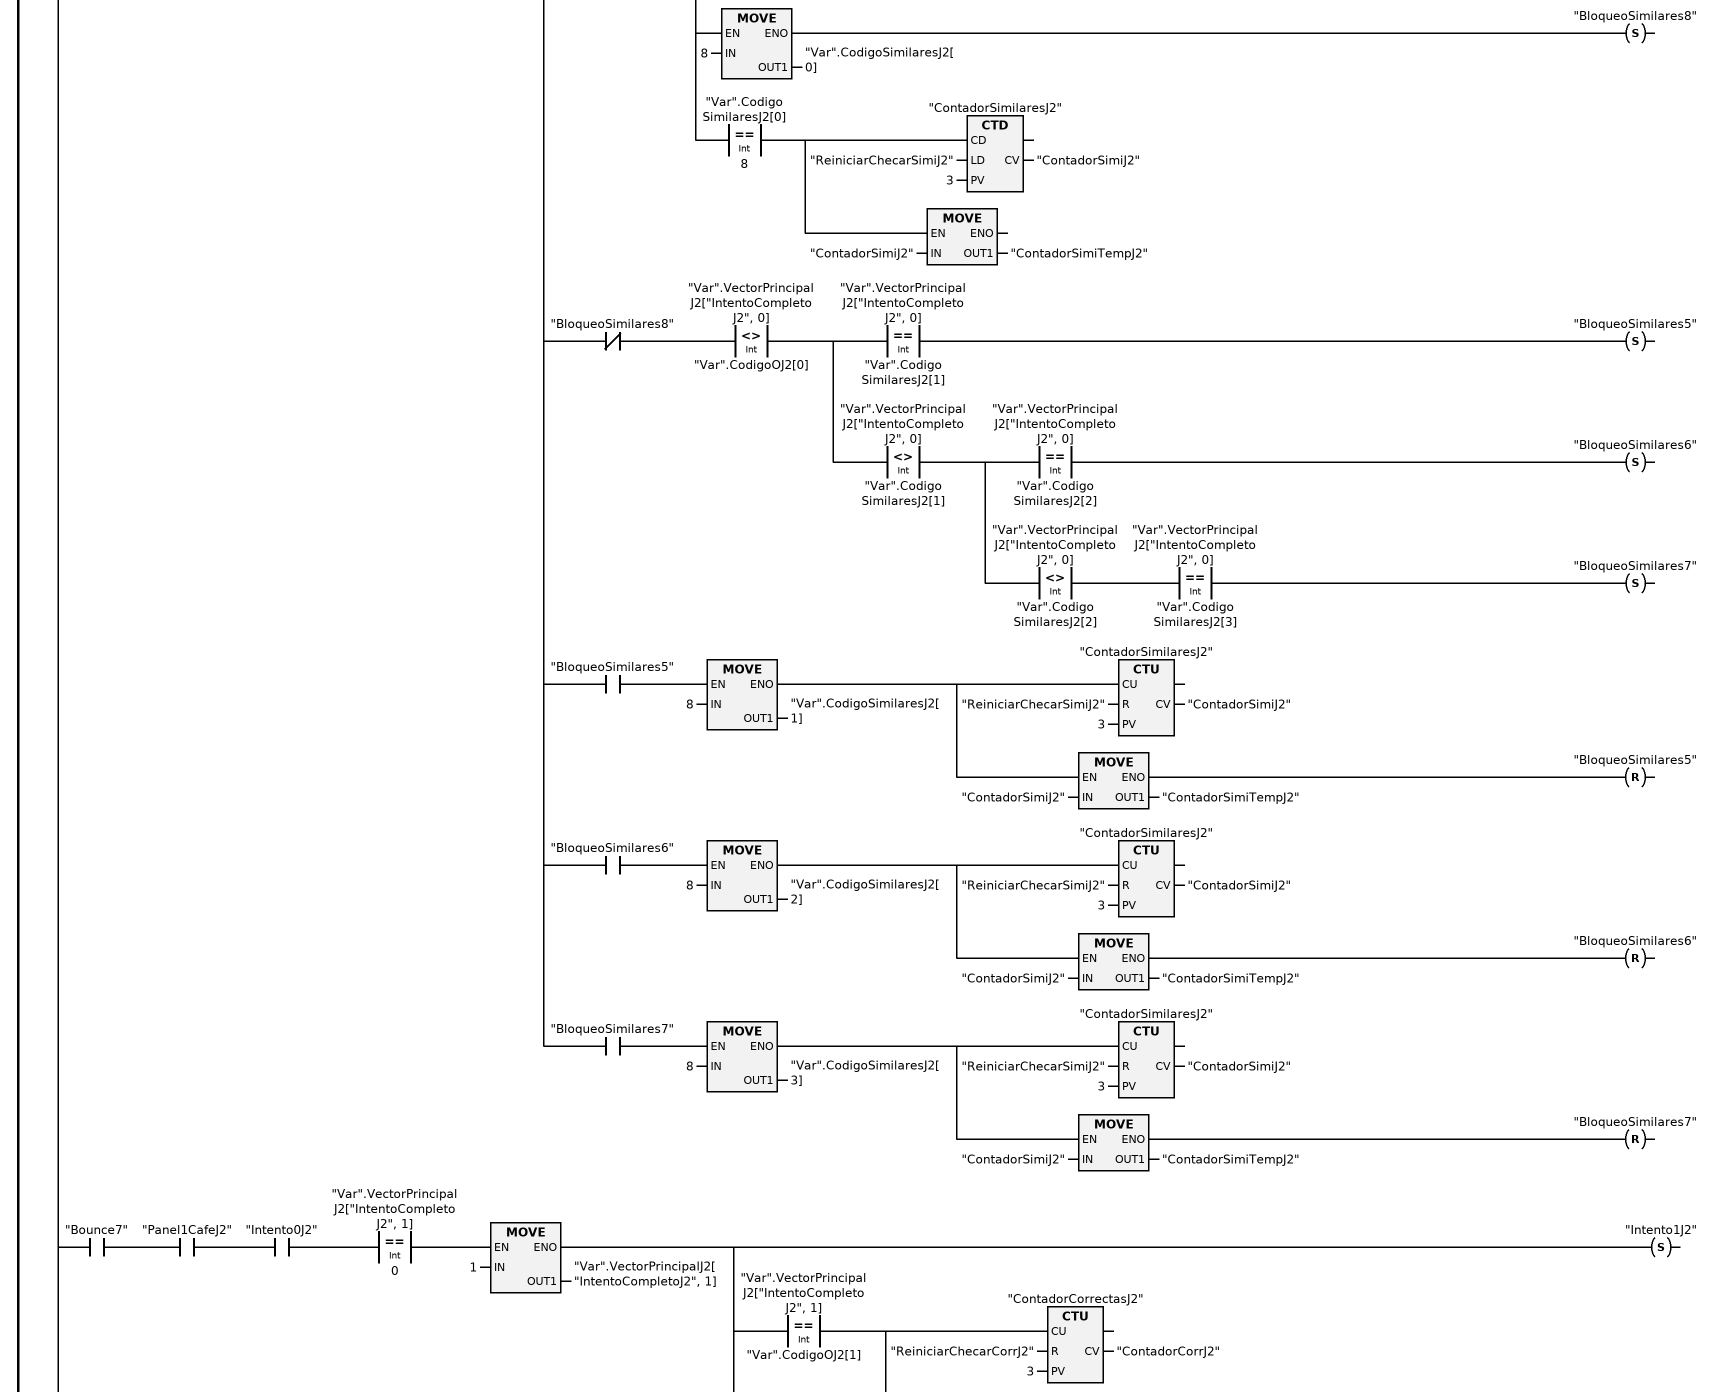
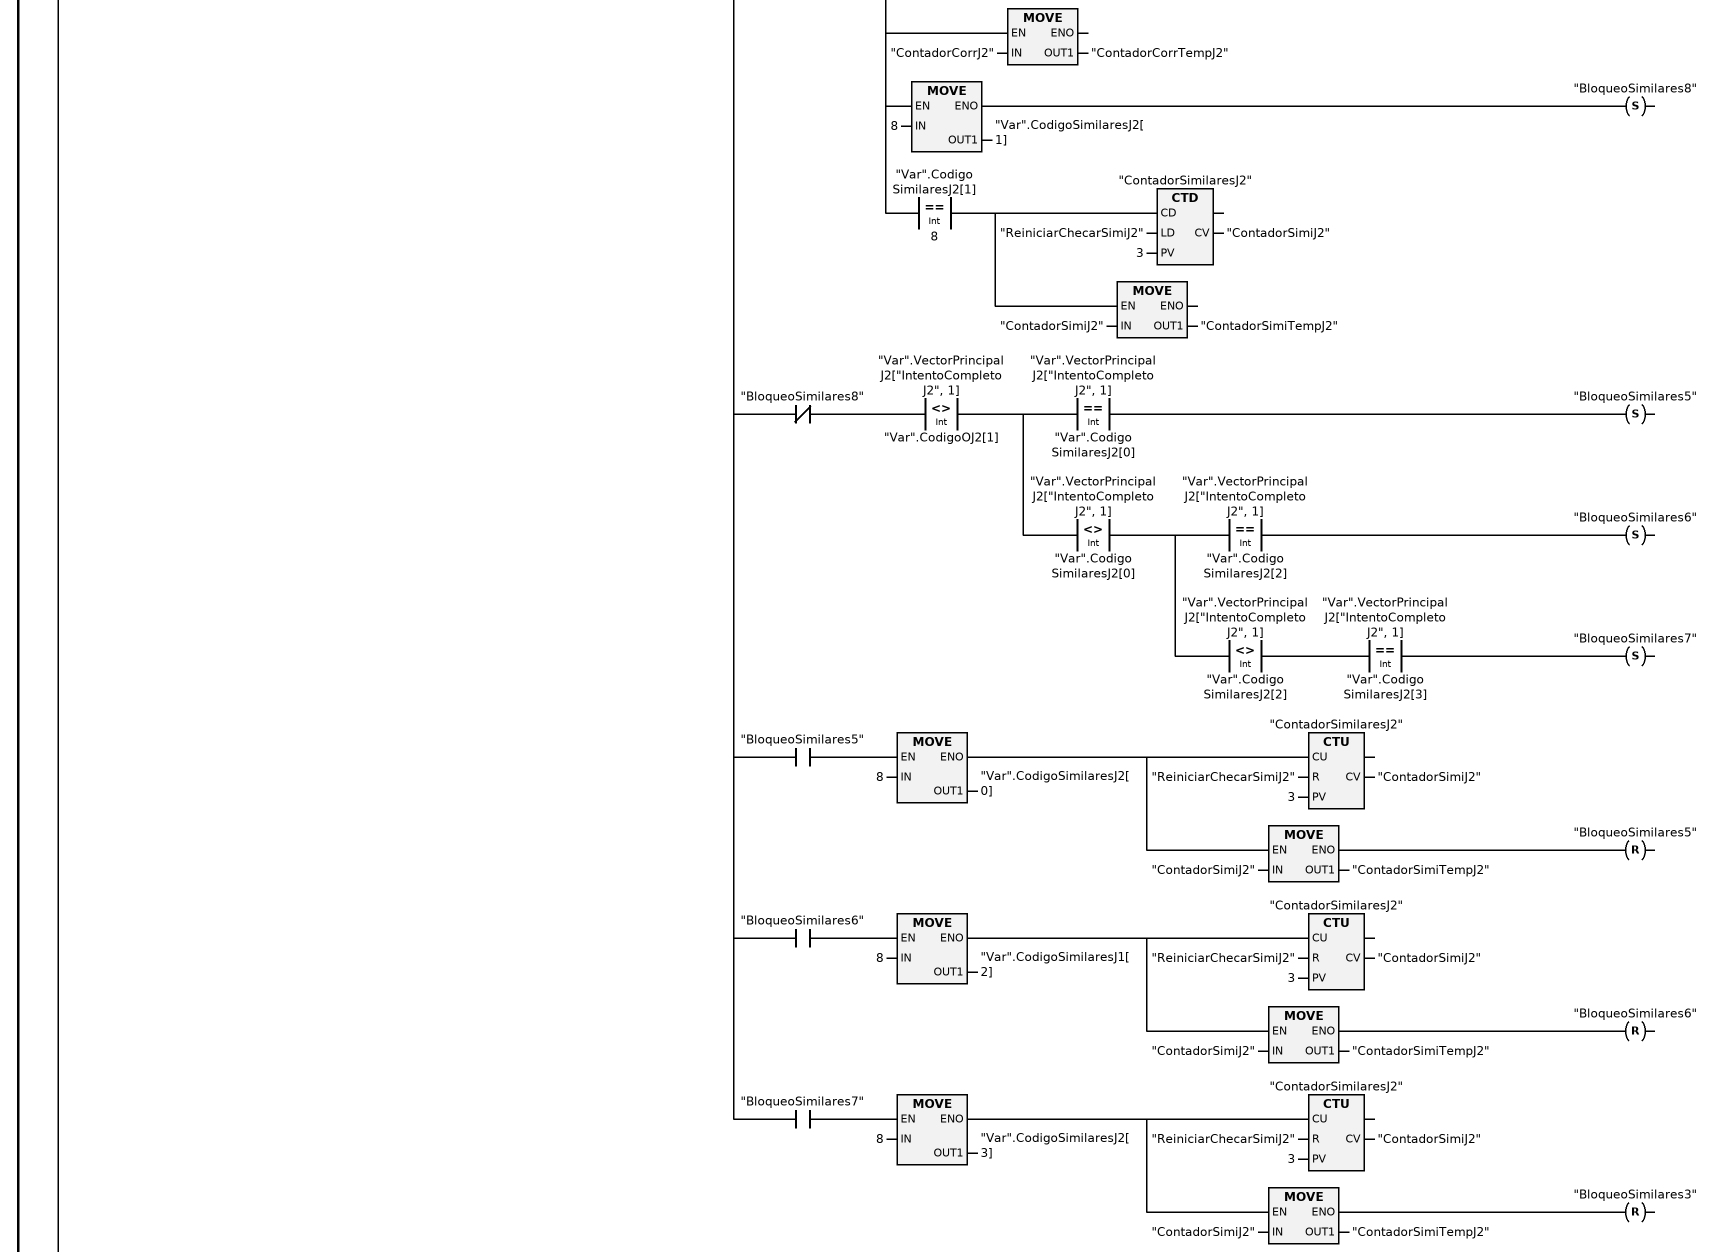
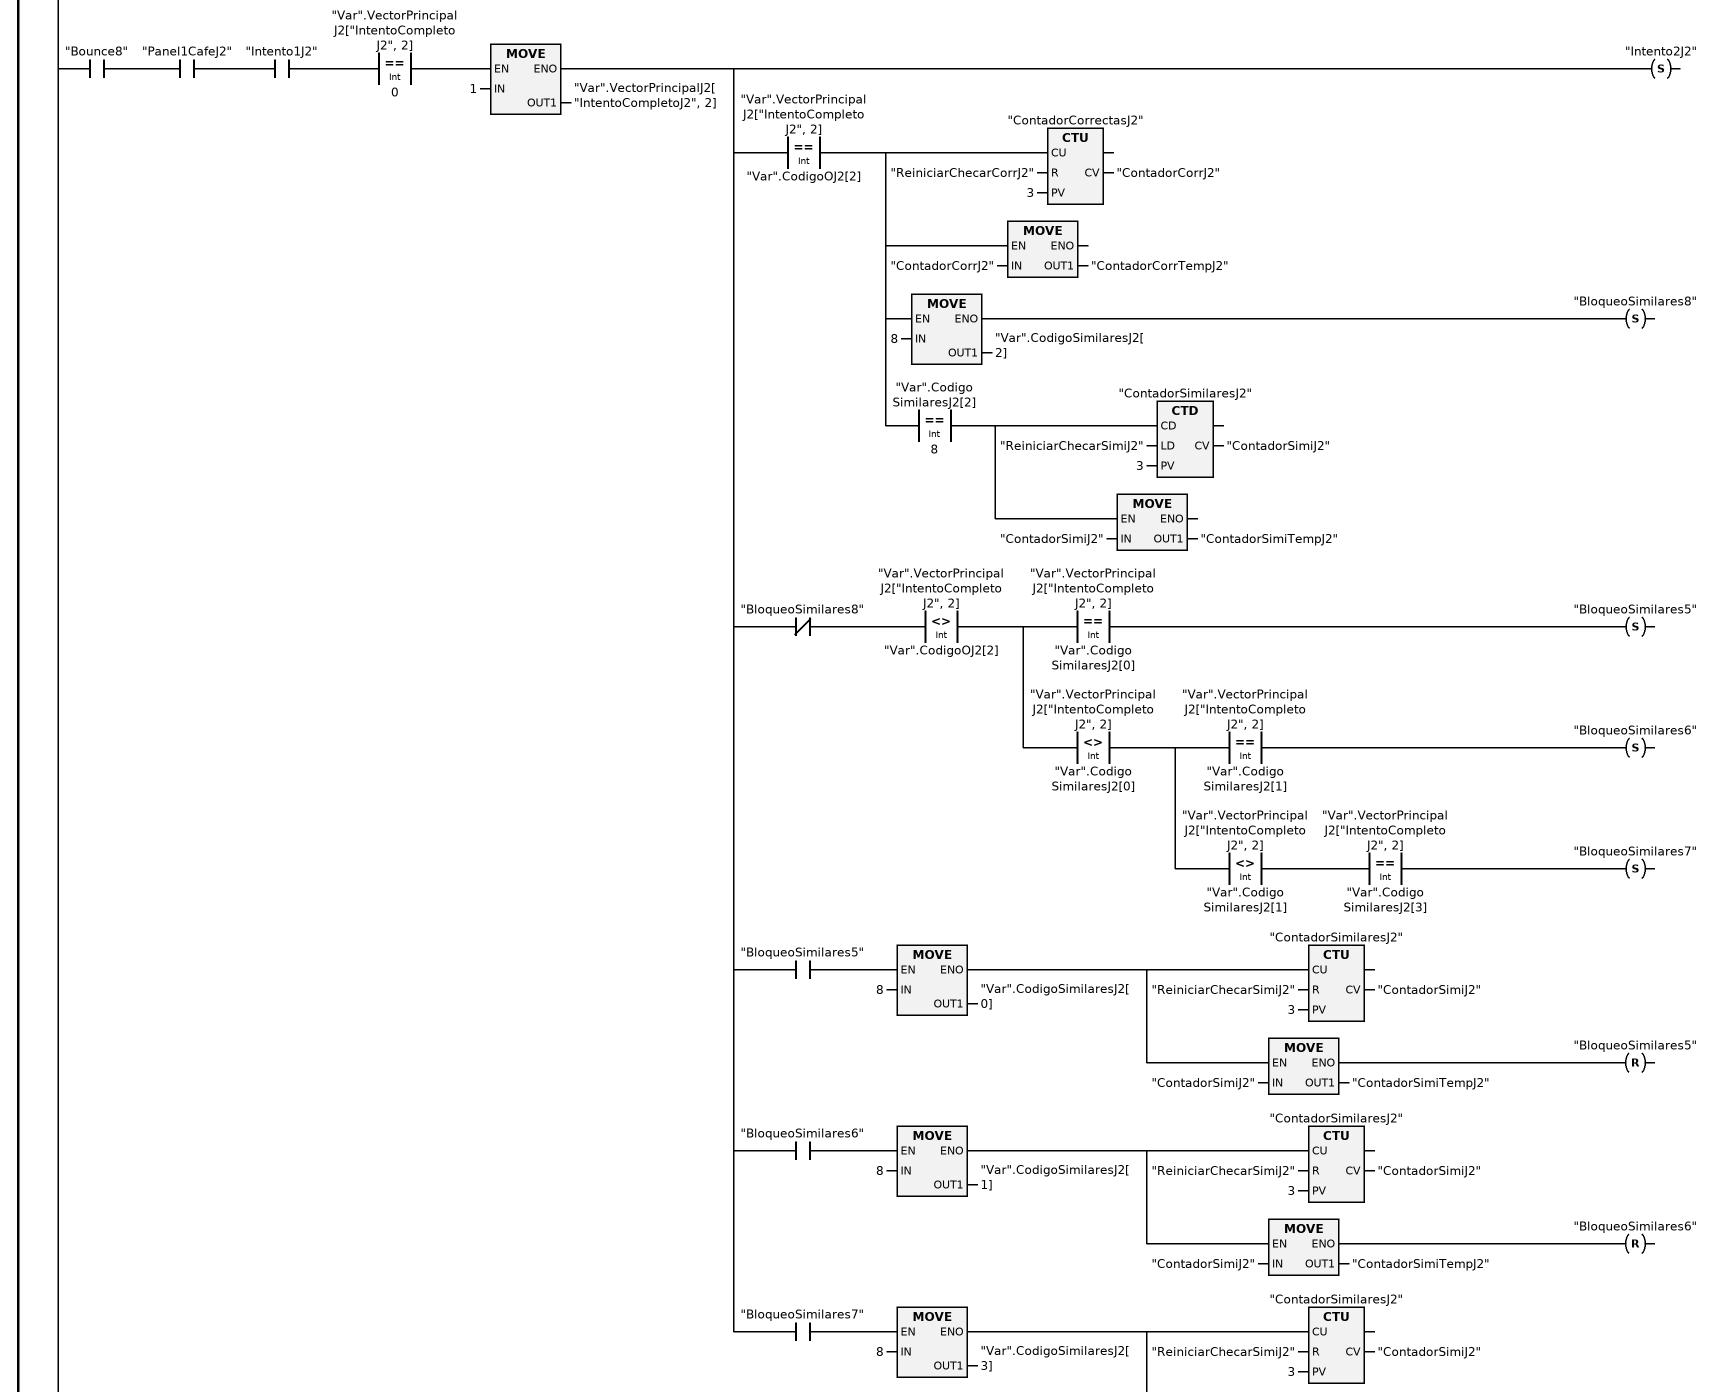
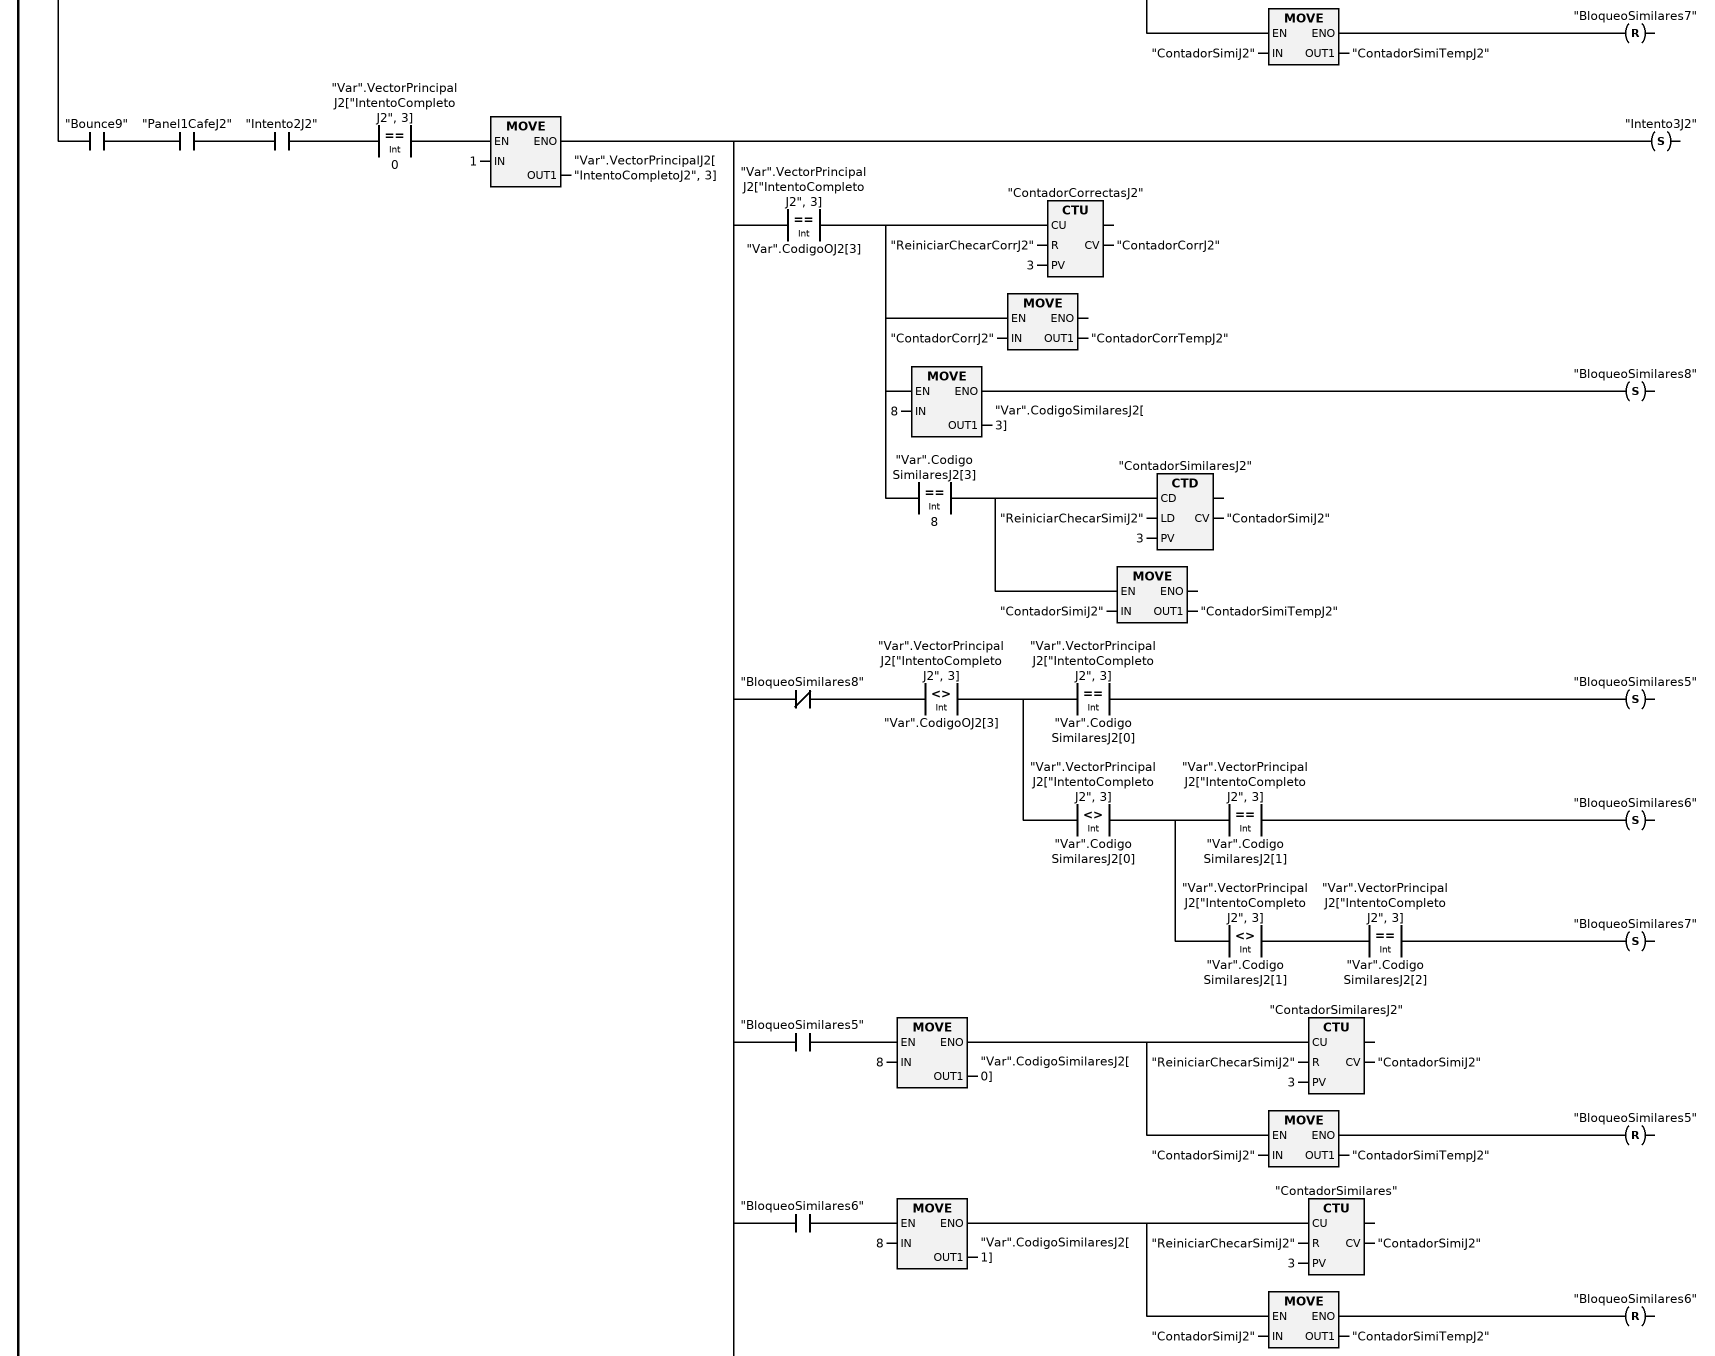
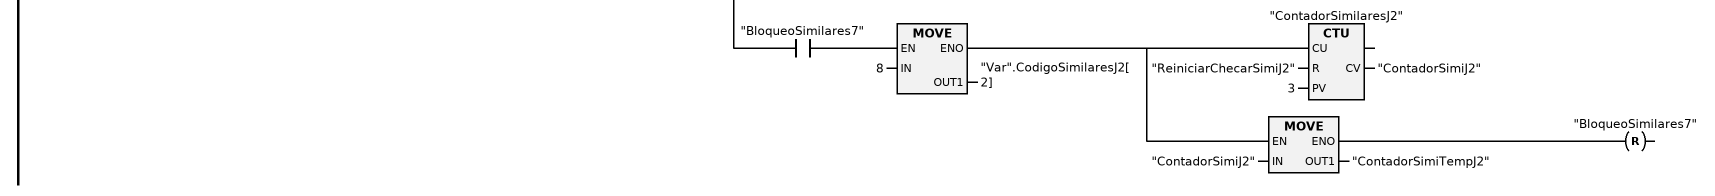
   // no SCL statement known for RBitfield: written as a call
   "IEC_Counter_0_DB_2".CTU(CU := "Intento3J2", R := "ReiniciarContadorJ2", PV := 10, CV => "IntentoCompletoJ2");
   "ReinicioCorrecto" := "IEC_Counter_0_DB_2".Q;
   #_w1 := "Intento3J2";
   IF #_w1 THEN
       RESET_BF(operand := "Bounce6", n := 4);
       "Bounce9" := FALSE;
       RESET_BF(operand := "Intento0J2", n := 4);
   END_IF;
   "CorrectasSimilaresJ2" := #_w1;
   IF #_w1 THEN
       MOVE_BLK(IN := "Var".CodigoSimilaresJ2Temp[0], COUNT := 4, OUT => "Var".CodigoSimilaresJ2[0]);
   END_IF;
   #_w2 := NOT "Panel2J2Activado" AND NOT "Panel1CafeJ2" AND NOT "Panel1RosaJ2" AND NOT "Panel1MoradoJ2" AND NOT "Panel1RojoJ2" AND NOT "Panel1AzulJ2" AND NOT "Panel1VerdeJ2" AND NOT "Panel1AmarilloJ2";
   #_w3 := #_w2 AND "Intento0J2" AND "Bounce10" AND NOT "Bounce7" AND NOT "Bounce8" AND NOT "Bounce9";
   IF #_w3 THEN
       "Bounce7" := TRUE;
       "BloqueoSimilares8" := FALSE;
   END_IF;
   #_w4 := #_w2 AND "Intento1J2" AND "Bounce10" AND "Bounce7" AND NOT "Bounce8" AND NOT "Bounce9";
   IF #_w4 THEN
       "Bounce8" := TRUE;
       "BloqueoSimilares8" := FALSE;
   END_IF;
   #_w5 := #_w2 AND "Intento2J2" AND "Bounce10" AND "Bounce7" AND "Bounce8" AND NOT "Bounce9";
   IF #_w5 THEN
       "Bounce9" := TRUE;
       "BloqueoSimilares8" := FALSE;
   END_IF;
   IF #_w2 AND "Bounce10" THEN
       "Bounce6" := TRUE;
       "BloqueoSimilares8" := FALSE;
   END_IF;
   #_w6 := "Panel1CafeJ2" AND ("Var".VectorPrincipalJ2["IntentoCompletoJ2", 0] = 0) AND "Bounce6";
   IF #_w6 THEN
       "Var".VectorPrincipalJ2["IntentoCompletoJ2", 0] := 1;
       "Intento0J2" := TRUE;
   END_IF;
   #_w7 := #_w6 AND ("Var".VectorPrincipalJ2["IntentoCompletoJ2", 0] = "Var".CodigoOJ2[0]);
   "ContadorCorrectasJ2".CTU(CU := #_w7, R := "ReiniciarChecarCorrJ2", PV := 3, CV => "ContadorCorrJ2");
   IF #_w7 THEN
       "ContadorCorrTempJ2" := "ContadorCorrJ2";
       "Var".CodigoSimilaresJ2[0] := 8;
       "BloqueoSimilares8" := TRUE;
   END_IF;
   #_w8 := #_w7 AND ("Var".CodigoSimilaresJ2[0] = 8);
   "ContadorSimilaresJ2".CTD(CD := #_w8, LD := "ReiniciarChecarSimiJ2", PV := 3, CV => "ContadorSimiJ2");
   IF #_w8 THEN "ContadorSimiTempJ2" := "ContadorSimiJ2"; END_IF;
   #_w9 := #_w6 AND NOT "BloqueoSimilares8" AND ("Var".VectorPrincipalJ2["IntentoCompletoJ2", 0] <> "Var".CodigoOJ2[0]);
   IF #_w9 AND ("Var".VectorPrincipalJ2["IntentoCompletoJ2", 0] = "Var".CodigoSimilaresJ2[1]) THEN
       "BloqueoSimilares5" := TRUE;
   END_IF;
   #_w10 := #_w9 AND ("Var".VectorPrincipalJ2["IntentoCompletoJ2", 0] <> "Var".CodigoSimilaresJ2[1]);
   IF #_w10 AND ("Var".VectorPrincipalJ2["IntentoCompletoJ2", 0] = "Var".CodigoSimilaresJ2[2]) THEN
       "BloqueoSimilares6" := TRUE;
   END_IF;
   IF #_w10 AND ("Var".VectorPrincipalJ2["IntentoCompletoJ2", 0] <> "Var".CodigoSimilaresJ2[2]) AND ("Var".VectorPrincipalJ2["IntentoCompletoJ2", 0] = "Var".CodigoSimilaresJ2[3]) THEN
       "BloqueoSimilares7" := TRUE;
   END_IF;
   #_w11 := #_w6 AND "BloqueoSimilares5";
   IF #_w11 THEN "Var".CodigoSimilaresJ2[1] := 8; END_IF;
   "ContadorSimilaresJ2".CTU(CU := #_w11, R := "ReiniciarChecarSimiJ2", PV := 3, CV => "ContadorSimiJ2");
   IF #_w11 THEN
       "ContadorSimiTempJ2" := "ContadorSimiJ2";
       "BloqueoSimilares5" := FALSE;
   END_IF;
   #_w12 := #_w6 AND "BloqueoSimilares6";
   IF #_w12 THEN "Var".CodigoSimilaresJ2[2] := 8; END_IF;
   "ContadorSimilaresJ2".CTU(CU := #_w12, R := "ReiniciarChecarSimiJ2", PV := 3, CV => "ContadorSimiJ2");
   IF #_w12 THEN
       "ContadorSimiTempJ2" := "ContadorSimiJ2";
       "BloqueoSimilares6" := FALSE;
   END_IF;
   #_w13 := #_w6 AND "BloqueoSimilares7";
   IF #_w13 THEN "Var".CodigoSimilaresJ2[3] := 8; END_IF;
   "ContadorSimilaresJ2".CTU(CU := #_w13, R := "ReiniciarChecarSimiJ2", PV := 3, CV => "ContadorSimiJ2");
   IF #_w13 THEN
       "ContadorSimiTempJ2" := "ContadorSimiJ2";
       "BloqueoSimilares7" := FALSE;
   END_IF;
   #_w14 := "Panel1CafeJ2" AND "Bounce7" AND "Panel1CafeJ2" AND "Intento0J2" AND ("Var".VectorPrincipalJ2["IntentoCompletoJ2", 1] = 0);
   IF #_w14 THEN
       "Var".VectorPrincipalJ2["IntentoCompletoJ2", 1] := 1;
       "Intento1J2" := TRUE;
   END_IF;
   #_w15 := #_w14 AND ("Var".VectorPrincipalJ2["IntentoCompletoJ2", 1] = "Var".CodigoOJ2[1]);
   "ContadorCorrectasJ2".CTU(CU := #_w15, R := "ReiniciarChecarCorrJ2", PV := 3, CV => "ContadorCorrJ2");
   IF #_w15 THEN
       "ContadorCorrTempJ2" := "ContadorCorrJ2";
       "Var".CodigoSimilaresJ2[1] := 8;
       "BloqueoSimilares8" := TRUE;
   END_IF;
   #_w16 := #_w15 AND ("Var".CodigoSimilaresJ2[1] = 8);
   "ContadorSimilaresJ2".CTD(CD := #_w16, LD := "ReiniciarChecarSimiJ2", PV := 3, CV => "ContadorSimiJ2");
   IF #_w16 THEN "ContadorSimiTempJ2" := "ContadorSimiJ2"; END_IF;
   #_w17 := #_w14 AND NOT "BloqueoSimilares8" AND ("Var".VectorPrincipalJ2["IntentoCompletoJ2", 1] <> "Var".CodigoOJ2[1]);
   IF #_w17 AND ("Var".VectorPrincipalJ2["IntentoCompletoJ2", 1] = "Var".CodigoSimilaresJ2[0]) THEN
       "BloqueoSimilares5" := TRUE;
   END_IF;
   #_w18 := #_w17 AND ("Var".VectorPrincipalJ2["IntentoCompletoJ2", 1] <> "Var".CodigoSimilaresJ2[0]);
   IF #_w18 AND ("Var".VectorPrincipalJ2["IntentoCompletoJ2", 1] = "Var".CodigoSimilaresJ2[2]) THEN
       "BloqueoSimilares6" := TRUE;
   END_IF;
   IF #_w18 AND ("Var".VectorPrincipalJ2["IntentoCompletoJ2", 1] <> "Var".CodigoSimilaresJ2[2]) AND ("Var".VectorPrincipalJ2["IntentoCompletoJ2", 1] = "Var".CodigoSimilaresJ2[3]) THEN
       "BloqueoSimilares7" := TRUE;
   END_IF;
   #_w19 := #_w14 AND "BloqueoSimilares5";
   IF #_w19 THEN "Var".CodigoSimilaresJ2[0] := 8; END_IF;
   "ContadorSimilaresJ2".CTU(CU := #_w19, R := "ReiniciarChecarSimiJ2", PV := 3, CV => "ContadorSimiJ2");
   IF #_w19 THEN
       "ContadorSimiTempJ2" := "ContadorSimiJ2";
       "BloqueoSimilares5" := FALSE;
   END_IF;
   #_w20 := #_w14 AND "BloqueoSimilares6";
   IF #_w20 THEN "Var".CodigoSimilaresJ1[2] := 8; END_IF;
   "ContadorSimilaresJ2".CTU(CU := #_w20, R := "ReiniciarChecarSimiJ2", PV := 3, CV => "ContadorSimiJ2");
   IF #_w20 THEN
       "ContadorSimiTempJ2" := "ContadorSimiJ2";
       "BloqueoSimilares6" := FALSE;
   END_IF;
   #_w21 := #_w14 AND "BloqueoSimilares7";
   IF #_w21 THEN "Var".CodigoSimilaresJ2[3] := 8; END_IF;
   "ContadorSimilaresJ2".CTU(CU := #_w21, R := "ReiniciarChecarSimiJ2", PV := 3, CV => "ContadorSimiJ2");
   IF #_w21 THEN
       "ContadorSimiTempJ2" := "ContadorSimiJ2";
       "BloqueoSimilares3" := FALSE;
   END_IF;
   #_w22 := "Panel1CafeJ2" AND "Bounce8" AND "Panel1CafeJ2" AND "Intento1J2" AND ("Var".VectorPrincipalJ2["IntentoCompletoJ2", 2] = 0);
   IF #_w22 THEN
       "Var".VectorPrincipalJ2["IntentoCompletoJ2", 2] := 1;
       "Intento2J2" := TRUE;
   END_IF;
   #_w23 := #_w22 AND ("Var".VectorPrincipalJ2["IntentoCompletoJ2", 2] = "Var".CodigoOJ2[2]);
   "ContadorCorrectasJ2".CTU(CU := #_w23, R := "ReiniciarChecarCorrJ2", PV := 3, CV => "ContadorCorrJ2");
   IF #_w23 THEN
       "ContadorCorrTempJ2" := "ContadorCorrJ2";
       "Var".CodigoSimilaresJ2[2] := 8;
       "BloqueoSimilares8" := TRUE;
   END_IF;
   #_w24 := #_w23 AND ("Var".CodigoSimilaresJ2[2] = 8);
   "ContadorSimilaresJ2".CTD(CD := #_w24, LD := "ReiniciarChecarSimiJ2", PV := 3, CV => "ContadorSimiJ2");
   IF #_w24 THEN "ContadorSimiTempJ2" := "ContadorSimiJ2"; END_IF;
   #_w25 := #_w22 AND NOT "BloqueoSimilares8" AND ("Var".VectorPrincipalJ2["IntentoCompletoJ2", 2] <> "Var".CodigoOJ2[2]);
   IF #_w25 AND ("Var".VectorPrincipalJ2["IntentoCompletoJ2", 2] = "Var".CodigoSimilaresJ2[0]) THEN
       "BloqueoSimilares5" := TRUE;
   END_IF;
   #_w26 := #_w25 AND ("Var".VectorPrincipalJ2["IntentoCompletoJ2", 2] <> "Var".CodigoSimilaresJ2[0]);
   IF #_w26 AND ("Var".VectorPrincipalJ2["IntentoCompletoJ2", 2] = "Var".CodigoSimilaresJ2[1]) THEN
       "BloqueoSimilares6" := TRUE;
   END_IF;
   IF #_w26 AND ("Var".VectorPrincipalJ2["IntentoCompletoJ2", 2] <> "Var".CodigoSimilaresJ2[1]) AND ("Var".VectorPrincipalJ2["IntentoCompletoJ2", 2] = "Var".CodigoSimilaresJ2[3]) THEN
       "BloqueoSimilares7" := TRUE;
   END_IF;
   #_w27 := #_w22 AND "BloqueoSimilares5";
   IF #_w27 THEN "Var".CodigoSimilaresJ2[0] := 8; END_IF;
   "ContadorSimilaresJ2".CTU(CU := #_w27, R := "ReiniciarChecarSimiJ2", PV := 3, CV => "ContadorSimiJ2");
   IF #_w27 THEN
       "ContadorSimiTempJ2" := "ContadorSimiJ2";
       "BloqueoSimilares5" := FALSE;
   END_IF;
   #_w28 := #_w22 AND "BloqueoSimilares6";
   IF #_w28 THEN "Var".CodigoSimilaresJ2[1] := 8; END_IF;
   "ContadorSimilaresJ2".CTU(CU := #_w28, R := "ReiniciarChecarSimiJ2", PV := 3, CV => "ContadorSimiJ2");
   IF #_w28 THEN
       "ContadorSimiTempJ2" := "ContadorSimiJ2";
       "BloqueoSimilares6" := FALSE;
   END_IF;
   #_w29 := #_w22 AND "BloqueoSimilares7";
   IF #_w29 THEN "Var".CodigoSimilaresJ2[3] := 8; END_IF;
   "ContadorSimilaresJ2".CTU(CU := #_w29, R := "ReiniciarChecarSimiJ2", PV := 3, CV => "ContadorSimiJ2");
   IF #_w29 THEN
       "ContadorSimiTempJ2" := "ContadorSimiJ2";
       "BloqueoSimilares7" := FALSE;
   END_IF;
   #_w30 := "Panel1CafeJ2" AND "Bounce9" AND "Panel1CafeJ2" AND "Intento2J2" AND ("Var".VectorPrincipalJ2["IntentoCompletoJ2", 3] = 0);
   IF #_w30 THEN
       "Var".VectorPrincipalJ2["IntentoCompletoJ2", 3] := 1;
       "Intento3J2" := TRUE;
   END_IF;
   #_w31 := #_w30 AND ("Var".VectorPrincipalJ2["IntentoCompletoJ2", 3] = "Var".CodigoOJ2[3]);
   "ContadorCorrectasJ2".CTU(CU := #_w31, R := "ReiniciarChecarCorrJ2", PV := 3, CV => "ContadorCorrJ2");
   IF #_w31 THEN
       "ContadorCorrTempJ2" := "ContadorCorrJ2";
       "Var".CodigoSimilaresJ2[3] := 8;
       "BloqueoSimilares8" := TRUE;
   END_IF;
   #_w32 := #_w31 AND ("Var".CodigoSimilaresJ2[3] = 8);
   "ContadorSimilaresJ2".CTD(CD := #_w32, LD := "ReiniciarChecarSimiJ2", PV := 3, CV => "ContadorSimiJ2");
   IF #_w32 THEN "ContadorSimiTempJ2" := "ContadorSimiJ2"; END_IF;
   #_w33 := #_w30 AND NOT "BloqueoSimilares8" AND ("Var".VectorPrincipalJ2["IntentoCompletoJ2", 3] <> "Var".CodigoOJ2[3]);
   IF #_w33 AND ("Var".VectorPrincipalJ2["IntentoCompletoJ2", 3] = "Var".CodigoSimilaresJ2[0]) THEN
       "BloqueoSimilares5" := TRUE;
   END_IF;
   #_w34 := #_w33 AND ("Var".VectorPrincipalJ2["IntentoCompletoJ2", 3] <> "Var".CodigoSimilaresJ2[0]);
   IF #_w34 AND ("Var".VectorPrincipalJ2["IntentoCompletoJ2", 3] = "Var".CodigoSimilaresJ2[1]) THEN
       "BloqueoSimilares6" := TRUE;
   END_IF;
   IF #_w34 AND ("Var".VectorPrincipalJ2["IntentoCompletoJ2", 3] <> "Var".CodigoSimilaresJ2[1]) AND ("Var".VectorPrincipalJ2["IntentoCompletoJ2", 3] = "Var".CodigoSimilaresJ2[2]) THEN
       "BloqueoSimilares7" := TRUE;
   END_IF;
   #_w35 := #_w30 AND "BloqueoSimilares5";
   IF #_w35 THEN "Var".CodigoSimilaresJ2[0] := 8; END_IF;
   "ContadorSimilaresJ2".CTU(CU := #_w35, R := "ReiniciarChecarSimiJ2", PV := 3, CV => "ContadorSimiJ2");
   IF #_w35 THEN
       "ContadorSimiTempJ2" := "ContadorSimiJ2";
       "BloqueoSimilares5" := FALSE;
   END_IF;
   #_w36 := #_w30 AND "BloqueoSimilares6";
   IF #_w36 THEN "Var".CodigoSimilaresJ2[1] := 8; END_IF;
   "ContadorSimilares".CTU(CU := #_w36, R := "ReiniciarChecarSimiJ2", PV := 3, CV => "ContadorSimiJ2");
   IF #_w36 THEN
       "ContadorSimiTempJ2" := "ContadorSimiJ2";
       "BloqueoSimilares6" := FALSE;
   END_IF;
   #_w37 := #_w30 AND "BloqueoSimilares7";
   IF #_w37 THEN "Var".CodigoSimilaresJ2[2] := 8; END_IF;
   "ContadorSimilaresJ2".CTU(CU := #_w37, R := "ReiniciarChecarSimiJ2", PV := 3, CV => "ContadorSimiJ2");
   IF #_w37 THEN
       "ContadorSimiTempJ2" := "ContadorSimiJ2";
       "BloqueoSimilares7" := FALSE;
   END_IF;
END_REGION

REGION Network 20: Rosa J2
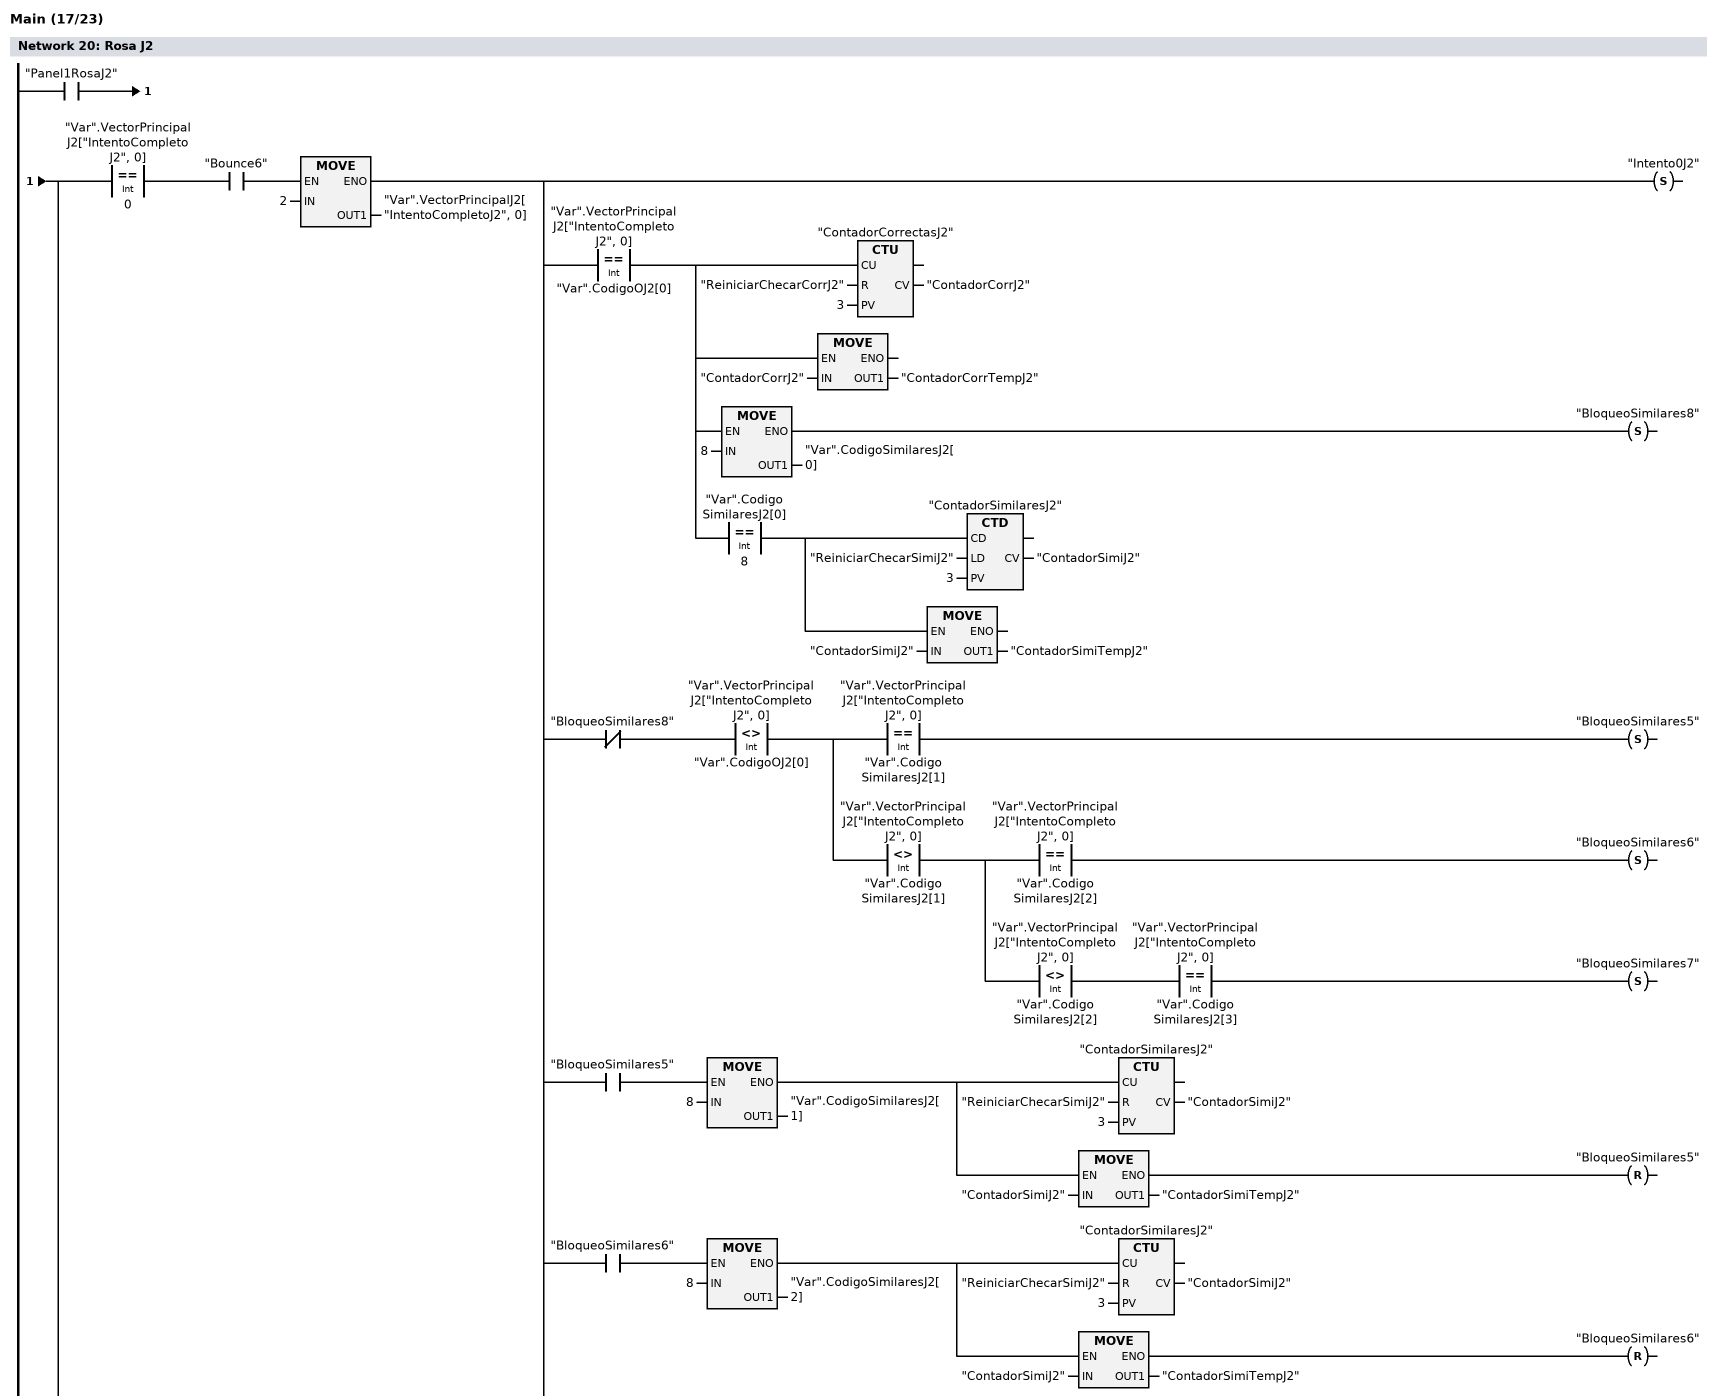
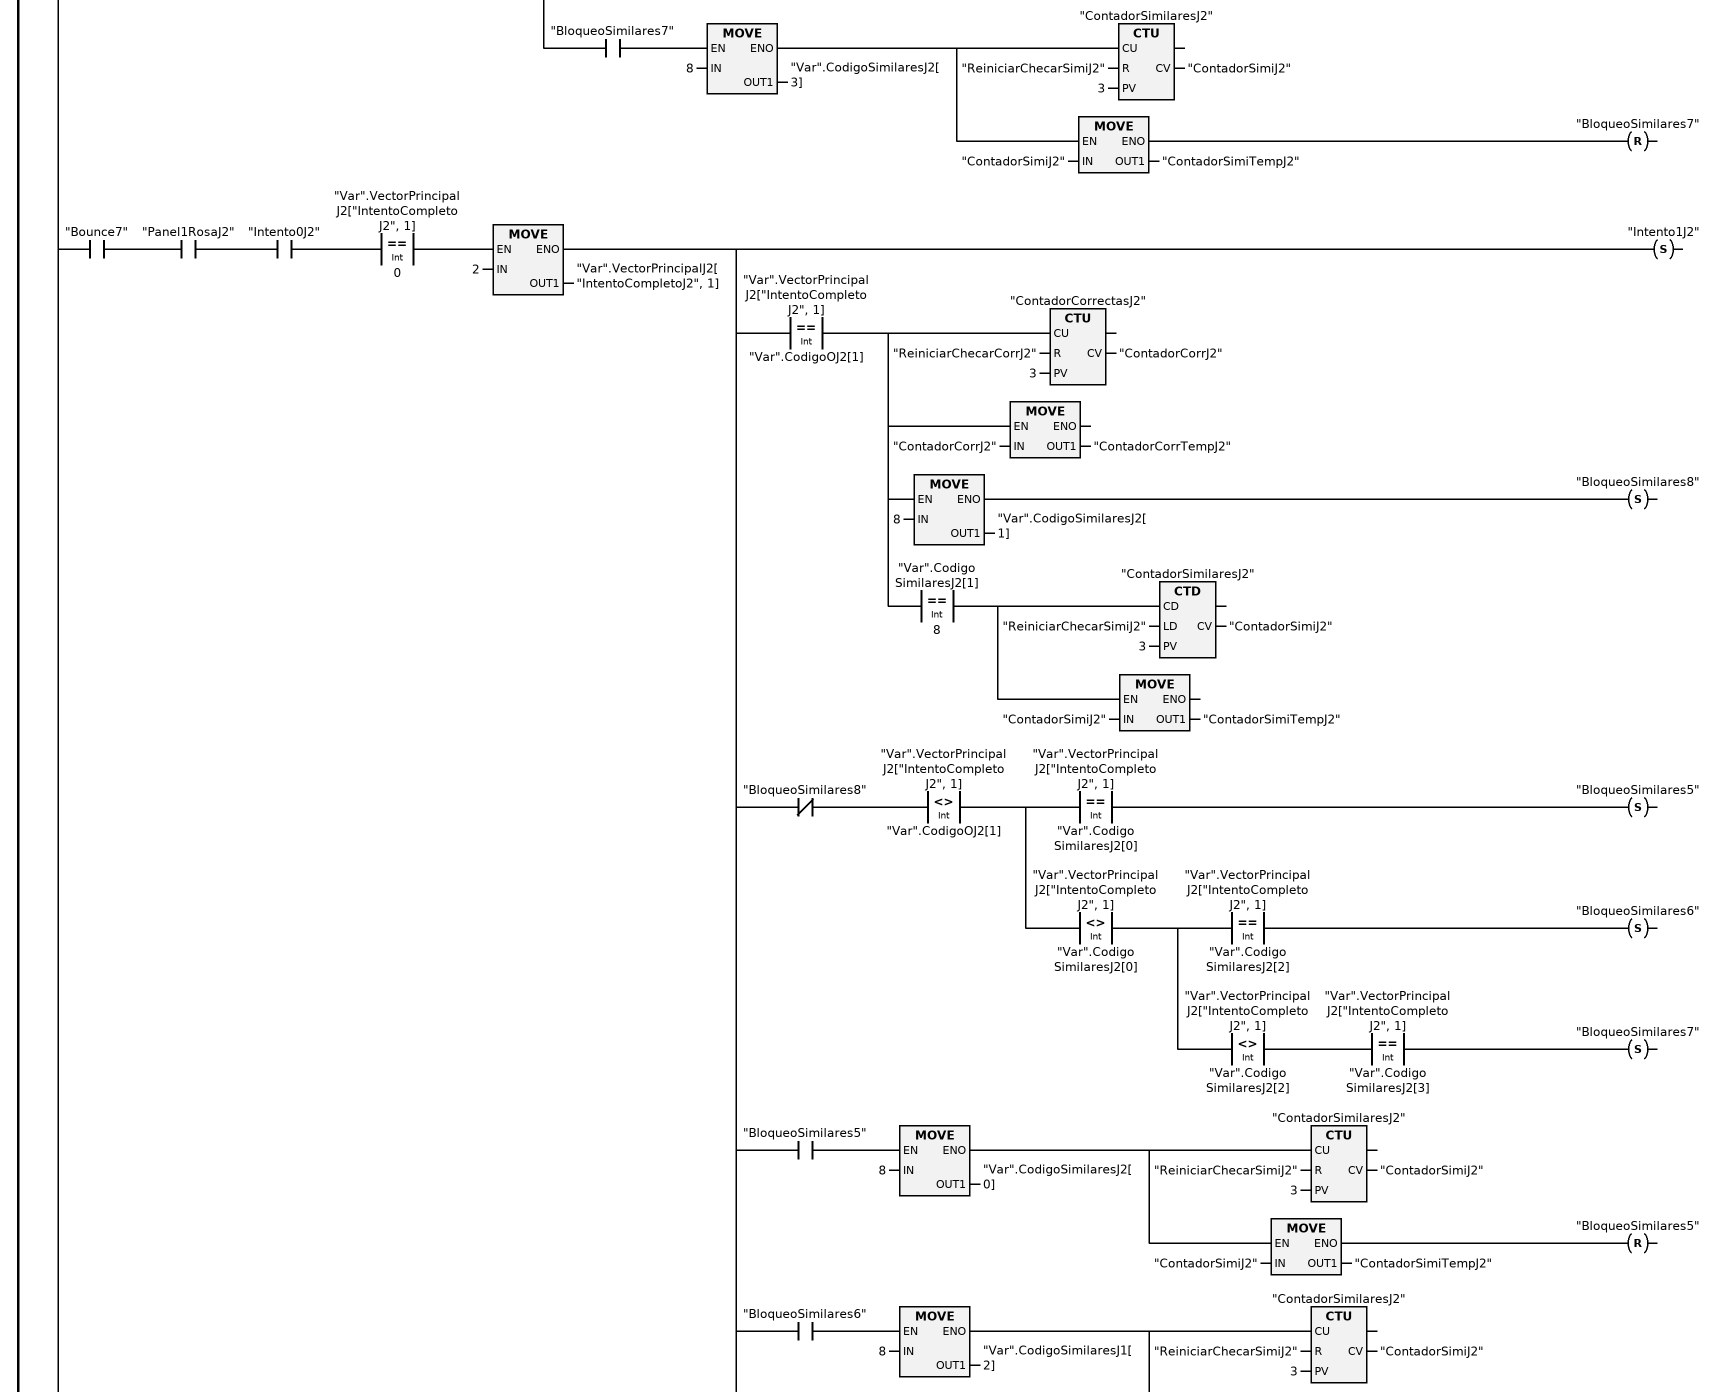
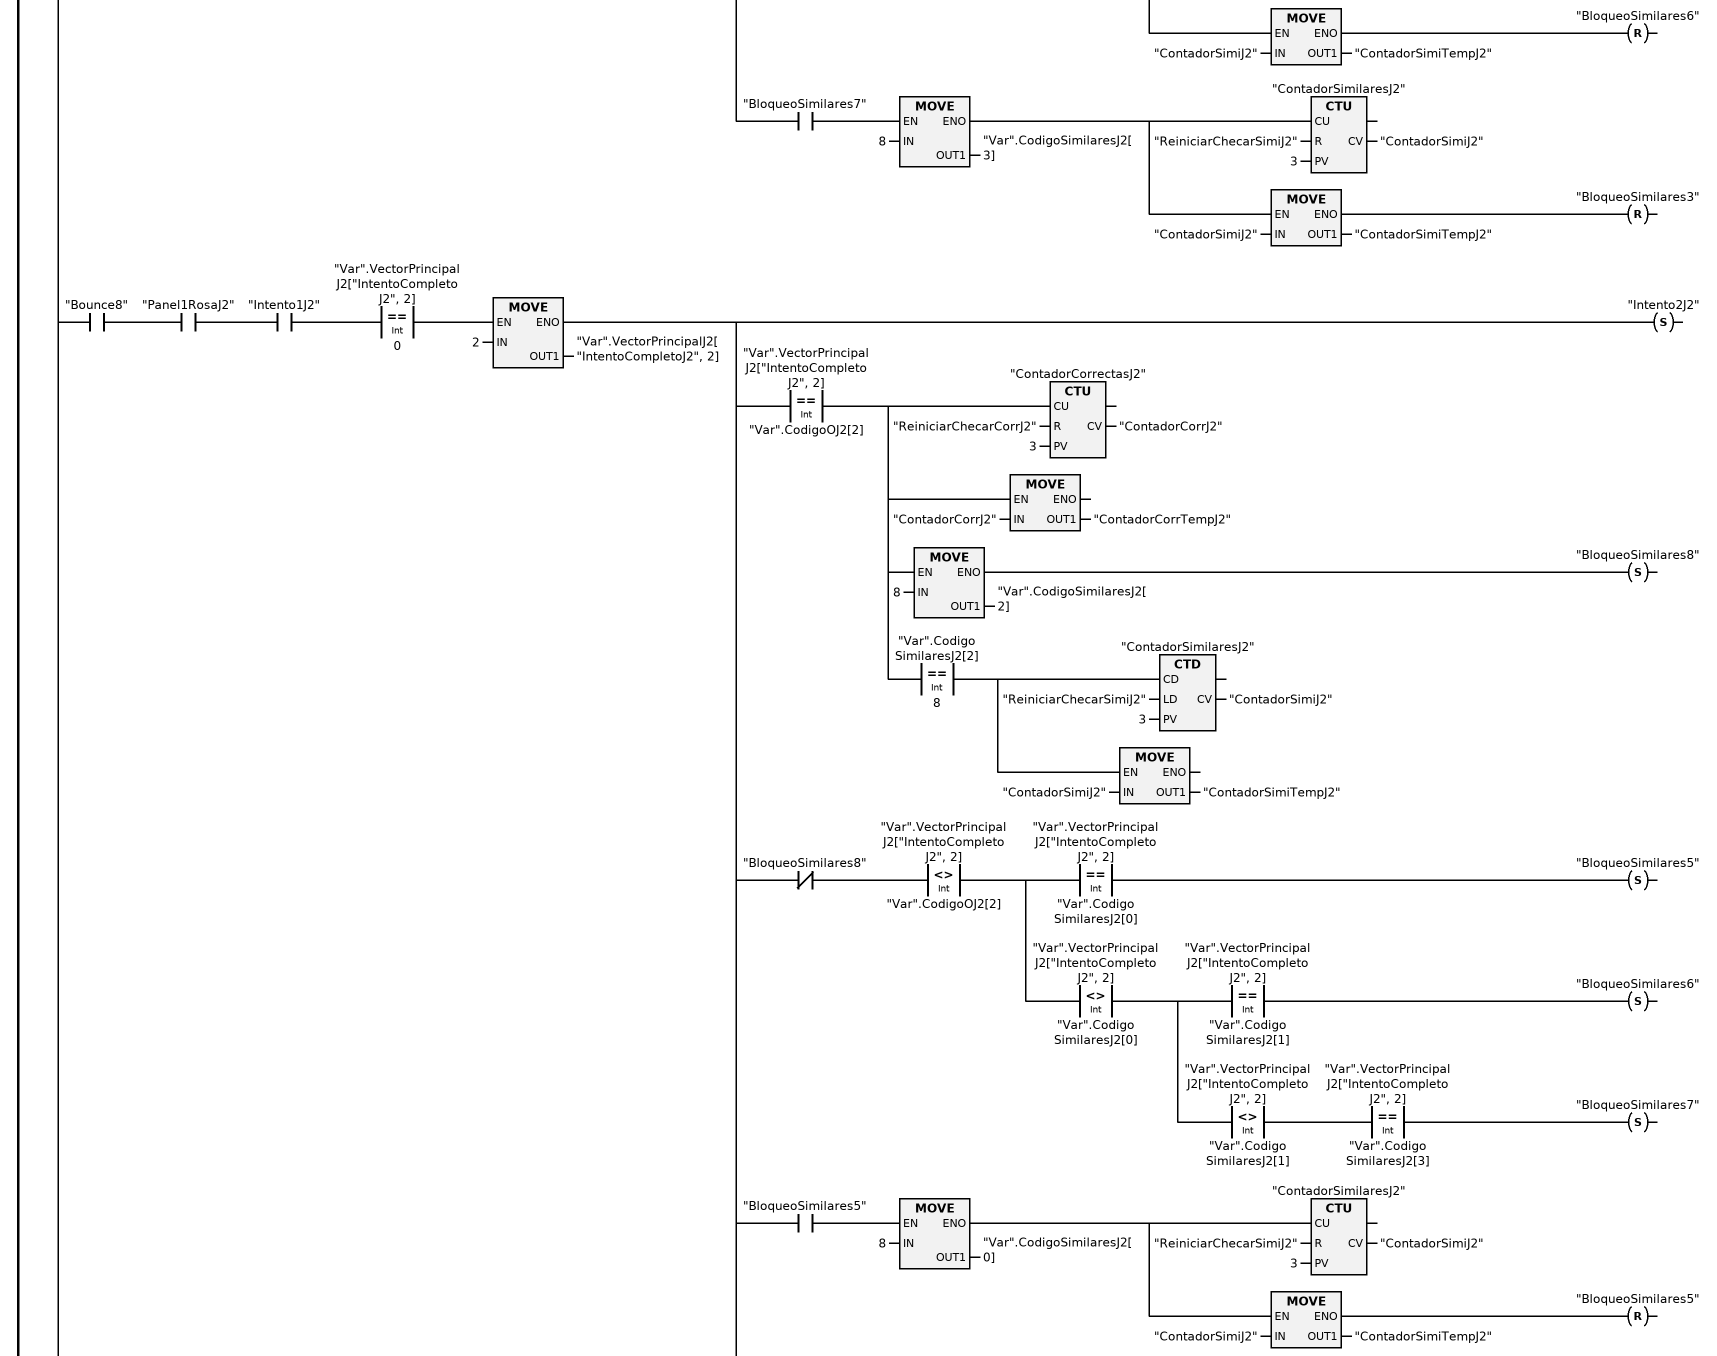
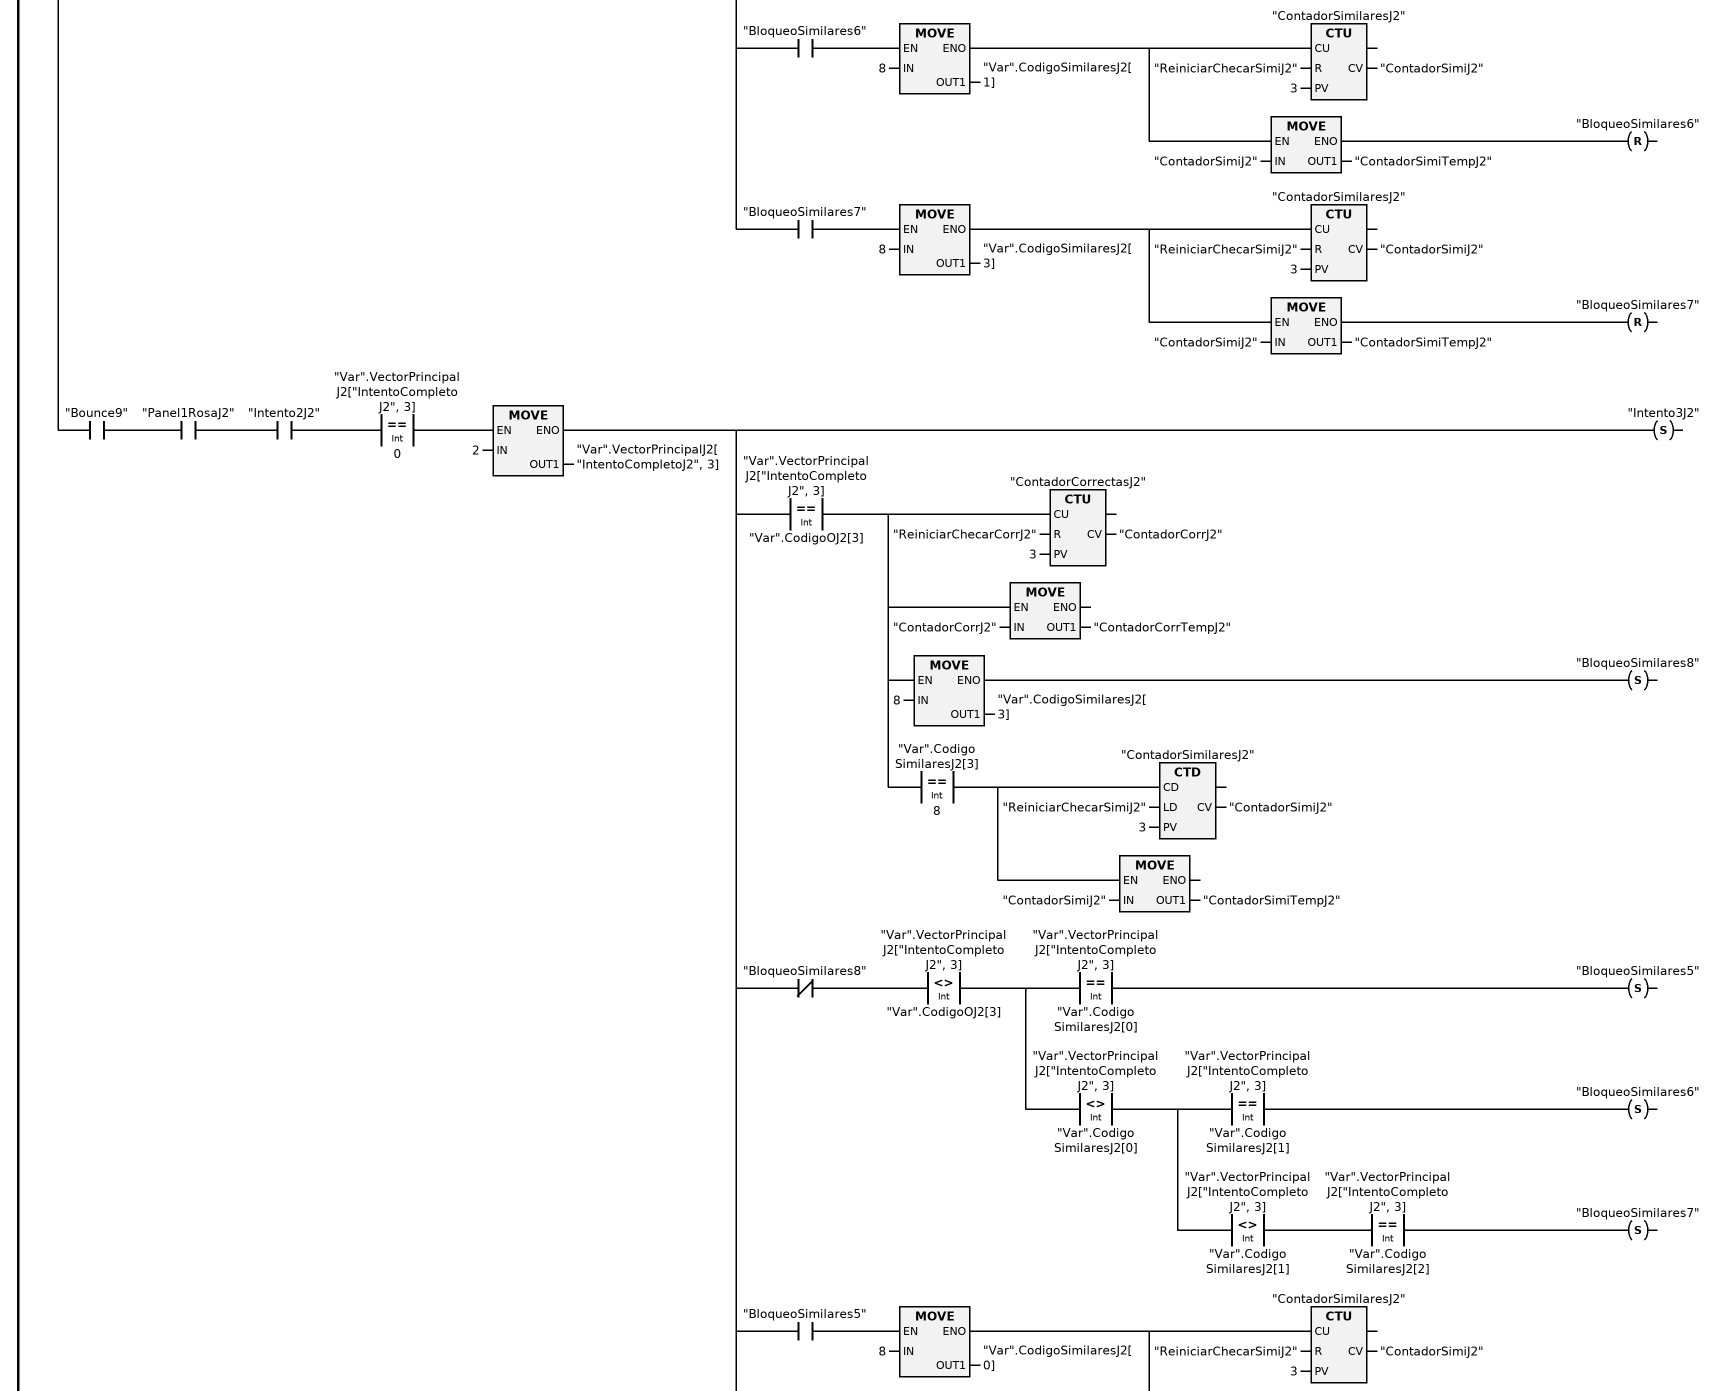
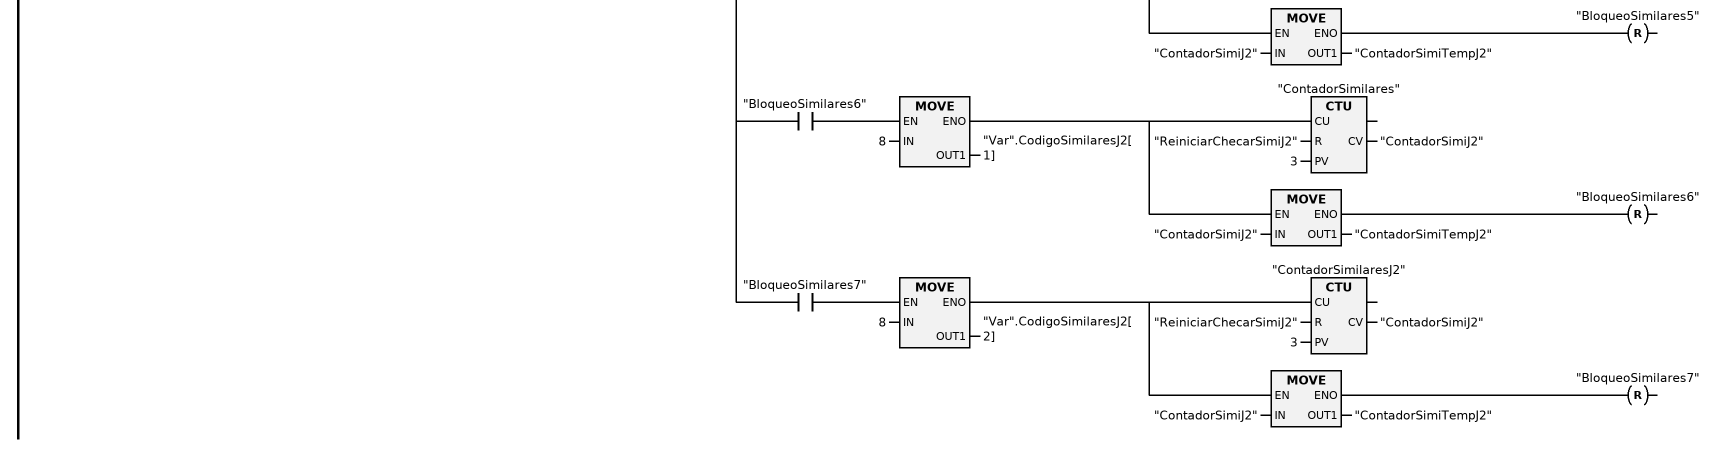
   #_w1 := "Panel1RosaJ2" AND ("Var".VectorPrincipalJ2["IntentoCompletoJ2", 0] = 0) AND "Bounce6";
   IF #_w1 THEN
       "Var".VectorPrincipalJ2["IntentoCompletoJ2", 0] := 2;
       "Intento0J2" := TRUE;
   END_IF;
   #_w2 := #_w1 AND ("Var".VectorPrincipalJ2["IntentoCompletoJ2", 0] = "Var".CodigoOJ2[0]);
   "ContadorCorrectasJ2".CTU(CU := #_w2, R := "ReiniciarChecarCorrJ2", PV := 3, CV => "ContadorCorrJ2");
   IF #_w2 THEN
       "ContadorCorrTempJ2" := "ContadorCorrJ2";
       "Var".CodigoSimilaresJ2[0] := 8;
       "BloqueoSimilares8" := TRUE;
   END_IF;
   #_w3 := #_w2 AND ("Var".CodigoSimilaresJ2[0] = 8);
   "ContadorSimilaresJ2".CTD(CD := #_w3, LD := "ReiniciarChecarSimiJ2", PV := 3, CV => "ContadorSimiJ2");
   IF #_w3 THEN "ContadorSimiTempJ2" := "ContadorSimiJ2"; END_IF;
   #_w4 := #_w1 AND NOT "BloqueoSimilares8" AND ("Var".VectorPrincipalJ2["IntentoCompletoJ2", 0] <> "Var".CodigoOJ2[0]);
   IF #_w4 AND ("Var".VectorPrincipalJ2["IntentoCompletoJ2", 0] = "Var".CodigoSimilaresJ2[1]) THEN
       "BloqueoSimilares5" := TRUE;
   END_IF;
   #_w5 := #_w4 AND ("Var".VectorPrincipalJ2["IntentoCompletoJ2", 0] <> "Var".CodigoSimilaresJ2[1]);
   IF #_w5 AND ("Var".VectorPrincipalJ2["IntentoCompletoJ2", 0] = "Var".CodigoSimilaresJ2[2]) THEN
       "BloqueoSimilares6" := TRUE;
   END_IF;
   IF #_w5 AND ("Var".VectorPrincipalJ2["IntentoCompletoJ2", 0] <> "Var".CodigoSimilaresJ2[2]) AND ("Var".VectorPrincipalJ2["IntentoCompletoJ2", 0] = "Var".CodigoSimilaresJ2[3]) THEN
       "BloqueoSimilares7" := TRUE;
   END_IF;
   #_w6 := #_w1 AND "BloqueoSimilares5";
   IF #_w6 THEN "Var".CodigoSimilaresJ2[1] := 8; END_IF;
   "ContadorSimilaresJ2".CTU(CU := #_w6, R := "ReiniciarChecarSimiJ2", PV := 3, CV => "ContadorSimiJ2");
   IF #_w6 THEN
       "ContadorSimiTempJ2" := "ContadorSimiJ2";
       "BloqueoSimilares5" := FALSE;
   END_IF;
   #_w7 := #_w1 AND "BloqueoSimilares6";
   IF #_w7 THEN "Var".CodigoSimilaresJ2[2] := 8; END_IF;
   "ContadorSimilaresJ2".CTU(CU := #_w7, R := "ReiniciarChecarSimiJ2", PV := 3, CV => "ContadorSimiJ2");
   IF #_w7 THEN
       "ContadorSimiTempJ2" := "ContadorSimiJ2";
       "BloqueoSimilares6" := FALSE;
   END_IF;
   #_w8 := #_w1 AND "BloqueoSimilares7";
   IF #_w8 THEN "Var".CodigoSimilaresJ2[3] := 8; END_IF;
   "ContadorSimilaresJ2".CTU(CU := #_w8, R := "ReiniciarChecarSimiJ2", PV := 3, CV => "ContadorSimiJ2");
   IF #_w8 THEN
       "ContadorSimiTempJ2" := "ContadorSimiJ2";
       "BloqueoSimilares7" := FALSE;
   END_IF;
   #_w9 := "Panel1RosaJ2" AND "Bounce7" AND "Panel1RosaJ2" AND "Intento0J2" AND ("Var".VectorPrincipalJ2["IntentoCompletoJ2", 1] = 0);
   IF #_w9 THEN
       "Var".VectorPrincipalJ2["IntentoCompletoJ2", 1] := 2;
       "Intento1J2" := TRUE;
   END_IF;
   #_w10 := #_w9 AND ("Var".VectorPrincipalJ2["IntentoCompletoJ2", 1] = "Var".CodigoOJ2[1]);
   "ContadorCorrectasJ2".CTU(CU := #_w10, R := "ReiniciarChecarCorrJ2", PV := 3, CV => "ContadorCorrJ2");
   IF #_w10 THEN
       "ContadorCorrTempJ2" := "ContadorCorrJ2";
       "Var".CodigoSimilaresJ2[1] := 8;
       "BloqueoSimilares8" := TRUE;
   END_IF;
   #_w11 := #_w10 AND ("Var".CodigoSimilaresJ2[1] = 8);
   "ContadorSimilaresJ2".CTD(CD := #_w11, LD := "ReiniciarChecarSimiJ2", PV := 3, CV => "ContadorSimiJ2");
   IF #_w11 THEN "ContadorSimiTempJ2" := "ContadorSimiJ2"; END_IF;
   #_w12 := #_w9 AND NOT "BloqueoSimilares8" AND ("Var".VectorPrincipalJ2["IntentoCompletoJ2", 1] <> "Var".CodigoOJ2[1]);
   IF #_w12 AND ("Var".VectorPrincipalJ2["IntentoCompletoJ2", 1] = "Var".CodigoSimilaresJ2[0]) THEN
       "BloqueoSimilares5" := TRUE;
   END_IF;
   #_w13 := #_w12 AND ("Var".VectorPrincipalJ2["IntentoCompletoJ2", 1] <> "Var".CodigoSimilaresJ2[0]);
   IF #_w13 AND ("Var".VectorPrincipalJ2["IntentoCompletoJ2", 1] = "Var".CodigoSimilaresJ2[2]) THEN
       "BloqueoSimilares6" := TRUE;
   END_IF;
   IF #_w13 AND ("Var".VectorPrincipalJ2["IntentoCompletoJ2", 1] <> "Var".CodigoSimilaresJ2[2]) AND ("Var".VectorPrincipalJ2["IntentoCompletoJ2", 1] = "Var".CodigoSimilaresJ2[3]) THEN
       "BloqueoSimilares7" := TRUE;
   END_IF;
   #_w14 := #_w9 AND "BloqueoSimilares5";
   IF #_w14 THEN "Var".CodigoSimilaresJ2[0] := 8; END_IF;
   "ContadorSimilaresJ2".CTU(CU := #_w14, R := "ReiniciarChecarSimiJ2", PV := 3, CV => "ContadorSimiJ2");
   IF #_w14 THEN
       "ContadorSimiTempJ2" := "ContadorSimiJ2";
       "BloqueoSimilares5" := FALSE;
   END_IF;
   #_w15 := #_w9 AND "BloqueoSimilares6";
   IF #_w15 THEN "Var".CodigoSimilaresJ1[2] := 8; END_IF;
   "ContadorSimilaresJ2".CTU(CU := #_w15, R := "ReiniciarChecarSimiJ2", PV := 3, CV => "ContadorSimiJ2");
   IF #_w15 THEN
       "ContadorSimiTempJ2" := "ContadorSimiJ2";
       "BloqueoSimilares6" := FALSE;
   END_IF;
   #_w16 := #_w9 AND "BloqueoSimilares7";
   IF #_w16 THEN "Var".CodigoSimilaresJ2[3] := 8; END_IF;
   "ContadorSimilaresJ2".CTU(CU := #_w16, R := "ReiniciarChecarSimiJ2", PV := 3, CV => "ContadorSimiJ2");
   IF #_w16 THEN
       "ContadorSimiTempJ2" := "ContadorSimiJ2";
       "BloqueoSimilares3" := FALSE;
   END_IF;
   #_w17 := "Panel1RosaJ2" AND "Bounce8" AND "Panel1RosaJ2" AND "Intento1J2" AND ("Var".VectorPrincipalJ2["IntentoCompletoJ2", 2] = 0);
   IF #_w17 THEN
       "Var".VectorPrincipalJ2["IntentoCompletoJ2", 2] := 2;
       "Intento2J2" := TRUE;
   END_IF;
   #_w18 := #_w17 AND ("Var".VectorPrincipalJ2["IntentoCompletoJ2", 2] = "Var".CodigoOJ2[2]);
   "ContadorCorrectasJ2".CTU(CU := #_w18, R := "ReiniciarChecarCorrJ2", PV := 3, CV => "ContadorCorrJ2");
   IF #_w18 THEN
       "ContadorCorrTempJ2" := "ContadorCorrJ2";
       "Var".CodigoSimilaresJ2[2] := 8;
       "BloqueoSimilares8" := TRUE;
   END_IF;
   #_w19 := #_w18 AND ("Var".CodigoSimilaresJ2[2] = 8);
   "ContadorSimilaresJ2".CTD(CD := #_w19, LD := "ReiniciarChecarSimiJ2", PV := 3, CV => "ContadorSimiJ2");
   IF #_w19 THEN "ContadorSimiTempJ2" := "ContadorSimiJ2"; END_IF;
   #_w20 := #_w17 AND NOT "BloqueoSimilares8" AND ("Var".VectorPrincipalJ2["IntentoCompletoJ2", 2] <> "Var".CodigoOJ2[2]);
   IF #_w20 AND ("Var".VectorPrincipalJ2["IntentoCompletoJ2", 2] = "Var".CodigoSimilaresJ2[0]) THEN
       "BloqueoSimilares5" := TRUE;
   END_IF;
   #_w21 := #_w20 AND ("Var".VectorPrincipalJ2["IntentoCompletoJ2", 2] <> "Var".CodigoSimilaresJ2[0]);
   IF #_w21 AND ("Var".VectorPrincipalJ2["IntentoCompletoJ2", 2] = "Var".CodigoSimilaresJ2[1]) THEN
       "BloqueoSimilares6" := TRUE;
   END_IF;
   IF #_w21 AND ("Var".VectorPrincipalJ2["IntentoCompletoJ2", 2] <> "Var".CodigoSimilaresJ2[1]) AND ("Var".VectorPrincipalJ2["IntentoCompletoJ2", 2] = "Var".CodigoSimilaresJ2[3]) THEN
       "BloqueoSimilares7" := TRUE;
   END_IF;
   #_w22 := #_w17 AND "BloqueoSimilares5";
   IF #_w22 THEN "Var".CodigoSimilaresJ2[0] := 8; END_IF;
   "ContadorSimilaresJ2".CTU(CU := #_w22, R := "ReiniciarChecarSimiJ2", PV := 3, CV => "ContadorSimiJ2");
   IF #_w22 THEN
       "ContadorSimiTempJ2" := "ContadorSimiJ2";
       "BloqueoSimilares5" := FALSE;
   END_IF;
   #_w23 := #_w17 AND "BloqueoSimilares6";
   IF #_w23 THEN "Var".CodigoSimilaresJ2[1] := 8; END_IF;
   "ContadorSimilaresJ2".CTU(CU := #_w23, R := "ReiniciarChecarSimiJ2", PV := 3, CV => "ContadorSimiJ2");
   IF #_w23 THEN
       "ContadorSimiTempJ2" := "ContadorSimiJ2";
       "BloqueoSimilares6" := FALSE;
   END_IF;
   #_w24 := #_w17 AND "BloqueoSimilares7";
   IF #_w24 THEN "Var".CodigoSimilaresJ2[3] := 8; END_IF;
   "ContadorSimilaresJ2".CTU(CU := #_w24, R := "ReiniciarChecarSimiJ2", PV := 3, CV => "ContadorSimiJ2");
   IF #_w24 THEN
       "ContadorSimiTempJ2" := "ContadorSimiJ2";
       "BloqueoSimilares7" := FALSE;
   END_IF;
   #_w25 := "Panel1RosaJ2" AND "Bounce9" AND "Panel1RosaJ2" AND "Intento2J2" AND ("Var".VectorPrincipalJ2["IntentoCompletoJ2", 3] = 0);
   IF #_w25 THEN
       "Var".VectorPrincipalJ2["IntentoCompletoJ2", 3] := 2;
       "Intento3J2" := TRUE;
   END_IF;
   #_w26 := #_w25 AND ("Var".VectorPrincipalJ2["IntentoCompletoJ2", 3] = "Var".CodigoOJ2[3]);
   "ContadorCorrectasJ2".CTU(CU := #_w26, R := "ReiniciarChecarCorrJ2", PV := 3, CV => "ContadorCorrJ2");
   IF #_w26 THEN
       "ContadorCorrTempJ2" := "ContadorCorrJ2";
       "Var".CodigoSimilaresJ2[3] := 8;
       "BloqueoSimilares8" := TRUE;
   END_IF;
   #_w27 := #_w26 AND ("Var".CodigoSimilaresJ2[3] = 8);
   "ContadorSimilaresJ2".CTD(CD := #_w27, LD := "ReiniciarChecarSimiJ2", PV := 3, CV => "ContadorSimiJ2");
   IF #_w27 THEN "ContadorSimiTempJ2" := "ContadorSimiJ2"; END_IF;
   #_w28 := #_w25 AND NOT "BloqueoSimilares8" AND ("Var".VectorPrincipalJ2["IntentoCompletoJ2", 3] <> "Var".CodigoOJ2[3]);
   IF #_w28 AND ("Var".VectorPrincipalJ2["IntentoCompletoJ2", 3] = "Var".CodigoSimilaresJ2[0]) THEN
       "BloqueoSimilares5" := TRUE;
   END_IF;
   #_w29 := #_w28 AND ("Var".VectorPrincipalJ2["IntentoCompletoJ2", 3] <> "Var".CodigoSimilaresJ2[0]);
   IF #_w29 AND ("Var".VectorPrincipalJ2["IntentoCompletoJ2", 3] = "Var".CodigoSimilaresJ2[1]) THEN
       "BloqueoSimilares6" := TRUE;
   END_IF;
   IF #_w29 AND ("Var".VectorPrincipalJ2["IntentoCompletoJ2", 3] <> "Var".CodigoSimilaresJ2[1]) AND ("Var".VectorPrincipalJ2["IntentoCompletoJ2", 3] = "Var".CodigoSimilaresJ2[2]) THEN
       "BloqueoSimilares7" := TRUE;
   END_IF;
   #_w30 := #_w25 AND "BloqueoSimilares5";
   IF #_w30 THEN "Var".CodigoSimilaresJ2[0] := 8; END_IF;
   "ContadorSimilaresJ2".CTU(CU := #_w30, R := "ReiniciarChecarSimiJ2", PV := 3, CV => "ContadorSimiJ2");
   IF #_w30 THEN
       "ContadorSimiTempJ2" := "ContadorSimiJ2";
       "BloqueoSimilares5" := FALSE;
   END_IF;
   #_w31 := #_w25 AND "BloqueoSimilares6";
   IF #_w31 THEN "Var".CodigoSimilaresJ2[1] := 8; END_IF;
   "ContadorSimilares".CTU(CU := #_w31, R := "ReiniciarChecarSimiJ2", PV := 3, CV => "ContadorSimiJ2");
   IF #_w31 THEN
       "ContadorSimiTempJ2" := "ContadorSimiJ2";
       "BloqueoSimilares6" := FALSE;
   END_IF;
   #_w32 := #_w25 AND "BloqueoSimilares7";
   IF #_w32 THEN "Var".CodigoSimilaresJ2[2] := 8; END_IF;
   "ContadorSimilaresJ2".CTU(CU := #_w32, R := "ReiniciarChecarSimiJ2", PV := 3, CV => "ContadorSimiJ2");
   IF #_w32 THEN
       "ContadorSimiTempJ2" := "ContadorSimiJ2";
       "BloqueoSimilares7" := FALSE;
   END_IF;
END_REGION

REGION Network 21: Morado J2
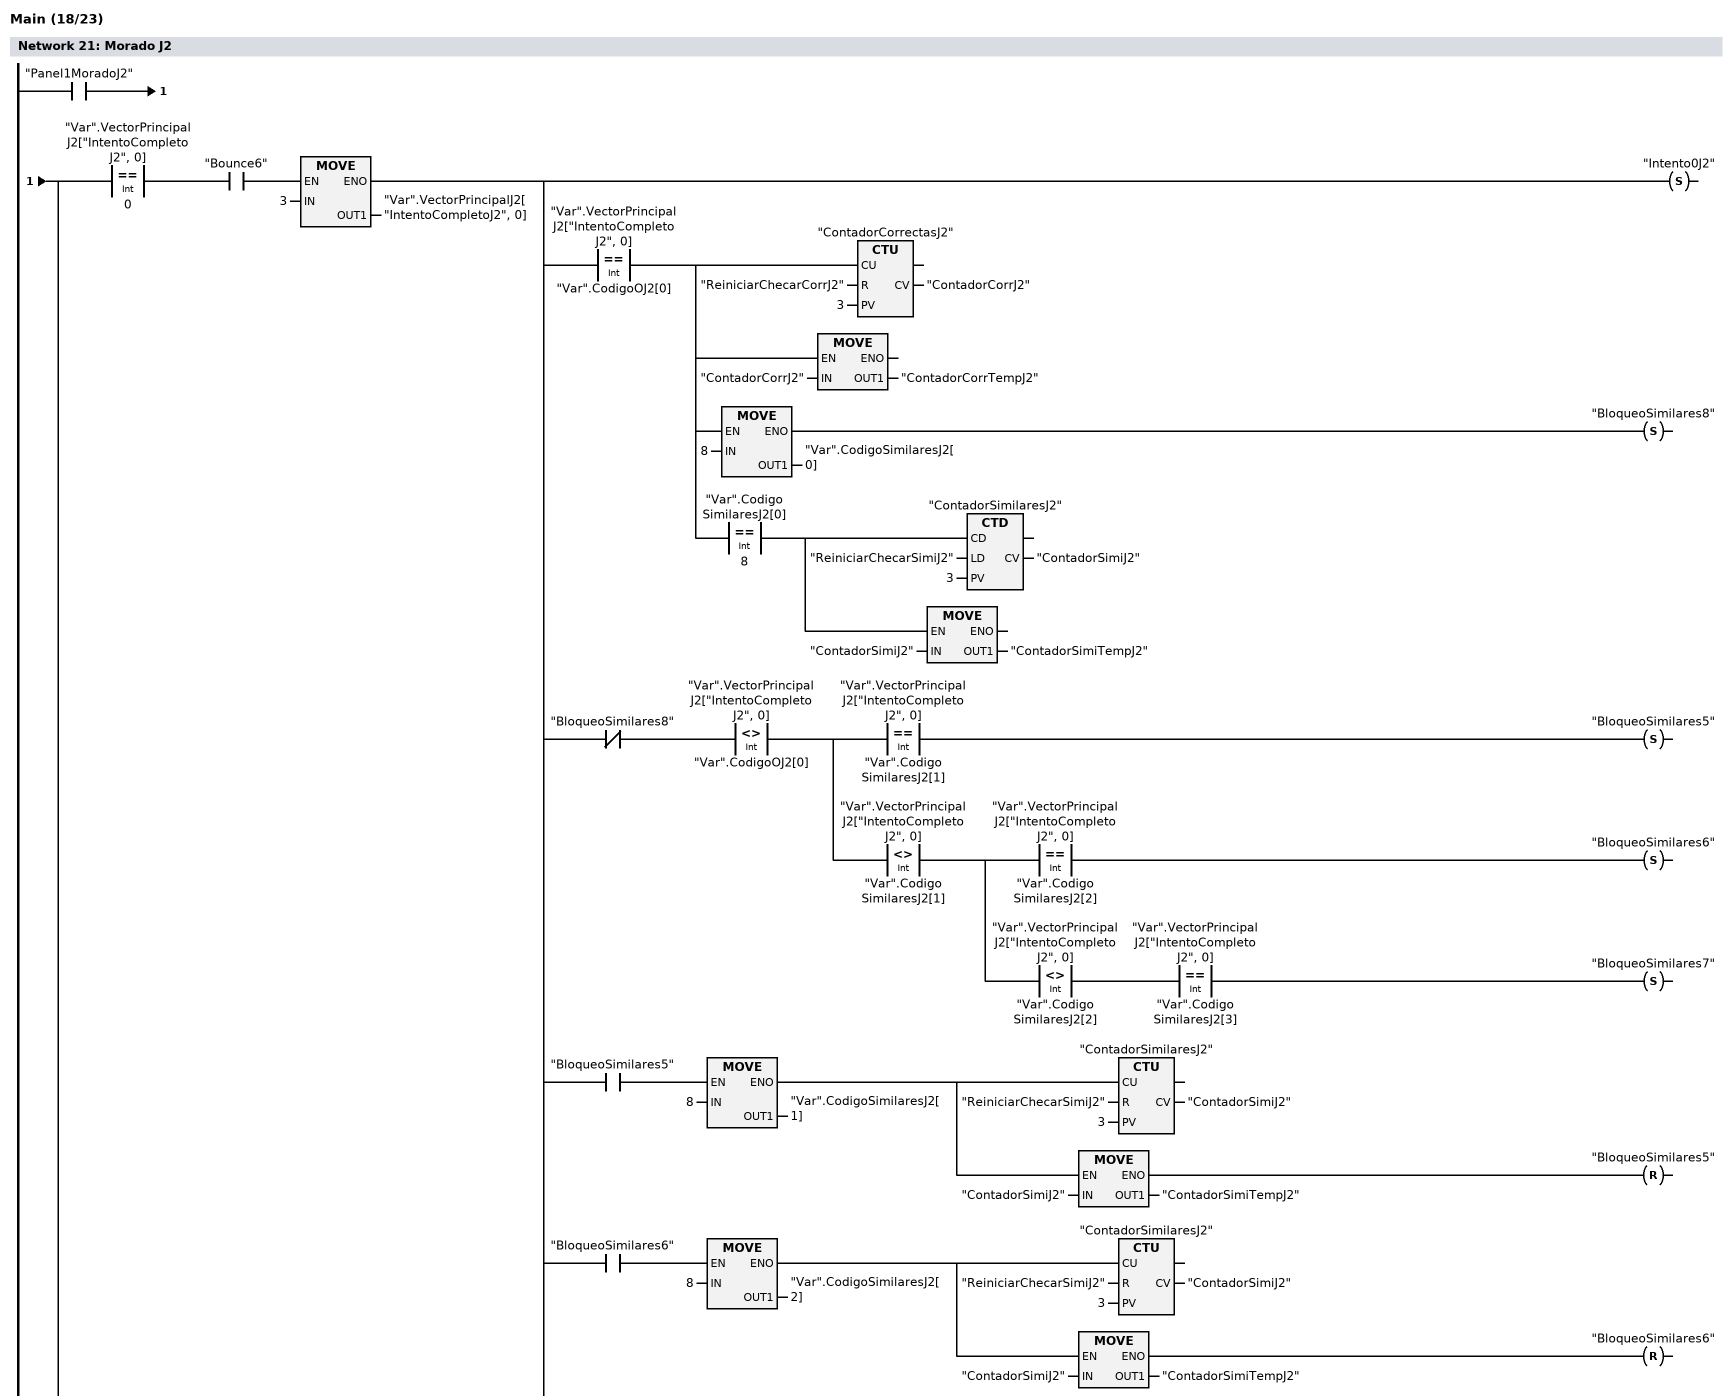
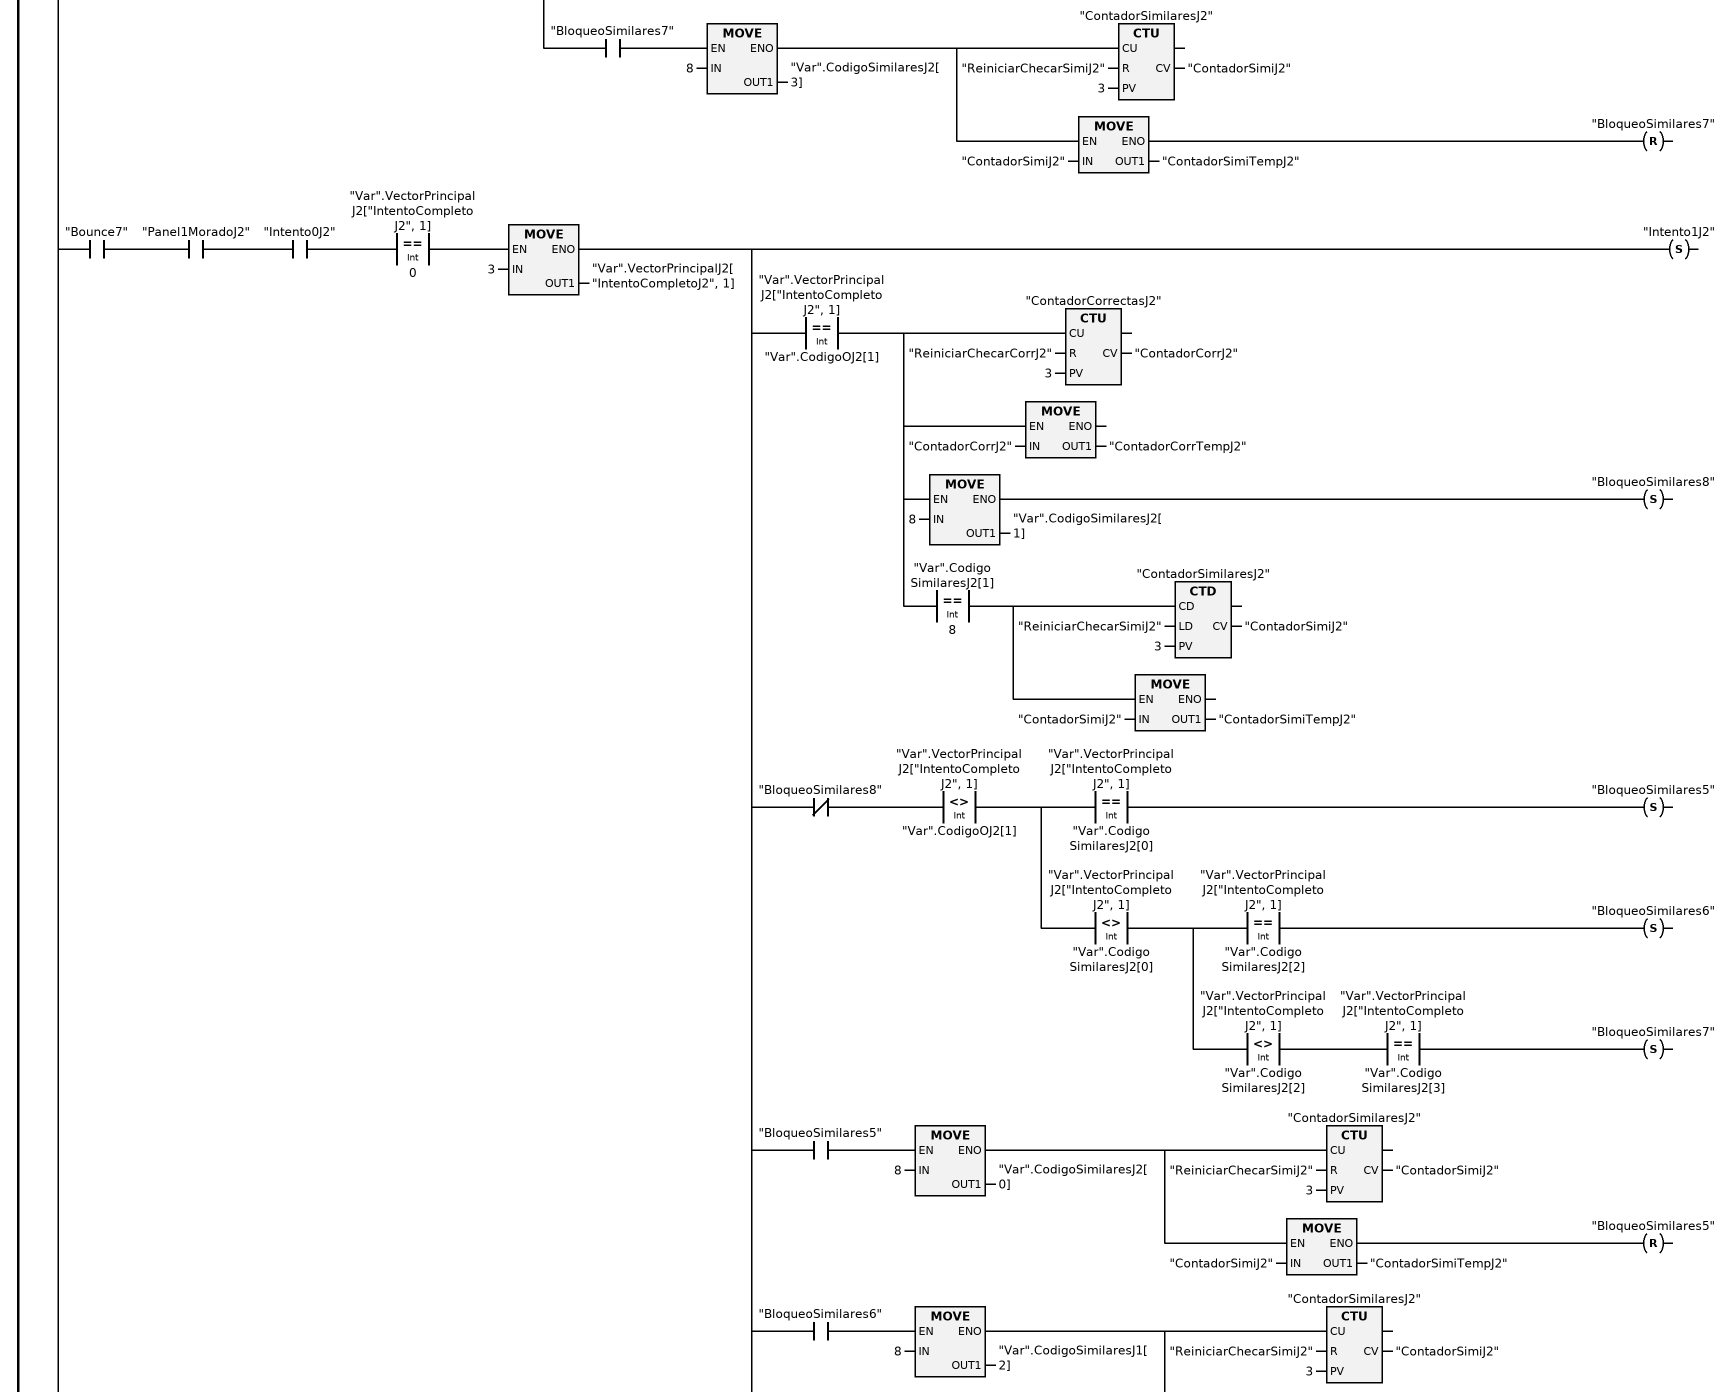
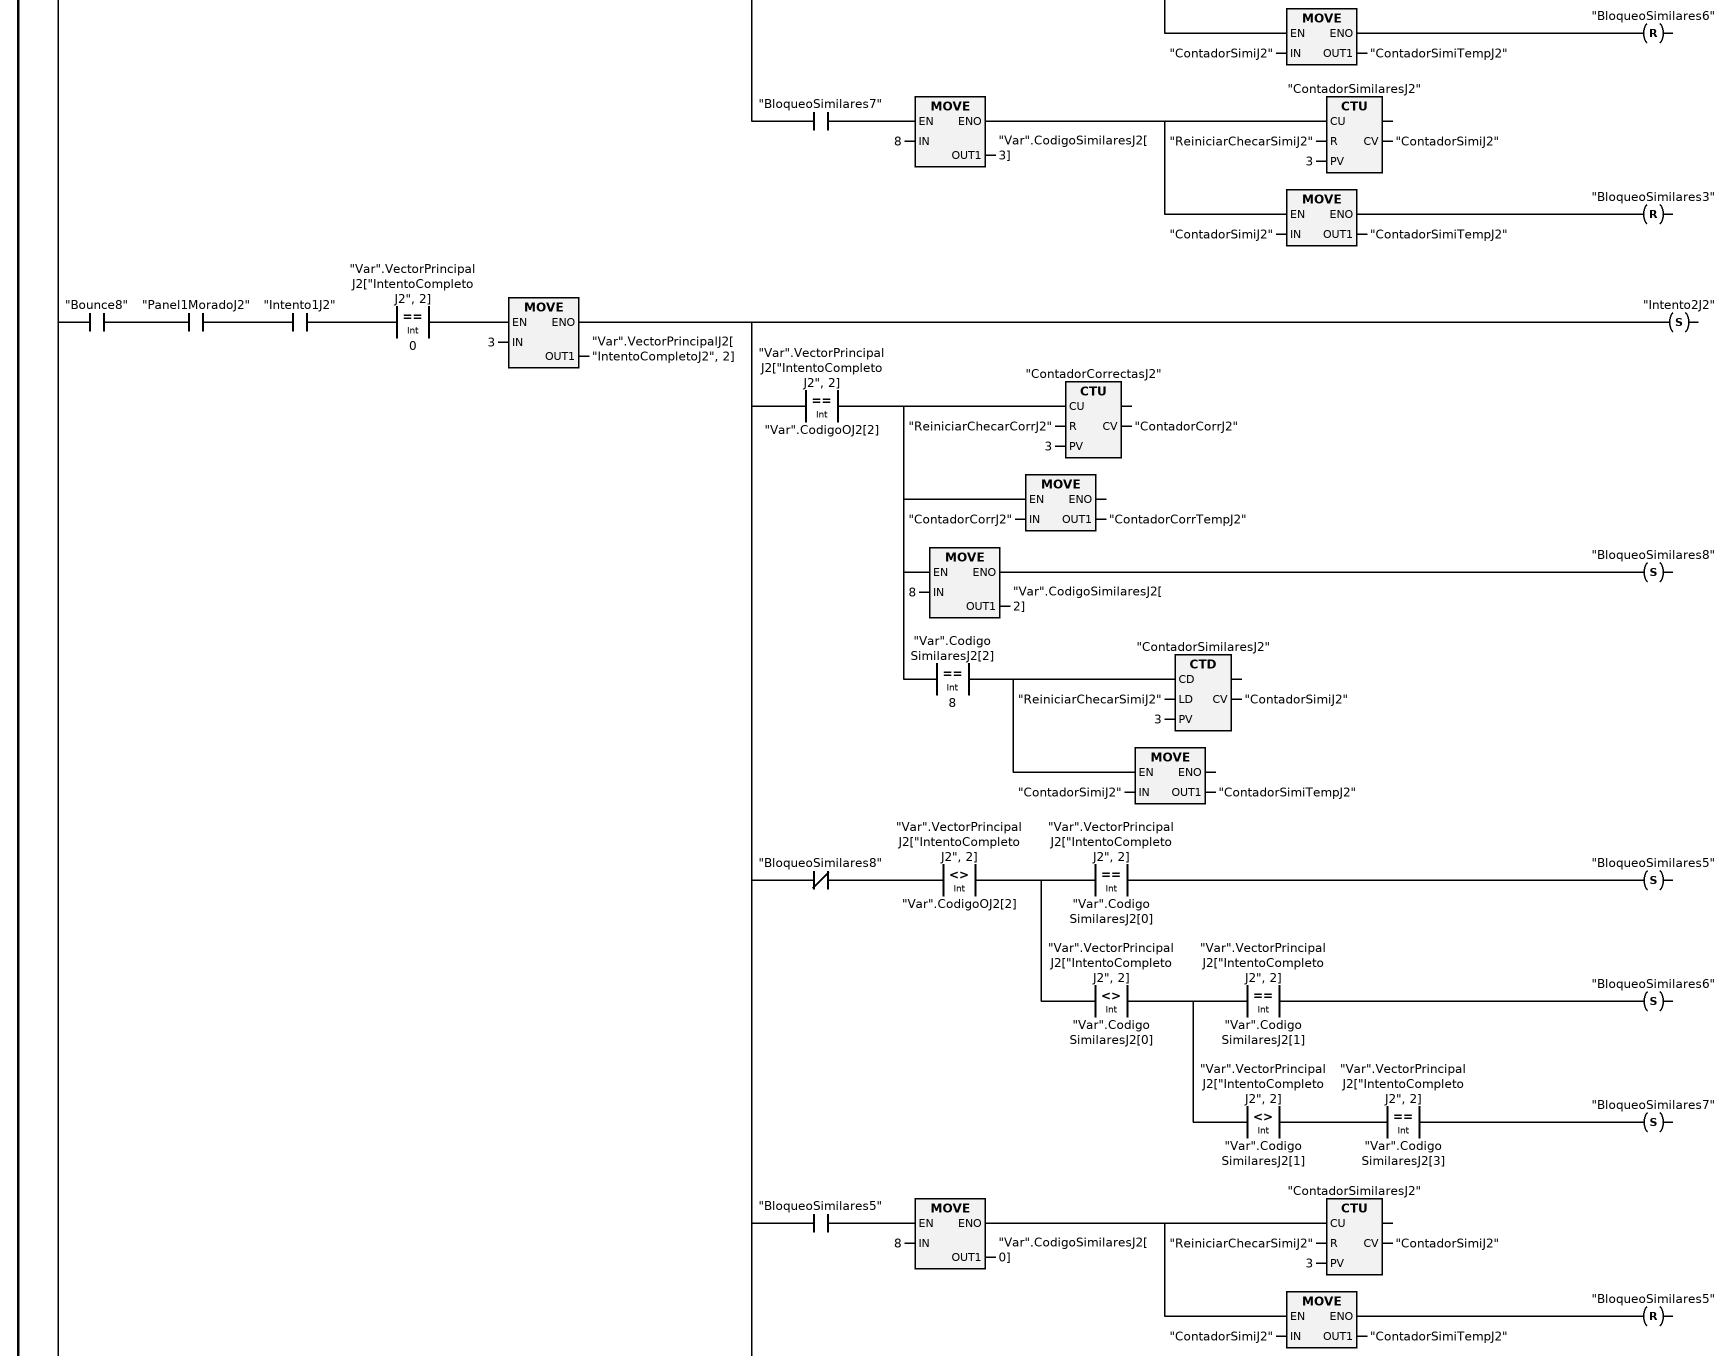
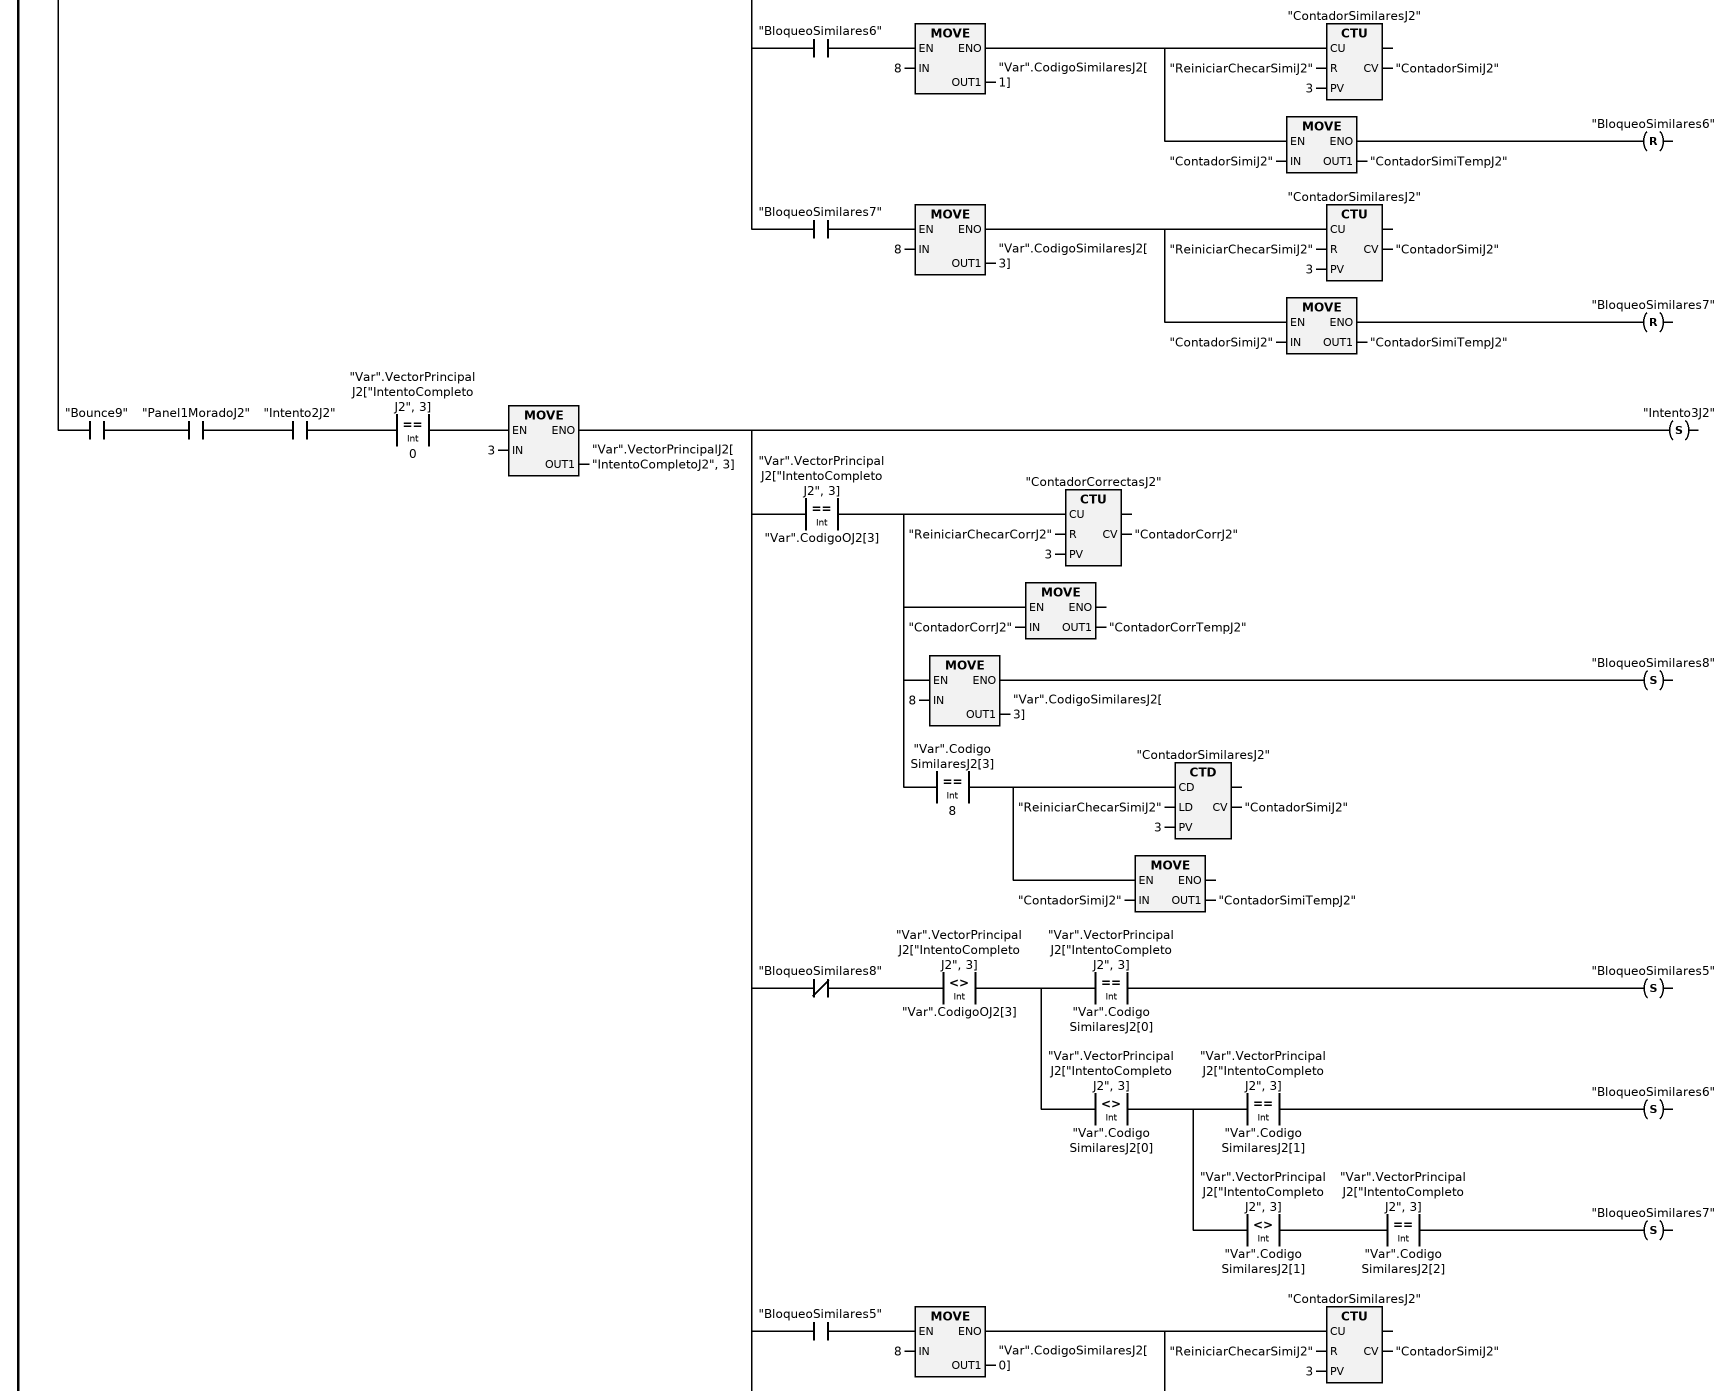
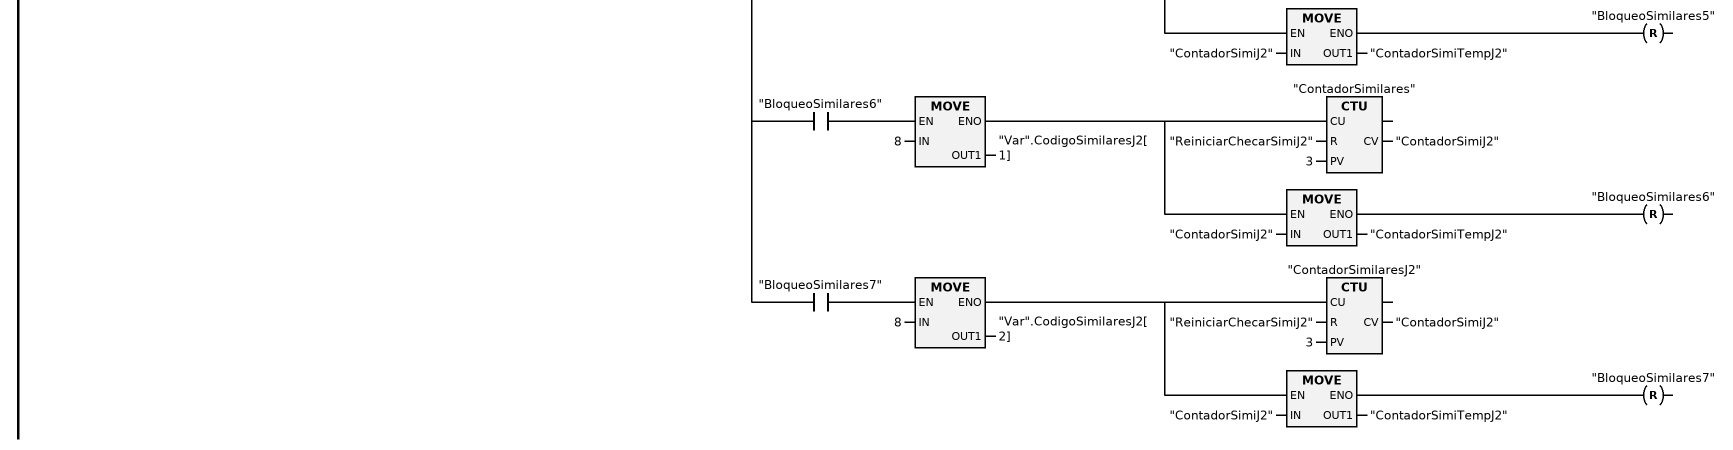
   #_w1 := "Panel1MoradoJ2" AND ("Var".VectorPrincipalJ2["IntentoCompletoJ2", 0] = 0) AND "Bounce6";
   IF #_w1 THEN
       "Var".VectorPrincipalJ2["IntentoCompletoJ2", 0] := 3;
       "Intento0J2" := TRUE;
   END_IF;
   #_w2 := #_w1 AND ("Var".VectorPrincipalJ2["IntentoCompletoJ2", 0] = "Var".CodigoOJ2[0]);
   "ContadorCorrectasJ2".CTU(CU := #_w2, R := "ReiniciarChecarCorrJ2", PV := 3, CV => "ContadorCorrJ2");
   IF #_w2 THEN
       "ContadorCorrTempJ2" := "ContadorCorrJ2";
       "Var".CodigoSimilaresJ2[0] := 8;
       "BloqueoSimilares8" := TRUE;
   END_IF;
   #_w3 := #_w2 AND ("Var".CodigoSimilaresJ2[0] = 8);
   "ContadorSimilaresJ2".CTD(CD := #_w3, LD := "ReiniciarChecarSimiJ2", PV := 3, CV => "ContadorSimiJ2");
   IF #_w3 THEN "ContadorSimiTempJ2" := "ContadorSimiJ2"; END_IF;
   #_w4 := #_w1 AND NOT "BloqueoSimilares8" AND ("Var".VectorPrincipalJ2["IntentoCompletoJ2", 0] <> "Var".CodigoOJ2[0]);
   IF #_w4 AND ("Var".VectorPrincipalJ2["IntentoCompletoJ2", 0] = "Var".CodigoSimilaresJ2[1]) THEN
       "BloqueoSimilares5" := TRUE;
   END_IF;
   #_w5 := #_w4 AND ("Var".VectorPrincipalJ2["IntentoCompletoJ2", 0] <> "Var".CodigoSimilaresJ2[1]);
   IF #_w5 AND ("Var".VectorPrincipalJ2["IntentoCompletoJ2", 0] = "Var".CodigoSimilaresJ2[2]) THEN
       "BloqueoSimilares6" := TRUE;
   END_IF;
   IF #_w5 AND ("Var".VectorPrincipalJ2["IntentoCompletoJ2", 0] <> "Var".CodigoSimilaresJ2[2]) AND ("Var".VectorPrincipalJ2["IntentoCompletoJ2", 0] = "Var".CodigoSimilaresJ2[3]) THEN
       "BloqueoSimilares7" := TRUE;
   END_IF;
   #_w6 := #_w1 AND "BloqueoSimilares5";
   IF #_w6 THEN "Var".CodigoSimilaresJ2[1] := 8; END_IF;
   "ContadorSimilaresJ2".CTU(CU := #_w6, R := "ReiniciarChecarSimiJ2", PV := 3, CV => "ContadorSimiJ2");
   IF #_w6 THEN
       "ContadorSimiTempJ2" := "ContadorSimiJ2";
       "BloqueoSimilares5" := FALSE;
   END_IF;
   #_w7 := #_w1 AND "BloqueoSimilares6";
   IF #_w7 THEN "Var".CodigoSimilaresJ2[2] := 8; END_IF;
   "ContadorSimilaresJ2".CTU(CU := #_w7, R := "ReiniciarChecarSimiJ2", PV := 3, CV => "ContadorSimiJ2");
   IF #_w7 THEN
       "ContadorSimiTempJ2" := "ContadorSimiJ2";
       "BloqueoSimilares6" := FALSE;
   END_IF;
   #_w8 := #_w1 AND "BloqueoSimilares7";
   IF #_w8 THEN "Var".CodigoSimilaresJ2[3] := 8; END_IF;
   "ContadorSimilaresJ2".CTU(CU := #_w8, R := "ReiniciarChecarSimiJ2", PV := 3, CV => "ContadorSimiJ2");
   IF #_w8 THEN
       "ContadorSimiTempJ2" := "ContadorSimiJ2";
       "BloqueoSimilares7" := FALSE;
   END_IF;
   #_w9 := "Panel1MoradoJ2" AND "Bounce7" AND "Panel1MoradoJ2" AND "Intento0J2" AND ("Var".VectorPrincipalJ2["IntentoCompletoJ2", 1] = 0);
   IF #_w9 THEN
       "Var".VectorPrincipalJ2["IntentoCompletoJ2", 1] := 3;
       "Intento1J2" := TRUE;
   END_IF;
   #_w10 := #_w9 AND ("Var".VectorPrincipalJ2["IntentoCompletoJ2", 1] = "Var".CodigoOJ2[1]);
   "ContadorCorrectasJ2".CTU(CU := #_w10, R := "ReiniciarChecarCorrJ2", PV := 3, CV => "ContadorCorrJ2");
   IF #_w10 THEN
       "ContadorCorrTempJ2" := "ContadorCorrJ2";
       "Var".CodigoSimilaresJ2[1] := 8;
       "BloqueoSimilares8" := TRUE;
   END_IF;
   #_w11 := #_w10 AND ("Var".CodigoSimilaresJ2[1] = 8);
   "ContadorSimilaresJ2".CTD(CD := #_w11, LD := "ReiniciarChecarSimiJ2", PV := 3, CV => "ContadorSimiJ2");
   IF #_w11 THEN "ContadorSimiTempJ2" := "ContadorSimiJ2"; END_IF;
   #_w12 := #_w9 AND NOT "BloqueoSimilares8" AND ("Var".VectorPrincipalJ2["IntentoCompletoJ2", 1] <> "Var".CodigoOJ2[1]);
   IF #_w12 AND ("Var".VectorPrincipalJ2["IntentoCompletoJ2", 1] = "Var".CodigoSimilaresJ2[0]) THEN
       "BloqueoSimilares5" := TRUE;
   END_IF;
   #_w13 := #_w12 AND ("Var".VectorPrincipalJ2["IntentoCompletoJ2", 1] <> "Var".CodigoSimilaresJ2[0]);
   IF #_w13 AND ("Var".VectorPrincipalJ2["IntentoCompletoJ2", 1] = "Var".CodigoSimilaresJ2[2]) THEN
       "BloqueoSimilares6" := TRUE;
   END_IF;
   IF #_w13 AND ("Var".VectorPrincipalJ2["IntentoCompletoJ2", 1] <> "Var".CodigoSimilaresJ2[2]) AND ("Var".VectorPrincipalJ2["IntentoCompletoJ2", 1] = "Var".CodigoSimilaresJ2[3]) THEN
       "BloqueoSimilares7" := TRUE;
   END_IF;
   #_w14 := #_w9 AND "BloqueoSimilares5";
   IF #_w14 THEN "Var".CodigoSimilaresJ2[0] := 8; END_IF;
   "ContadorSimilaresJ2".CTU(CU := #_w14, R := "ReiniciarChecarSimiJ2", PV := 3, CV => "ContadorSimiJ2");
   IF #_w14 THEN
       "ContadorSimiTempJ2" := "ContadorSimiJ2";
       "BloqueoSimilares5" := FALSE;
   END_IF;
   #_w15 := #_w9 AND "BloqueoSimilares6";
   IF #_w15 THEN "Var".CodigoSimilaresJ1[2] := 8; END_IF;
   "ContadorSimilaresJ2".CTU(CU := #_w15, R := "ReiniciarChecarSimiJ2", PV := 3, CV => "ContadorSimiJ2");
   IF #_w15 THEN
       "ContadorSimiTempJ2" := "ContadorSimiJ2";
       "BloqueoSimilares6" := FALSE;
   END_IF;
   #_w16 := #_w9 AND "BloqueoSimilares7";
   IF #_w16 THEN "Var".CodigoSimilaresJ2[3] := 8; END_IF;
   "ContadorSimilaresJ2".CTU(CU := #_w16, R := "ReiniciarChecarSimiJ2", PV := 3, CV => "ContadorSimiJ2");
   IF #_w16 THEN
       "ContadorSimiTempJ2" := "ContadorSimiJ2";
       "BloqueoSimilares3" := FALSE;
   END_IF;
   #_w17 := "Panel1MoradoJ2" AND "Bounce8" AND "Panel1MoradoJ2" AND "Intento1J2" AND ("Var".VectorPrincipalJ2["IntentoCompletoJ2", 2] = 0);
   IF #_w17 THEN
       "Var".VectorPrincipalJ2["IntentoCompletoJ2", 2] := 3;
       "Intento2J2" := TRUE;
   END_IF;
   #_w18 := #_w17 AND ("Var".VectorPrincipalJ2["IntentoCompletoJ2", 2] = "Var".CodigoOJ2[2]);
   "ContadorCorrectasJ2".CTU(CU := #_w18, R := "ReiniciarChecarCorrJ2", PV := 3, CV => "ContadorCorrJ2");
   IF #_w18 THEN
       "ContadorCorrTempJ2" := "ContadorCorrJ2";
       "Var".CodigoSimilaresJ2[2] := 8;
       "BloqueoSimilares8" := TRUE;
   END_IF;
   #_w19 := #_w18 AND ("Var".CodigoSimilaresJ2[2] = 8);
   "ContadorSimilaresJ2".CTD(CD := #_w19, LD := "ReiniciarChecarSimiJ2", PV := 3, CV => "ContadorSimiJ2");
   IF #_w19 THEN "ContadorSimiTempJ2" := "ContadorSimiJ2"; END_IF;
   #_w20 := #_w17 AND NOT "BloqueoSimilares8" AND ("Var".VectorPrincipalJ2["IntentoCompletoJ2", 2] <> "Var".CodigoOJ2[2]);
   IF #_w20 AND ("Var".VectorPrincipalJ2["IntentoCompletoJ2", 2] = "Var".CodigoSimilaresJ2[0]) THEN
       "BloqueoSimilares5" := TRUE;
   END_IF;
   #_w21 := #_w20 AND ("Var".VectorPrincipalJ2["IntentoCompletoJ2", 2] <> "Var".CodigoSimilaresJ2[0]);
   IF #_w21 AND ("Var".VectorPrincipalJ2["IntentoCompletoJ2", 2] = "Var".CodigoSimilaresJ2[1]) THEN
       "BloqueoSimilares6" := TRUE;
   END_IF;
   IF #_w21 AND ("Var".VectorPrincipalJ2["IntentoCompletoJ2", 2] <> "Var".CodigoSimilaresJ2[1]) AND ("Var".VectorPrincipalJ2["IntentoCompletoJ2", 2] = "Var".CodigoSimilaresJ2[3]) THEN
       "BloqueoSimilares7" := TRUE;
   END_IF;
   #_w22 := #_w17 AND "BloqueoSimilares5";
   IF #_w22 THEN "Var".CodigoSimilaresJ2[0] := 8; END_IF;
   "ContadorSimilaresJ2".CTU(CU := #_w22, R := "ReiniciarChecarSimiJ2", PV := 3, CV => "ContadorSimiJ2");
   IF #_w22 THEN
       "ContadorSimiTempJ2" := "ContadorSimiJ2";
       "BloqueoSimilares5" := FALSE;
   END_IF;
   #_w23 := #_w17 AND "BloqueoSimilares6";
   IF #_w23 THEN "Var".CodigoSimilaresJ2[1] := 8; END_IF;
   "ContadorSimilaresJ2".CTU(CU := #_w23, R := "ReiniciarChecarSimiJ2", PV := 3, CV => "ContadorSimiJ2");
   IF #_w23 THEN
       "ContadorSimiTempJ2" := "ContadorSimiJ2";
       "BloqueoSimilares6" := FALSE;
   END_IF;
   #_w24 := #_w17 AND "BloqueoSimilares7";
   IF #_w24 THEN "Var".CodigoSimilaresJ2[3] := 8; END_IF;
   "ContadorSimilaresJ2".CTU(CU := #_w24, R := "ReiniciarChecarSimiJ2", PV := 3, CV => "ContadorSimiJ2");
   IF #_w24 THEN
       "ContadorSimiTempJ2" := "ContadorSimiJ2";
       "BloqueoSimilares7" := FALSE;
   END_IF;
   #_w25 := "Panel1MoradoJ2" AND "Bounce9" AND "Panel1MoradoJ2" AND "Intento2J2" AND ("Var".VectorPrincipalJ2["IntentoCompletoJ2", 3] = 0);
   IF #_w25 THEN
       "Var".VectorPrincipalJ2["IntentoCompletoJ2", 3] := 3;
       "Intento3J2" := TRUE;
   END_IF;
   #_w26 := #_w25 AND ("Var".VectorPrincipalJ2["IntentoCompletoJ2", 3] = "Var".CodigoOJ2[3]);
   "ContadorCorrectasJ2".CTU(CU := #_w26, R := "ReiniciarChecarCorrJ2", PV := 3, CV => "ContadorCorrJ2");
   IF #_w26 THEN
       "ContadorCorrTempJ2" := "ContadorCorrJ2";
       "Var".CodigoSimilaresJ2[3] := 8;
       "BloqueoSimilares8" := TRUE;
   END_IF;
   #_w27 := #_w26 AND ("Var".CodigoSimilaresJ2[3] = 8);
   "ContadorSimilaresJ2".CTD(CD := #_w27, LD := "ReiniciarChecarSimiJ2", PV := 3, CV => "ContadorSimiJ2");
   IF #_w27 THEN "ContadorSimiTempJ2" := "ContadorSimiJ2"; END_IF;
   #_w28 := #_w25 AND NOT "BloqueoSimilares8" AND ("Var".VectorPrincipalJ2["IntentoCompletoJ2", 3] <> "Var".CodigoOJ2[3]);
   IF #_w28 AND ("Var".VectorPrincipalJ2["IntentoCompletoJ2", 3] = "Var".CodigoSimilaresJ2[0]) THEN
       "BloqueoSimilares5" := TRUE;
   END_IF;
   #_w29 := #_w28 AND ("Var".VectorPrincipalJ2["IntentoCompletoJ2", 3] <> "Var".CodigoSimilaresJ2[0]);
   IF #_w29 AND ("Var".VectorPrincipalJ2["IntentoCompletoJ2", 3] = "Var".CodigoSimilaresJ2[1]) THEN
       "BloqueoSimilares6" := TRUE;
   END_IF;
   IF #_w29 AND ("Var".VectorPrincipalJ2["IntentoCompletoJ2", 3] <> "Var".CodigoSimilaresJ2[1]) AND ("Var".VectorPrincipalJ2["IntentoCompletoJ2", 3] = "Var".CodigoSimilaresJ2[2]) THEN
       "BloqueoSimilares7" := TRUE;
   END_IF;
   #_w30 := #_w25 AND "BloqueoSimilares5";
   IF #_w30 THEN "Var".CodigoSimilaresJ2[0] := 8; END_IF;
   "ContadorSimilaresJ2".CTU(CU := #_w30, R := "ReiniciarChecarSimiJ2", PV := 3, CV => "ContadorSimiJ2");
   IF #_w30 THEN
       "ContadorSimiTempJ2" := "ContadorSimiJ2";
       "BloqueoSimilares5" := FALSE;
   END_IF;
   #_w31 := #_w25 AND "BloqueoSimilares6";
   IF #_w31 THEN "Var".CodigoSimilaresJ2[1] := 8; END_IF;
   "ContadorSimilares".CTU(CU := #_w31, R := "ReiniciarChecarSimiJ2", PV := 3, CV => "ContadorSimiJ2");
   IF #_w31 THEN
       "ContadorSimiTempJ2" := "ContadorSimiJ2";
       "BloqueoSimilares6" := FALSE;
   END_IF;
   #_w32 := #_w25 AND "BloqueoSimilares7";
   IF #_w32 THEN "Var".CodigoSimilaresJ2[2] := 8; END_IF;
   "ContadorSimilaresJ2".CTU(CU := #_w32, R := "ReiniciarChecarSimiJ2", PV := 3, CV => "ContadorSimiJ2");
   IF #_w32 THEN
       "ContadorSimiTempJ2" := "ContadorSimiJ2";
       "BloqueoSimilares7" := FALSE;
   END_IF;
END_REGION

REGION Network 22: Rojo J2
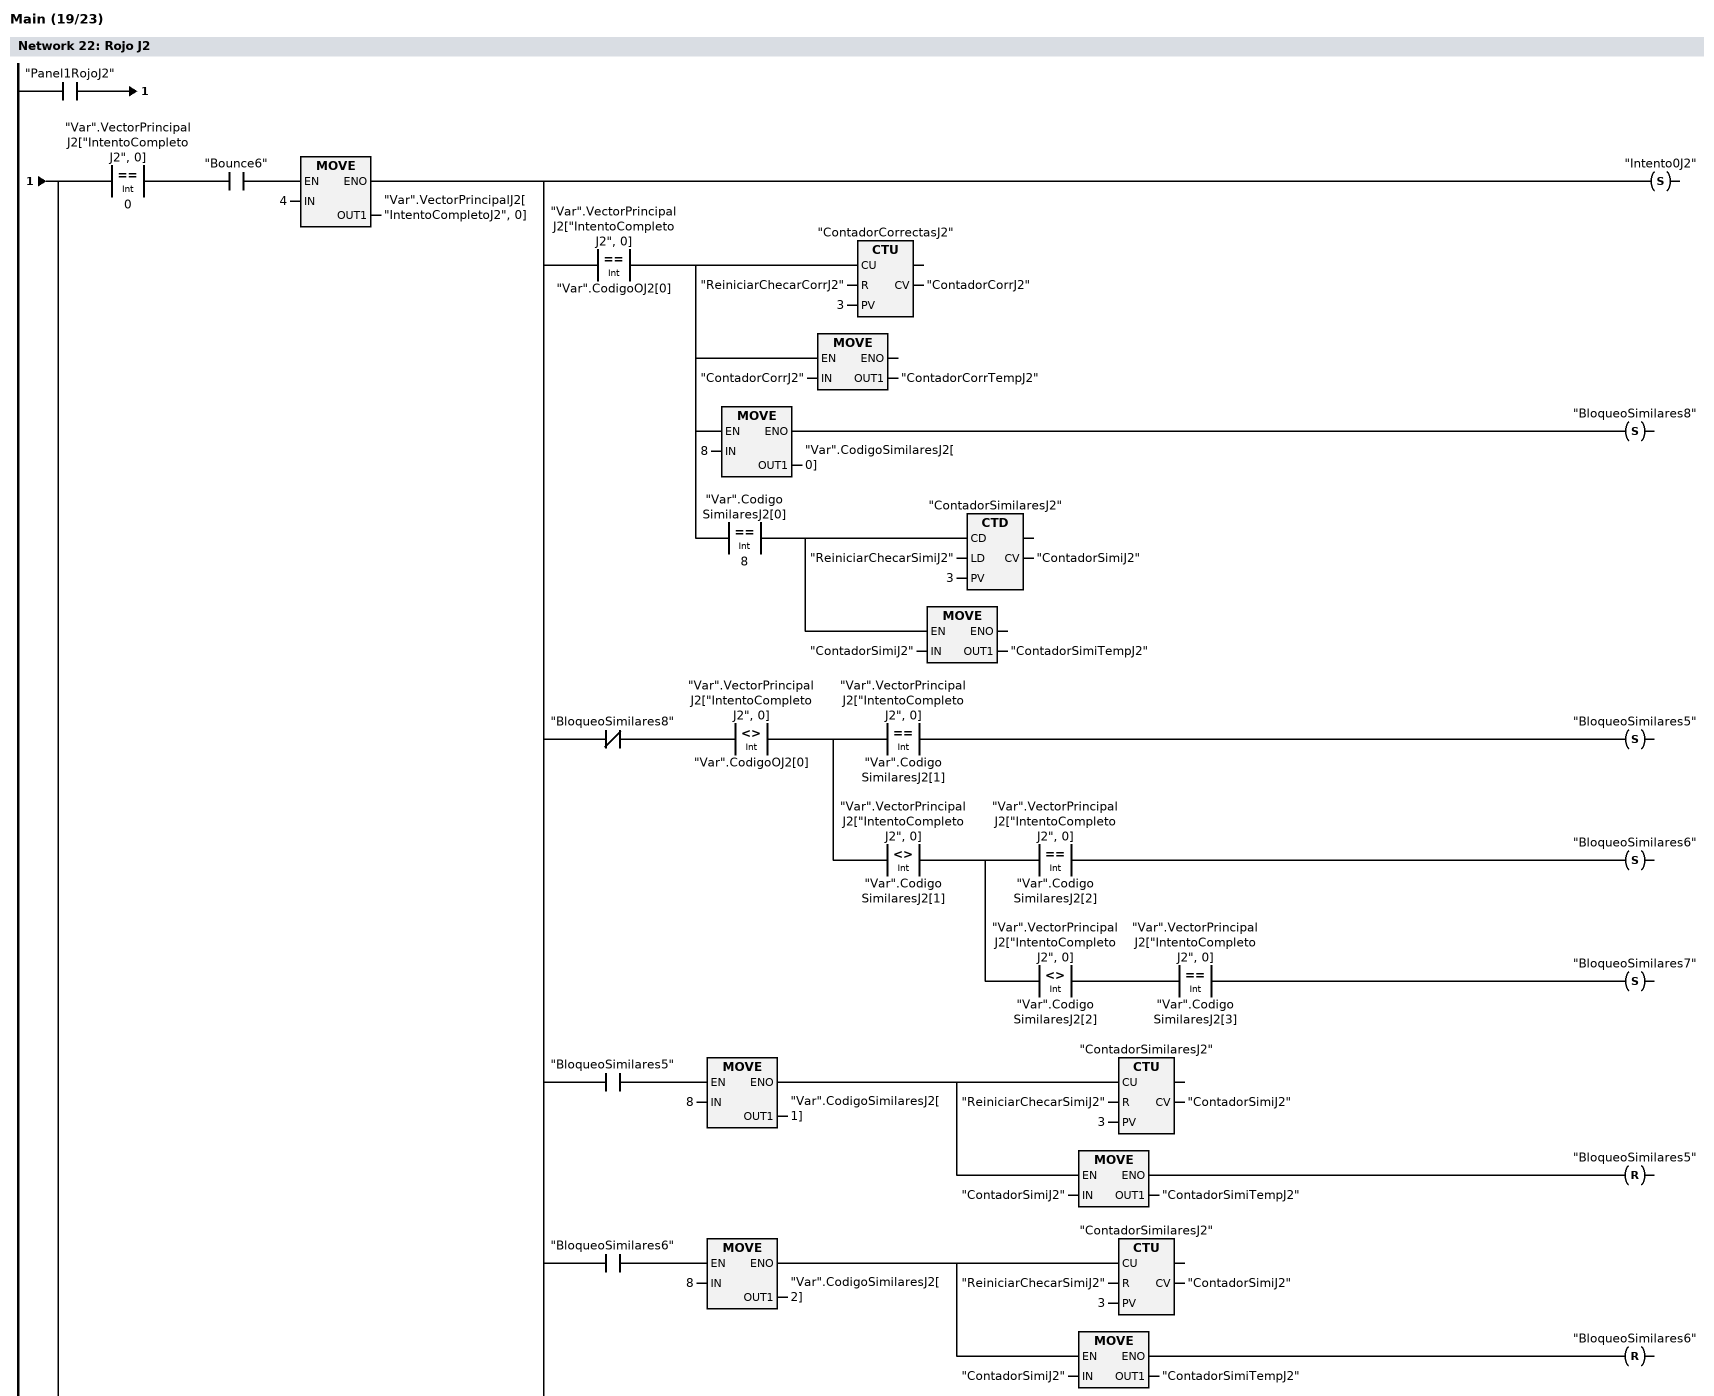
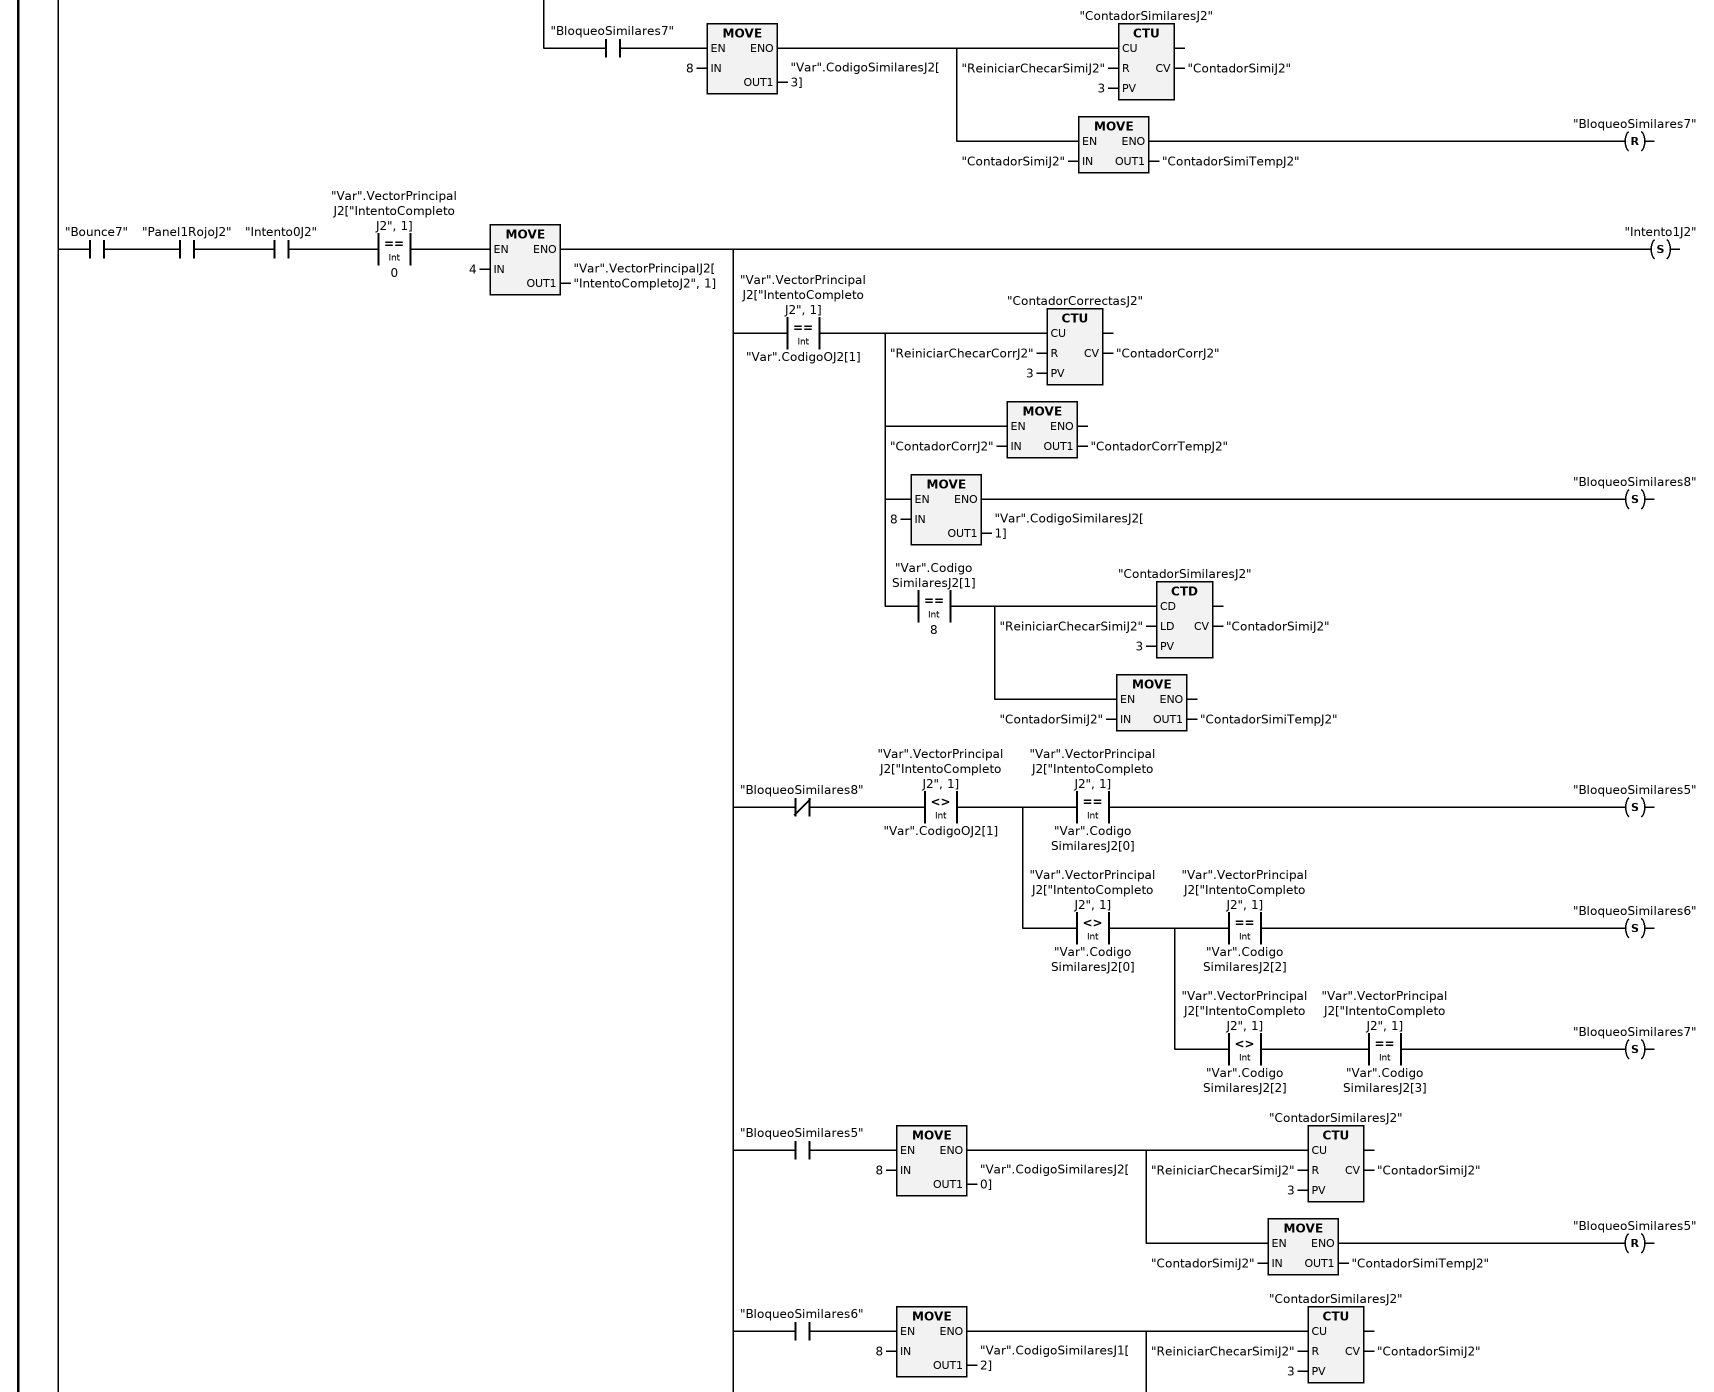
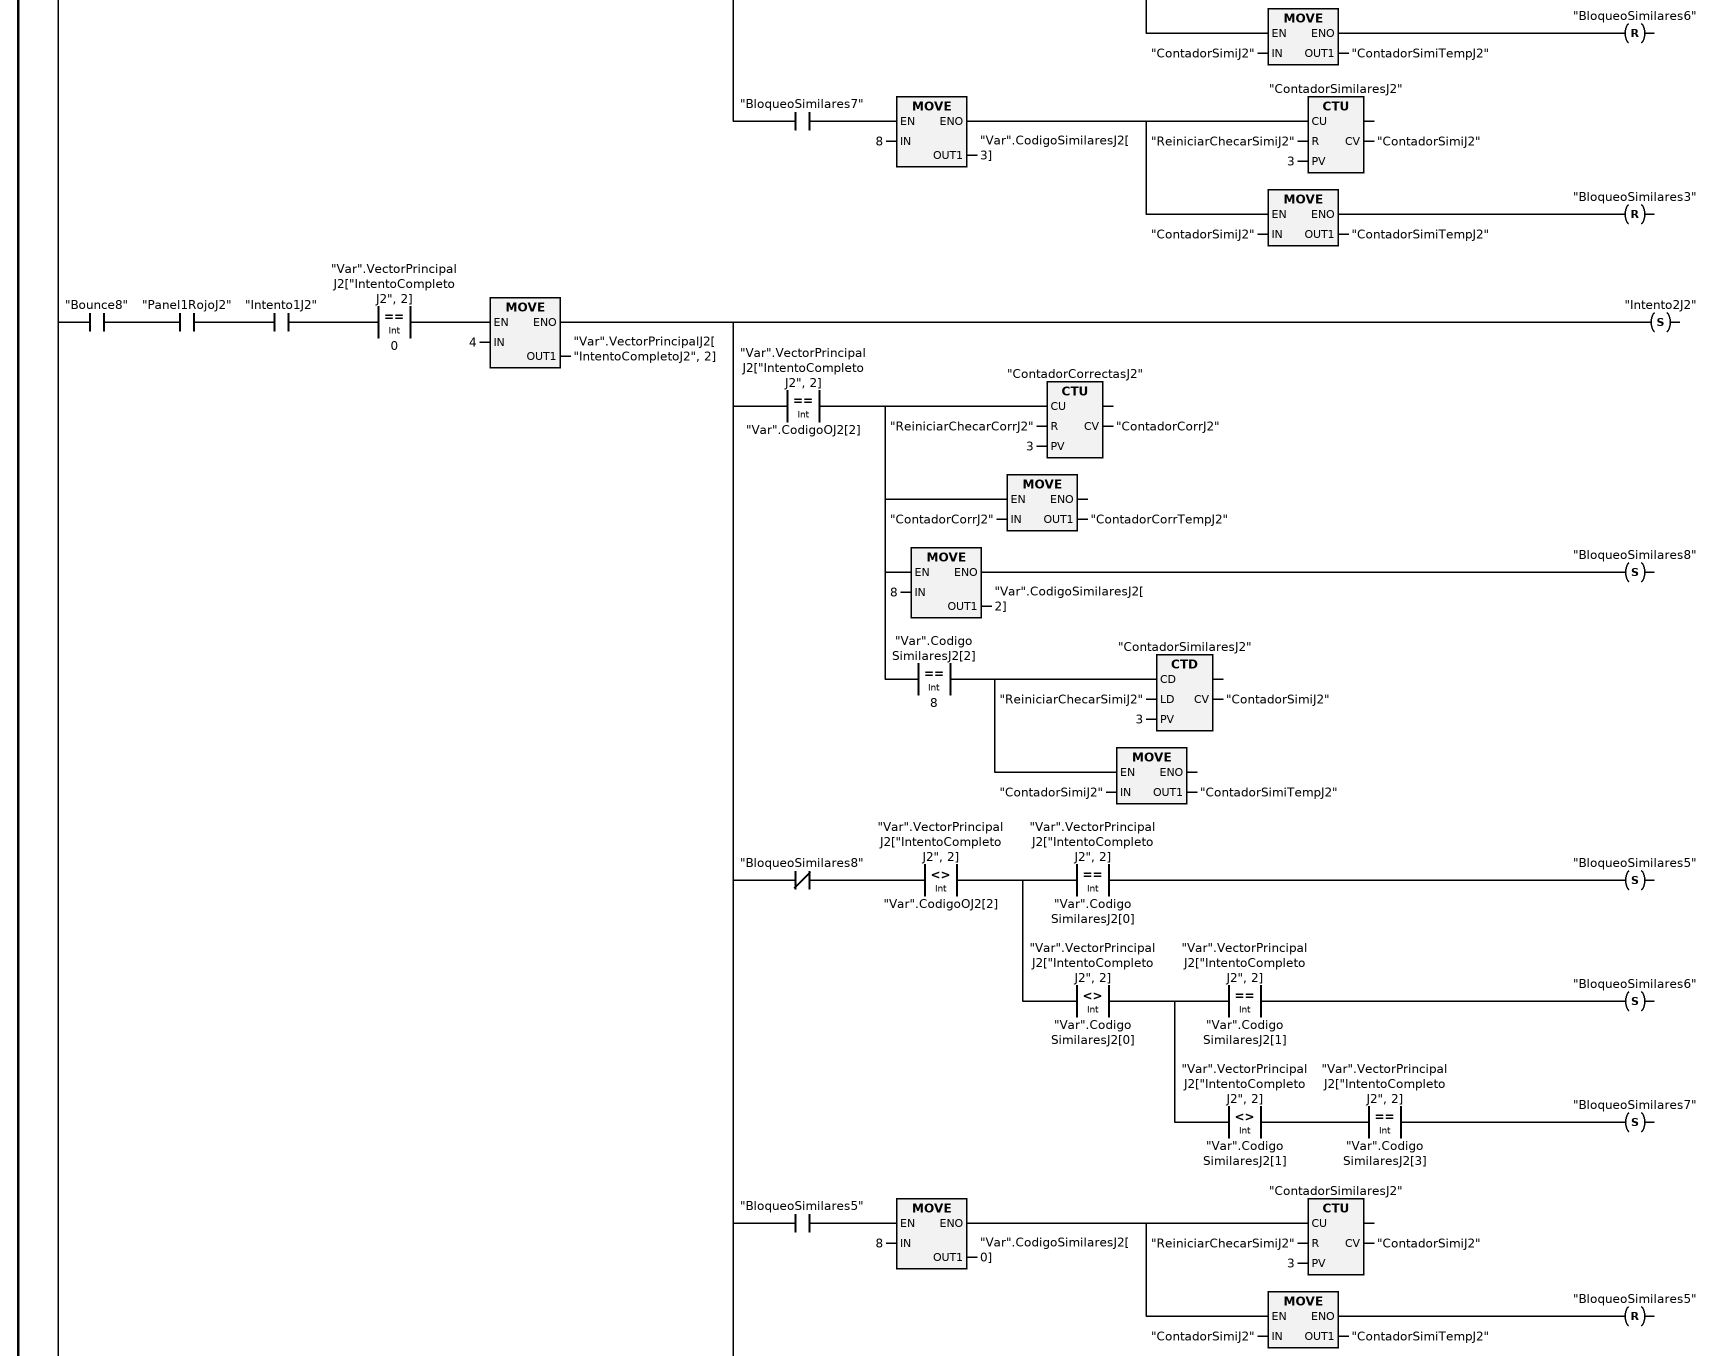
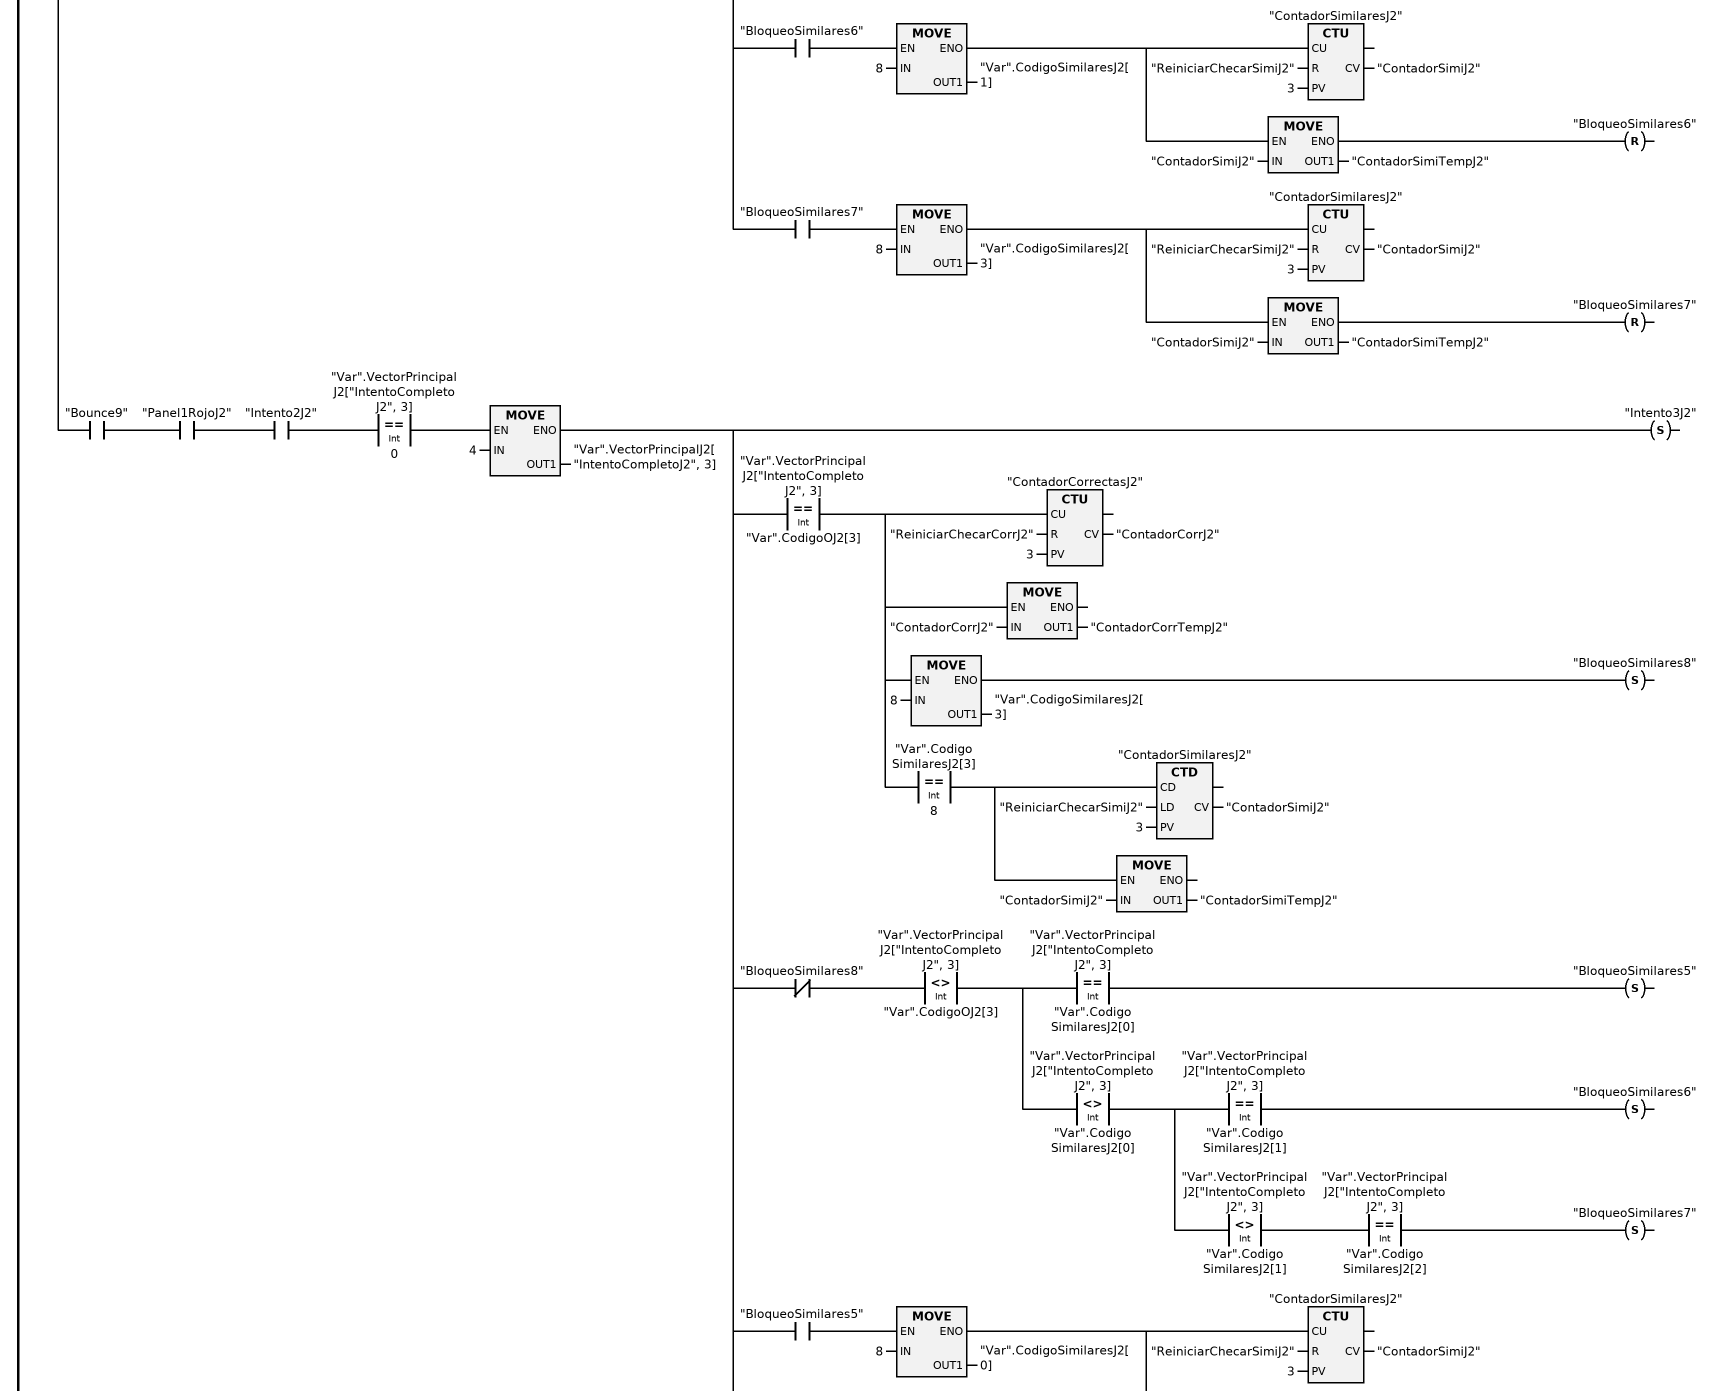
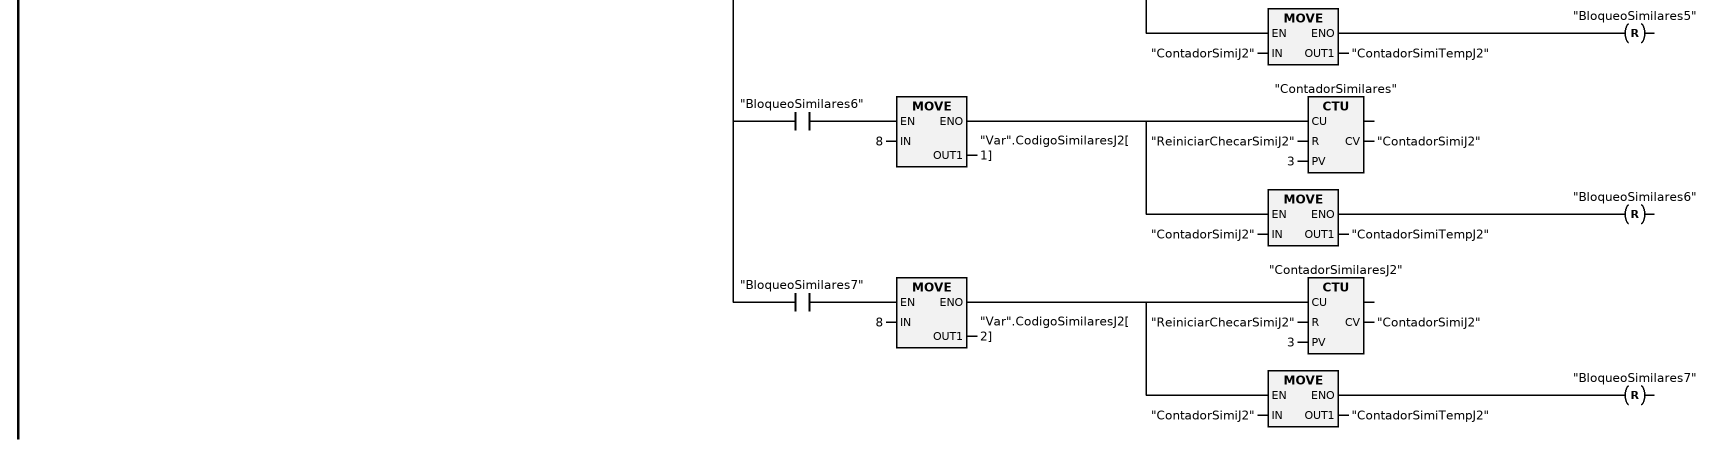
   #_w1 := "Panel1RojoJ2" AND ("Var".VectorPrincipalJ2["IntentoCompletoJ2", 0] = 0) AND "Bounce6";
   IF #_w1 THEN
       "Var".VectorPrincipalJ2["IntentoCompletoJ2", 0] := 4;
       "Intento0J2" := TRUE;
   END_IF;
   #_w2 := #_w1 AND ("Var".VectorPrincipalJ2["IntentoCompletoJ2", 0] = "Var".CodigoOJ2[0]);
   "ContadorCorrectasJ2".CTU(CU := #_w2, R := "ReiniciarChecarCorrJ2", PV := 3, CV => "ContadorCorrJ2");
   IF #_w2 THEN
       "ContadorCorrTempJ2" := "ContadorCorrJ2";
       "Var".CodigoSimilaresJ2[0] := 8;
       "BloqueoSimilares8" := TRUE;
   END_IF;
   #_w3 := #_w2 AND ("Var".CodigoSimilaresJ2[0] = 8);
   "ContadorSimilaresJ2".CTD(CD := #_w3, LD := "ReiniciarChecarSimiJ2", PV := 3, CV => "ContadorSimiJ2");
   IF #_w3 THEN "ContadorSimiTempJ2" := "ContadorSimiJ2"; END_IF;
   #_w4 := #_w1 AND NOT "BloqueoSimilares8" AND ("Var".VectorPrincipalJ2["IntentoCompletoJ2", 0] <> "Var".CodigoOJ2[0]);
   IF #_w4 AND ("Var".VectorPrincipalJ2["IntentoCompletoJ2", 0] = "Var".CodigoSimilaresJ2[1]) THEN
       "BloqueoSimilares5" := TRUE;
   END_IF;
   #_w5 := #_w4 AND ("Var".VectorPrincipalJ2["IntentoCompletoJ2", 0] <> "Var".CodigoSimilaresJ2[1]);
   IF #_w5 AND ("Var".VectorPrincipalJ2["IntentoCompletoJ2", 0] = "Var".CodigoSimilaresJ2[2]) THEN
       "BloqueoSimilares6" := TRUE;
   END_IF;
   IF #_w5 AND ("Var".VectorPrincipalJ2["IntentoCompletoJ2", 0] <> "Var".CodigoSimilaresJ2[2]) AND ("Var".VectorPrincipalJ2["IntentoCompletoJ2", 0] = "Var".CodigoSimilaresJ2[3]) THEN
       "BloqueoSimilares7" := TRUE;
   END_IF;
   #_w6 := #_w1 AND "BloqueoSimilares5";
   IF #_w6 THEN "Var".CodigoSimilaresJ2[1] := 8; END_IF;
   "ContadorSimilaresJ2".CTU(CU := #_w6, R := "ReiniciarChecarSimiJ2", PV := 3, CV => "ContadorSimiJ2");
   IF #_w6 THEN
       "ContadorSimiTempJ2" := "ContadorSimiJ2";
       "BloqueoSimilares5" := FALSE;
   END_IF;
   #_w7 := #_w1 AND "BloqueoSimilares6";
   IF #_w7 THEN "Var".CodigoSimilaresJ2[2] := 8; END_IF;
   "ContadorSimilaresJ2".CTU(CU := #_w7, R := "ReiniciarChecarSimiJ2", PV := 3, CV => "ContadorSimiJ2");
   IF #_w7 THEN
       "ContadorSimiTempJ2" := "ContadorSimiJ2";
       "BloqueoSimilares6" := FALSE;
   END_IF;
   #_w8 := #_w1 AND "BloqueoSimilares7";
   IF #_w8 THEN "Var".CodigoSimilaresJ2[3] := 8; END_IF;
   "ContadorSimilaresJ2".CTU(CU := #_w8, R := "ReiniciarChecarSimiJ2", PV := 3, CV => "ContadorSimiJ2");
   IF #_w8 THEN
       "ContadorSimiTempJ2" := "ContadorSimiJ2";
       "BloqueoSimilares7" := FALSE;
   END_IF;
   #_w9 := "Panel1RojoJ2" AND "Bounce7" AND "Panel1RojoJ2" AND "Intento0J2" AND ("Var".VectorPrincipalJ2["IntentoCompletoJ2", 1] = 0);
   IF #_w9 THEN
       "Var".VectorPrincipalJ2["IntentoCompletoJ2", 1] := 4;
       "Intento1J2" := TRUE;
   END_IF;
   #_w10 := #_w9 AND ("Var".VectorPrincipalJ2["IntentoCompletoJ2", 1] = "Var".CodigoOJ2[1]);
   "ContadorCorrectasJ2".CTU(CU := #_w10, R := "ReiniciarChecarCorrJ2", PV := 3, CV => "ContadorCorrJ2");
   IF #_w10 THEN
       "ContadorCorrTempJ2" := "ContadorCorrJ2";
       "Var".CodigoSimilaresJ2[1] := 8;
       "BloqueoSimilares8" := TRUE;
   END_IF;
   #_w11 := #_w10 AND ("Var".CodigoSimilaresJ2[1] = 8);
   "ContadorSimilaresJ2".CTD(CD := #_w11, LD := "ReiniciarChecarSimiJ2", PV := 3, CV => "ContadorSimiJ2");
   IF #_w11 THEN "ContadorSimiTempJ2" := "ContadorSimiJ2"; END_IF;
   #_w12 := #_w9 AND NOT "BloqueoSimilares8" AND ("Var".VectorPrincipalJ2["IntentoCompletoJ2", 1] <> "Var".CodigoOJ2[1]);
   IF #_w12 AND ("Var".VectorPrincipalJ2["IntentoCompletoJ2", 1] = "Var".CodigoSimilaresJ2[0]) THEN
       "BloqueoSimilares5" := TRUE;
   END_IF;
   #_w13 := #_w12 AND ("Var".VectorPrincipalJ2["IntentoCompletoJ2", 1] <> "Var".CodigoSimilaresJ2[0]);
   IF #_w13 AND ("Var".VectorPrincipalJ2["IntentoCompletoJ2", 1] = "Var".CodigoSimilaresJ2[2]) THEN
       "BloqueoSimilares6" := TRUE;
   END_IF;
   IF #_w13 AND ("Var".VectorPrincipalJ2["IntentoCompletoJ2", 1] <> "Var".CodigoSimilaresJ2[2]) AND ("Var".VectorPrincipalJ2["IntentoCompletoJ2", 1] = "Var".CodigoSimilaresJ2[3]) THEN
       "BloqueoSimilares7" := TRUE;
   END_IF;
   #_w14 := #_w9 AND "BloqueoSimilares5";
   IF #_w14 THEN "Var".CodigoSimilaresJ2[0] := 8; END_IF;
   "ContadorSimilaresJ2".CTU(CU := #_w14, R := "ReiniciarChecarSimiJ2", PV := 3, CV => "ContadorSimiJ2");
   IF #_w14 THEN
       "ContadorSimiTempJ2" := "ContadorSimiJ2";
       "BloqueoSimilares5" := FALSE;
   END_IF;
   #_w15 := #_w9 AND "BloqueoSimilares6";
   IF #_w15 THEN "Var".CodigoSimilaresJ1[2] := 8; END_IF;
   "ContadorSimilaresJ2".CTU(CU := #_w15, R := "ReiniciarChecarSimiJ2", PV := 3, CV => "ContadorSimiJ2");
   IF #_w15 THEN
       "ContadorSimiTempJ2" := "ContadorSimiJ2";
       "BloqueoSimilares6" := FALSE;
   END_IF;
   #_w16 := #_w9 AND "BloqueoSimilares7";
   IF #_w16 THEN "Var".CodigoSimilaresJ2[3] := 8; END_IF;
   "ContadorSimilaresJ2".CTU(CU := #_w16, R := "ReiniciarChecarSimiJ2", PV := 3, CV => "ContadorSimiJ2");
   IF #_w16 THEN
       "ContadorSimiTempJ2" := "ContadorSimiJ2";
       "BloqueoSimilares3" := FALSE;
   END_IF;
   #_w17 := "Panel1RojoJ2" AND "Bounce8" AND "Panel1RojoJ2" AND "Intento1J2" AND ("Var".VectorPrincipalJ2["IntentoCompletoJ2", 2] = 0);
   IF #_w17 THEN
       "Var".VectorPrincipalJ2["IntentoCompletoJ2", 2] := 4;
       "Intento2J2" := TRUE;
   END_IF;
   #_w18 := #_w17 AND ("Var".VectorPrincipalJ2["IntentoCompletoJ2", 2] = "Var".CodigoOJ2[2]);
   "ContadorCorrectasJ2".CTU(CU := #_w18, R := "ReiniciarChecarCorrJ2", PV := 3, CV => "ContadorCorrJ2");
   IF #_w18 THEN
       "ContadorCorrTempJ2" := "ContadorCorrJ2";
       "Var".CodigoSimilaresJ2[2] := 8;
       "BloqueoSimilares8" := TRUE;
   END_IF;
   #_w19 := #_w18 AND ("Var".CodigoSimilaresJ2[2] = 8);
   "ContadorSimilaresJ2".CTD(CD := #_w19, LD := "ReiniciarChecarSimiJ2", PV := 3, CV => "ContadorSimiJ2");
   IF #_w19 THEN "ContadorSimiTempJ2" := "ContadorSimiJ2"; END_IF;
   #_w20 := #_w17 AND NOT "BloqueoSimilares8" AND ("Var".VectorPrincipalJ2["IntentoCompletoJ2", 2] <> "Var".CodigoOJ2[2]);
   IF #_w20 AND ("Var".VectorPrincipalJ2["IntentoCompletoJ2", 2] = "Var".CodigoSimilaresJ2[0]) THEN
       "BloqueoSimilares5" := TRUE;
   END_IF;
   #_w21 := #_w20 AND ("Var".VectorPrincipalJ2["IntentoCompletoJ2", 2] <> "Var".CodigoSimilaresJ2[0]);
   IF #_w21 AND ("Var".VectorPrincipalJ2["IntentoCompletoJ2", 2] = "Var".CodigoSimilaresJ2[1]) THEN
       "BloqueoSimilares6" := TRUE;
   END_IF;
   IF #_w21 AND ("Var".VectorPrincipalJ2["IntentoCompletoJ2", 2] <> "Var".CodigoSimilaresJ2[1]) AND ("Var".VectorPrincipalJ2["IntentoCompletoJ2", 2] = "Var".CodigoSimilaresJ2[3]) THEN
       "BloqueoSimilares7" := TRUE;
   END_IF;
   #_w22 := #_w17 AND "BloqueoSimilares5";
   IF #_w22 THEN "Var".CodigoSimilaresJ2[0] := 8; END_IF;
   "ContadorSimilaresJ2".CTU(CU := #_w22, R := "ReiniciarChecarSimiJ2", PV := 3, CV => "ContadorSimiJ2");
   IF #_w22 THEN
       "ContadorSimiTempJ2" := "ContadorSimiJ2";
       "BloqueoSimilares5" := FALSE;
   END_IF;
   #_w23 := #_w17 AND "BloqueoSimilares6";
   IF #_w23 THEN "Var".CodigoSimilaresJ2[1] := 8; END_IF;
   "ContadorSimilaresJ2".CTU(CU := #_w23, R := "ReiniciarChecarSimiJ2", PV := 3, CV => "ContadorSimiJ2");
   IF #_w23 THEN
       "ContadorSimiTempJ2" := "ContadorSimiJ2";
       "BloqueoSimilares6" := FALSE;
   END_IF;
   #_w24 := #_w17 AND "BloqueoSimilares7";
   IF #_w24 THEN "Var".CodigoSimilaresJ2[3] := 8; END_IF;
   "ContadorSimilaresJ2".CTU(CU := #_w24, R := "ReiniciarChecarSimiJ2", PV := 3, CV => "ContadorSimiJ2");
   IF #_w24 THEN
       "ContadorSimiTempJ2" := "ContadorSimiJ2";
       "BloqueoSimilares7" := FALSE;
   END_IF;
   #_w25 := "Panel1RojoJ2" AND "Bounce9" AND "Panel1RojoJ2" AND "Intento2J2" AND ("Var".VectorPrincipalJ2["IntentoCompletoJ2", 3] = 0);
   IF #_w25 THEN
       "Var".VectorPrincipalJ2["IntentoCompletoJ2", 3] := 4;
       "Intento3J2" := TRUE;
   END_IF;
   #_w26 := #_w25 AND ("Var".VectorPrincipalJ2["IntentoCompletoJ2", 3] = "Var".CodigoOJ2[3]);
   "ContadorCorrectasJ2".CTU(CU := #_w26, R := "ReiniciarChecarCorrJ2", PV := 3, CV => "ContadorCorrJ2");
   IF #_w26 THEN
       "ContadorCorrTempJ2" := "ContadorCorrJ2";
       "Var".CodigoSimilaresJ2[3] := 8;
       "BloqueoSimilares8" := TRUE;
   END_IF;
   #_w27 := #_w26 AND ("Var".CodigoSimilaresJ2[3] = 8);
   "ContadorSimilaresJ2".CTD(CD := #_w27, LD := "ReiniciarChecarSimiJ2", PV := 3, CV => "ContadorSimiJ2");
   IF #_w27 THEN "ContadorSimiTempJ2" := "ContadorSimiJ2"; END_IF;
   #_w28 := #_w25 AND NOT "BloqueoSimilares8" AND ("Var".VectorPrincipalJ2["IntentoCompletoJ2", 3] <> "Var".CodigoOJ2[3]);
   IF #_w28 AND ("Var".VectorPrincipalJ2["IntentoCompletoJ2", 3] = "Var".CodigoSimilaresJ2[0]) THEN
       "BloqueoSimilares5" := TRUE;
   END_IF;
   #_w29 := #_w28 AND ("Var".VectorPrincipalJ2["IntentoCompletoJ2", 3] <> "Var".CodigoSimilaresJ2[0]);
   IF #_w29 AND ("Var".VectorPrincipalJ2["IntentoCompletoJ2", 3] = "Var".CodigoSimilaresJ2[1]) THEN
       "BloqueoSimilares6" := TRUE;
   END_IF;
   IF #_w29 AND ("Var".VectorPrincipalJ2["IntentoCompletoJ2", 3] <> "Var".CodigoSimilaresJ2[1]) AND ("Var".VectorPrincipalJ2["IntentoCompletoJ2", 3] = "Var".CodigoSimilaresJ2[2]) THEN
       "BloqueoSimilares7" := TRUE;
   END_IF;
   #_w30 := #_w25 AND "BloqueoSimilares5";
   IF #_w30 THEN "Var".CodigoSimilaresJ2[0] := 8; END_IF;
   "ContadorSimilaresJ2".CTU(CU := #_w30, R := "ReiniciarChecarSimiJ2", PV := 3, CV => "ContadorSimiJ2");
   IF #_w30 THEN
       "ContadorSimiTempJ2" := "ContadorSimiJ2";
       "BloqueoSimilares5" := FALSE;
   END_IF;
   #_w31 := #_w25 AND "BloqueoSimilares6";
   IF #_w31 THEN "Var".CodigoSimilaresJ2[1] := 8; END_IF;
   "ContadorSimilares".CTU(CU := #_w31, R := "ReiniciarChecarSimiJ2", PV := 3, CV => "ContadorSimiJ2");
   IF #_w31 THEN
       "ContadorSimiTempJ2" := "ContadorSimiJ2";
       "BloqueoSimilares6" := FALSE;
   END_IF;
   #_w32 := #_w25 AND "BloqueoSimilares7";
   IF #_w32 THEN "Var".CodigoSimilaresJ2[2] := 8; END_IF;
   "ContadorSimilaresJ2".CTU(CU := #_w32, R := "ReiniciarChecarSimiJ2", PV := 3, CV => "ContadorSimiJ2");
   IF #_w32 THEN
       "ContadorSimiTempJ2" := "ContadorSimiJ2";
       "BloqueoSimilares7" := FALSE;
   END_IF;
END_REGION

REGION Network 23: Azul J2
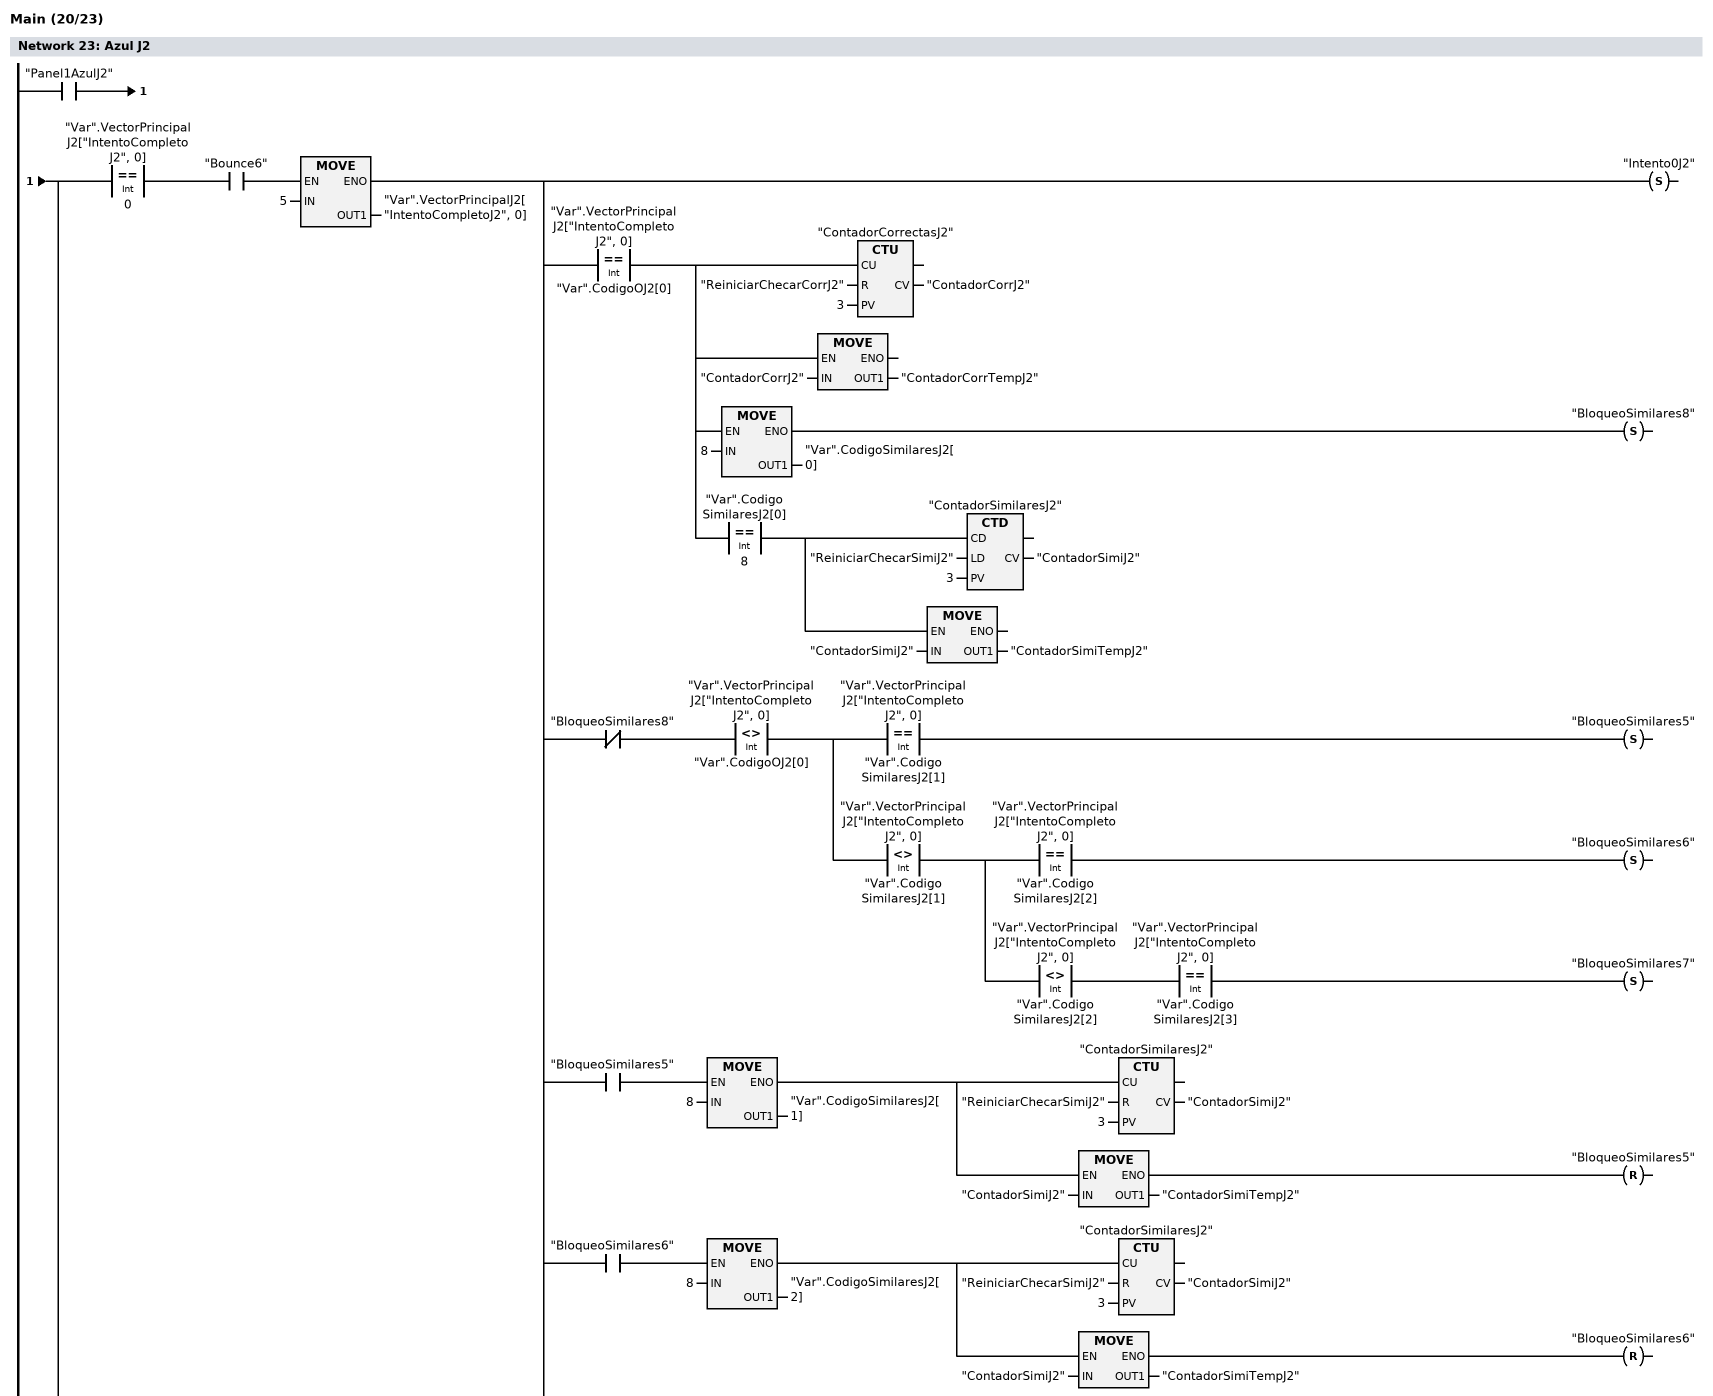
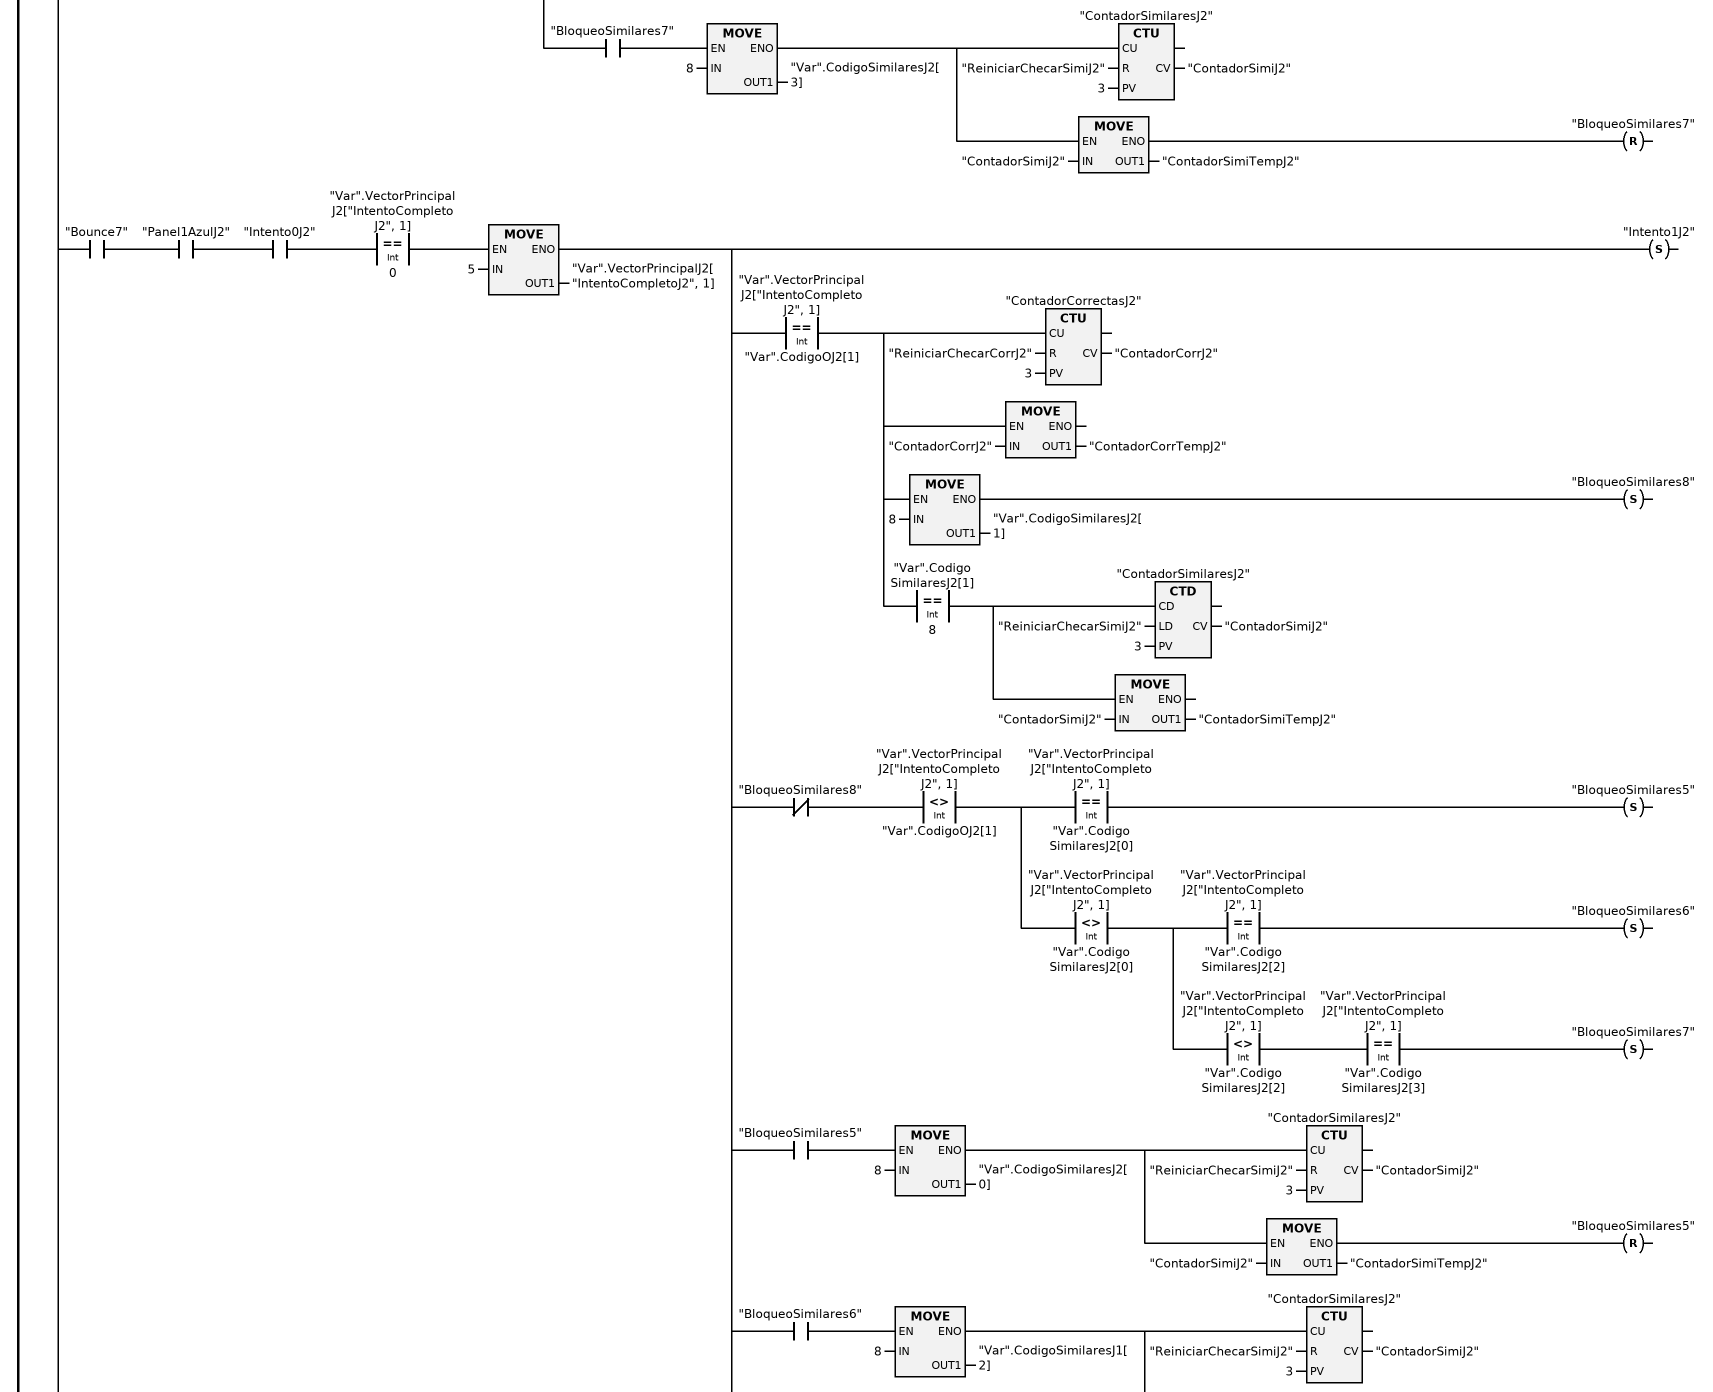
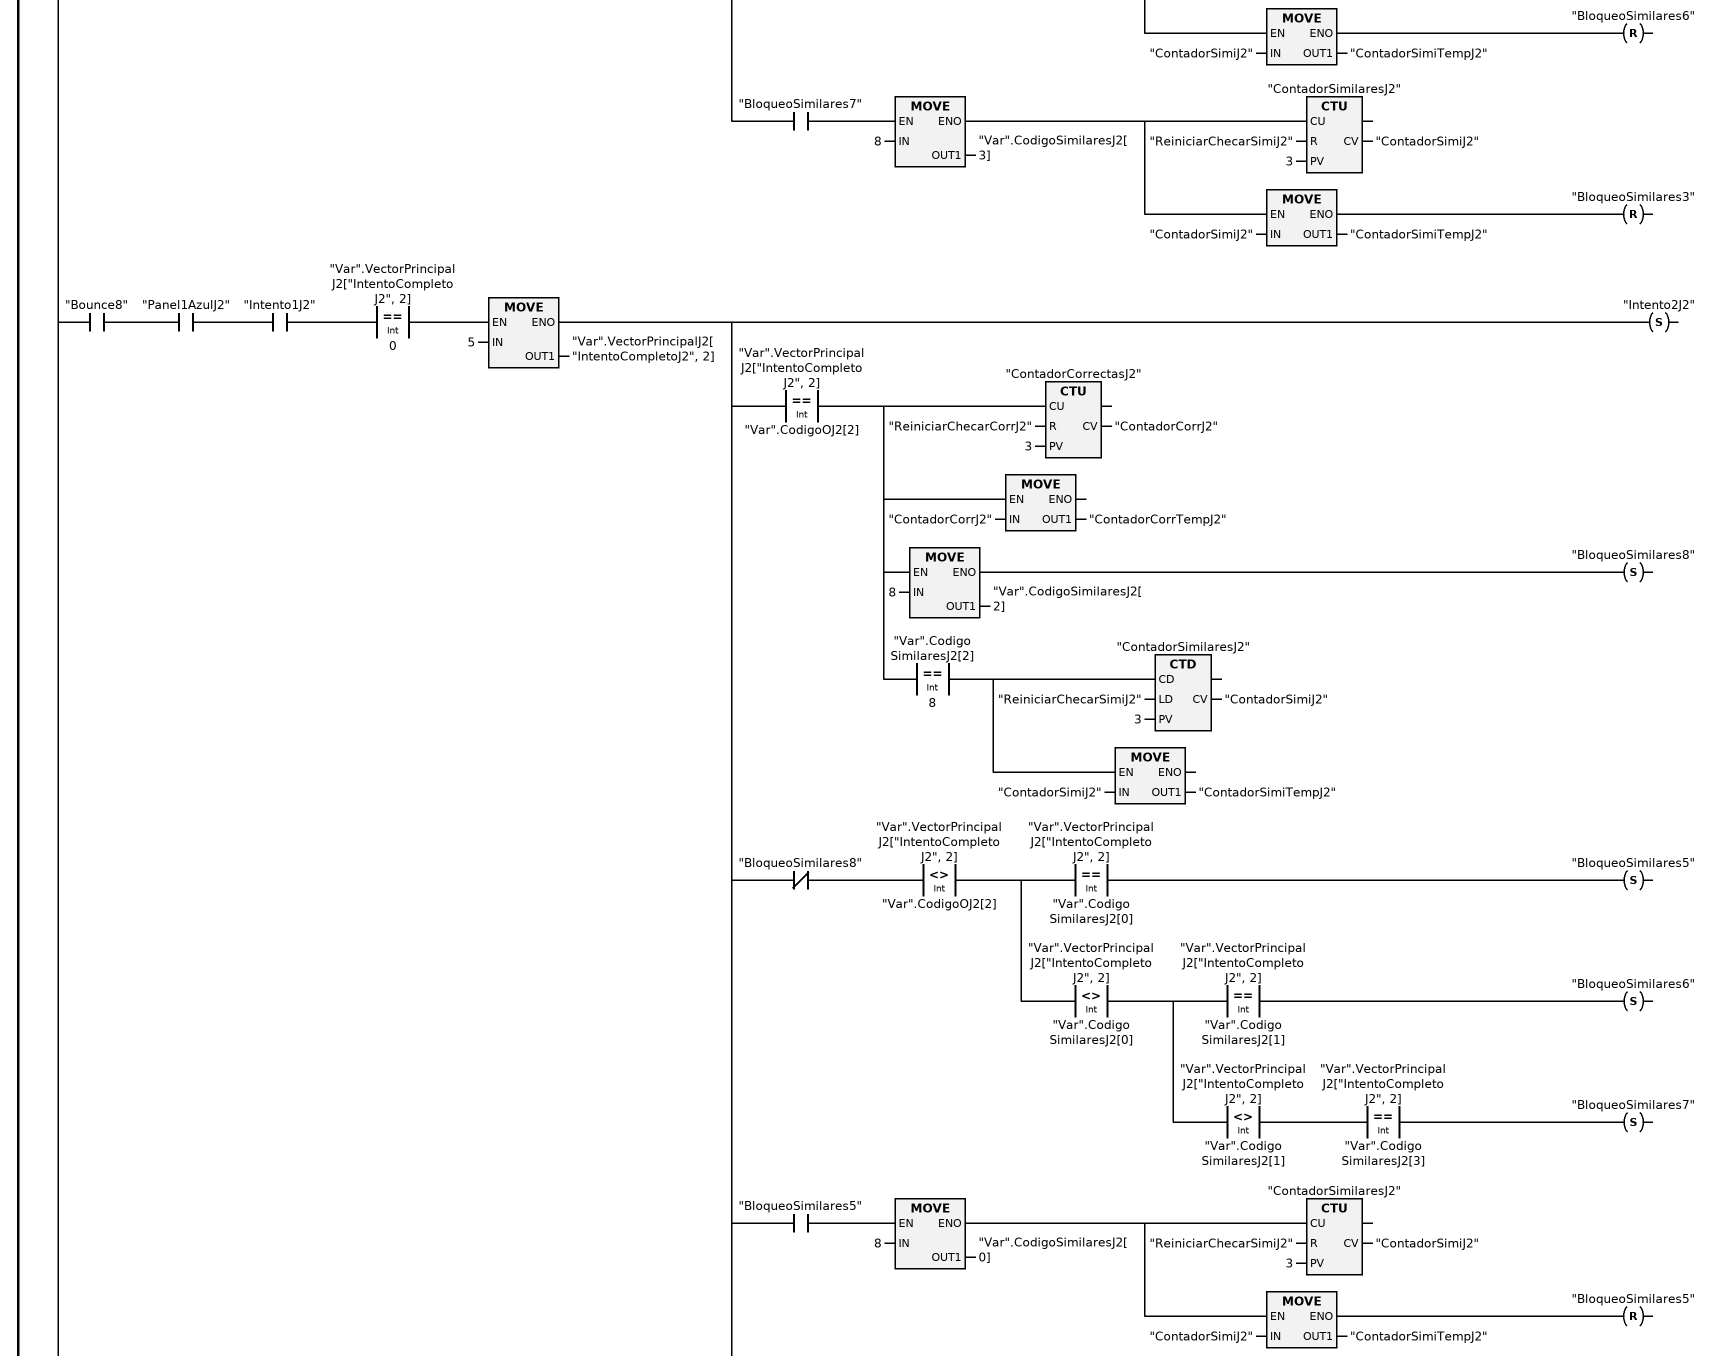
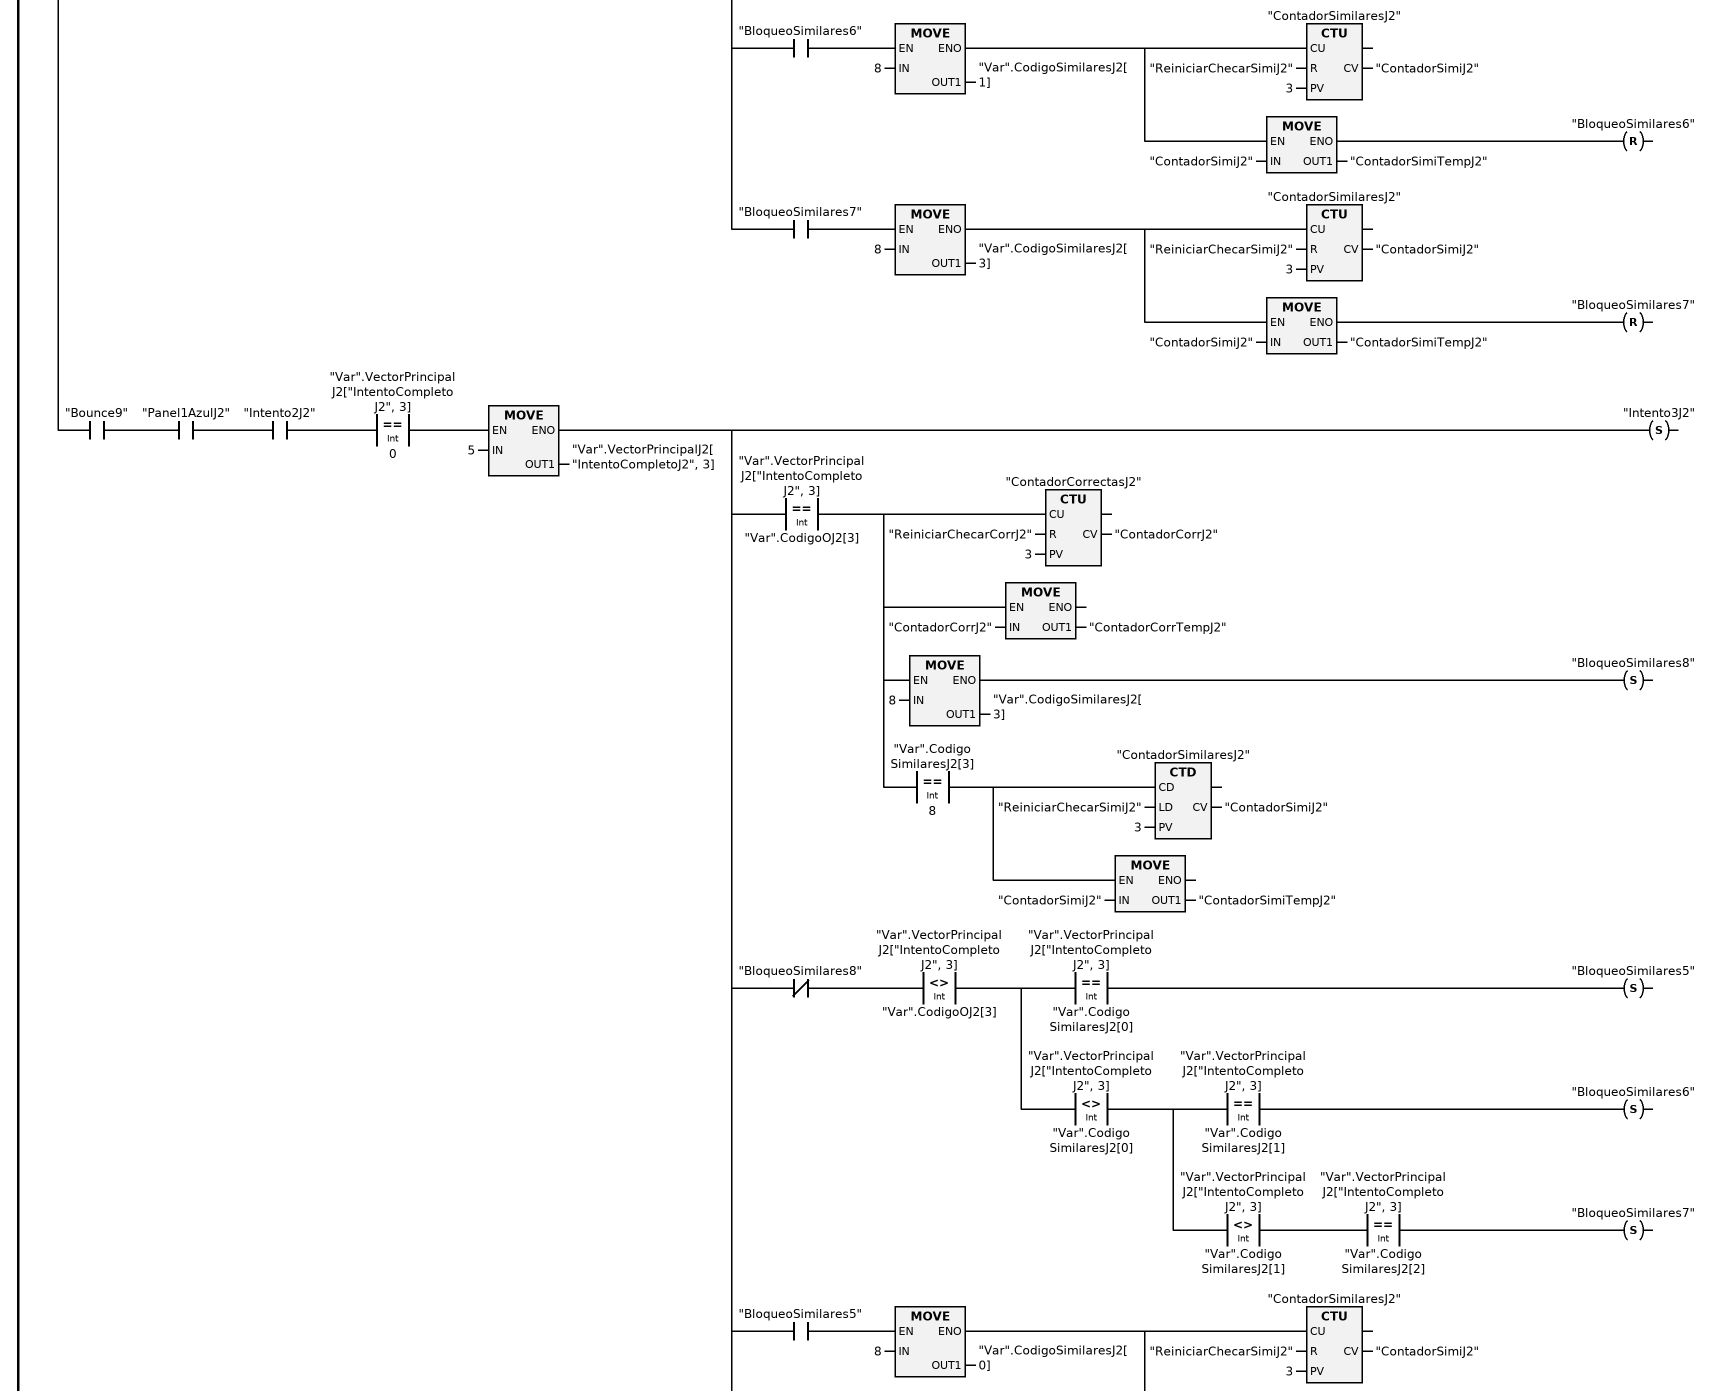
